REGION Network 4: CALL FB21013 POWDER FEEDER 1 HOPPER UNIT 02
   // 2#0000_0001 OPTIONS 0 BIT 0 LINE 1 ENABLED OPTION
   // 2#0000_0010 OPTIONS 0 BIT 1 LINE 2 ENABLED OPTION
   // 2#0000_0100 OPTIONS 0 BIT 2 SPARE
   // 2#0000_1000 OPTIONS 0 BIT 3 SPARE
   // 2#0001_0000 OPTIONS 0 BIT 4 SPARE
   // 2#0010_0000 OPTIONS 0 BIT 5 SPARE
   // 2#0100_0000 OPTIONS 0 BIT 6 SPARE
   // 2#1000_0000 OPTIONS 0 BIT 7 SPARE
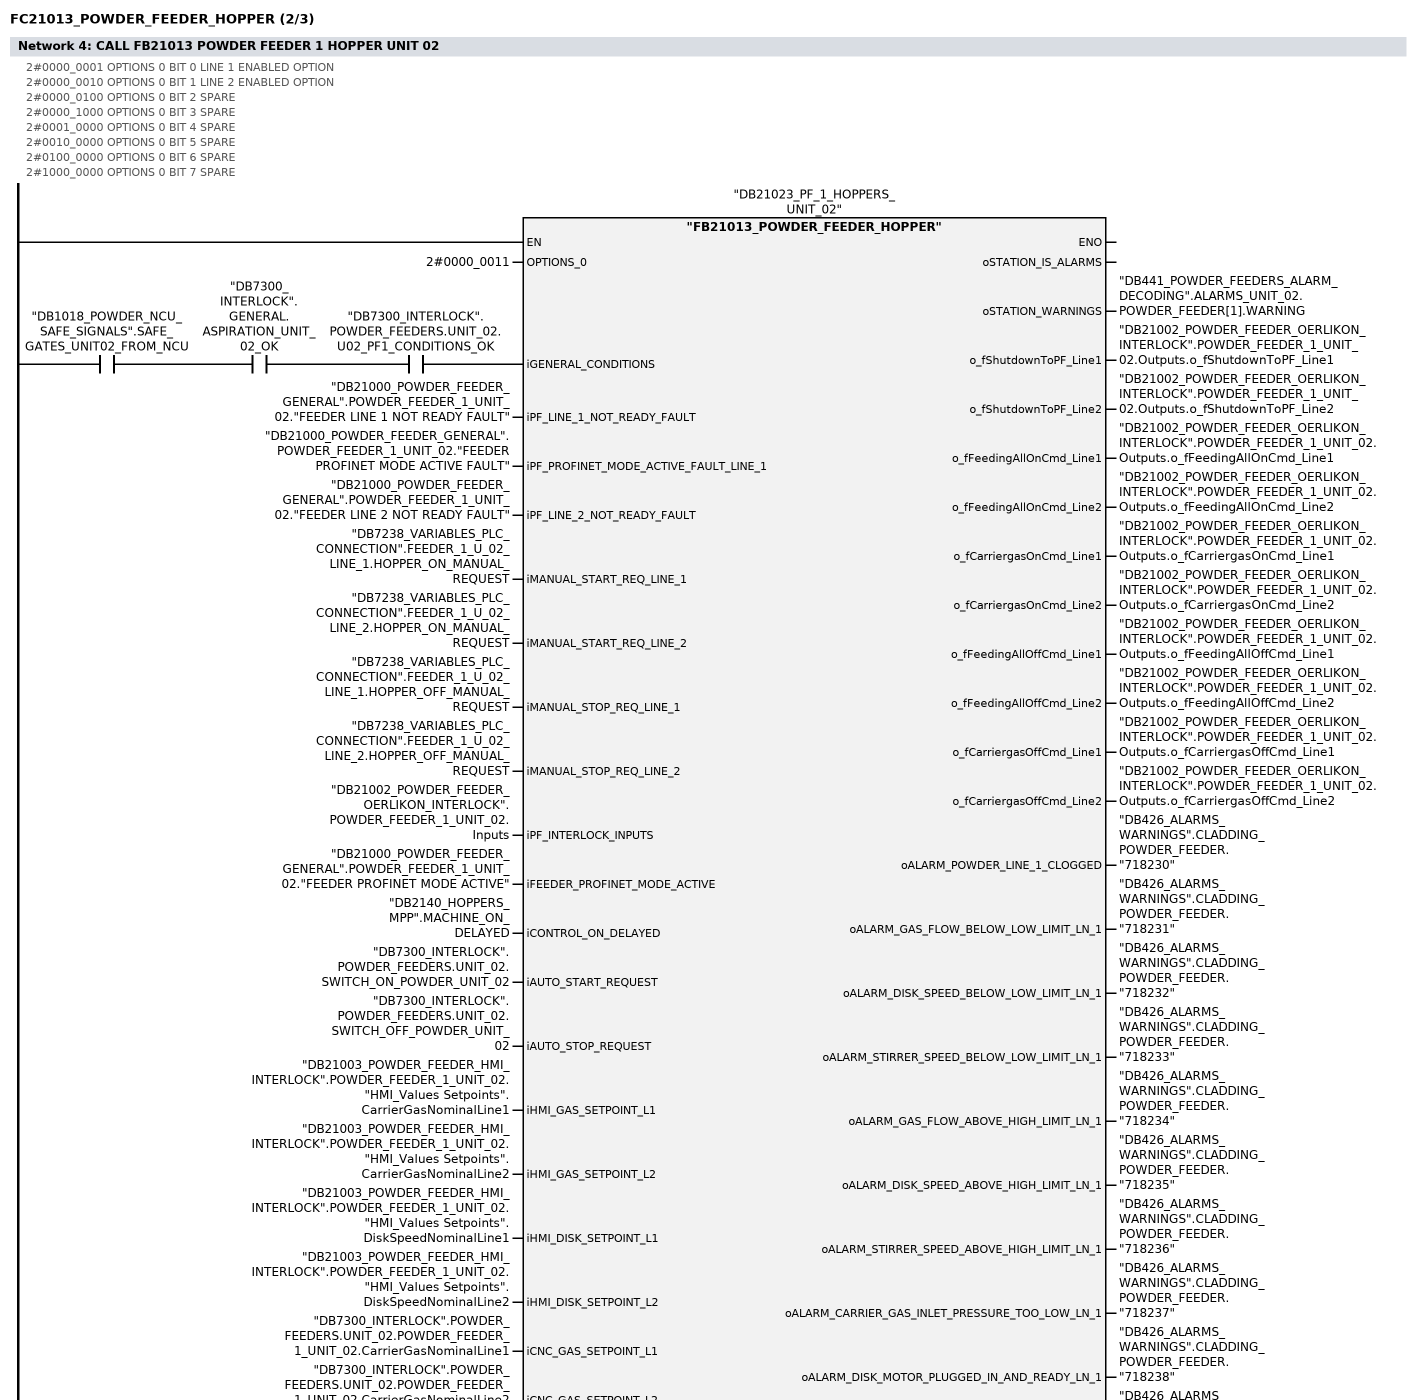
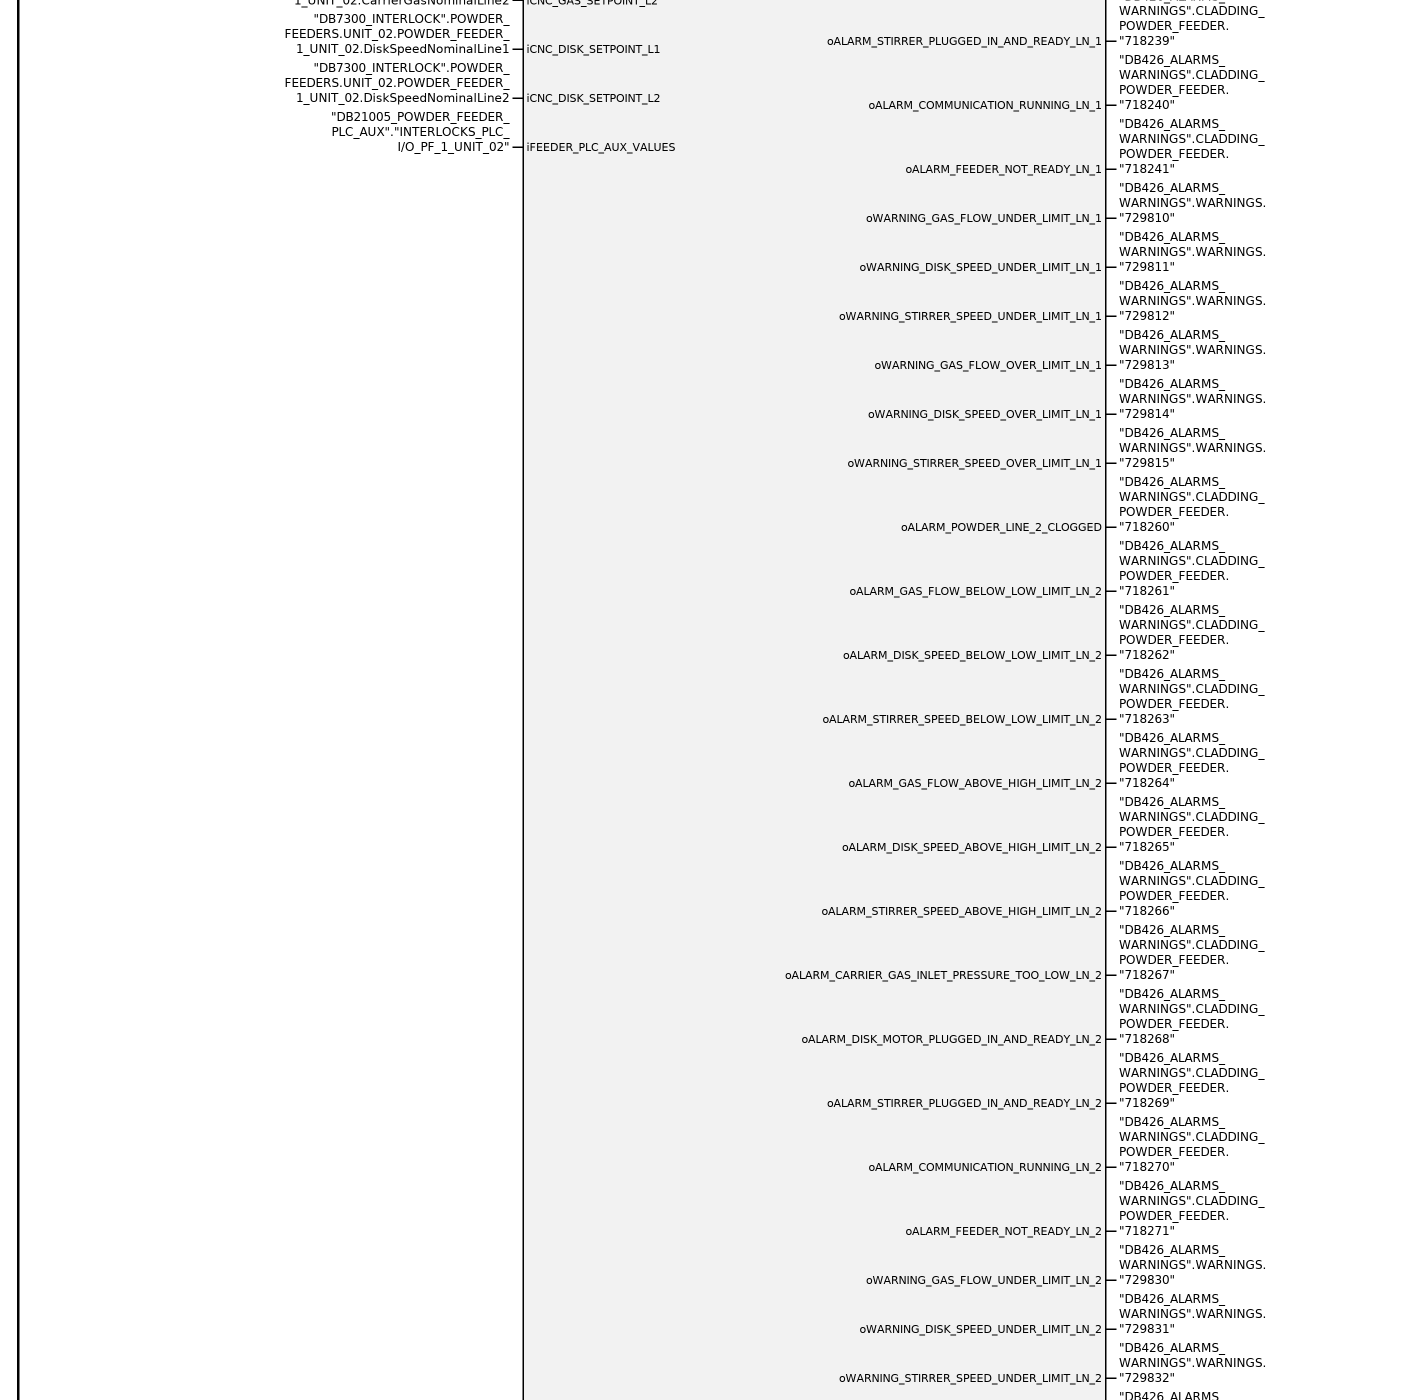
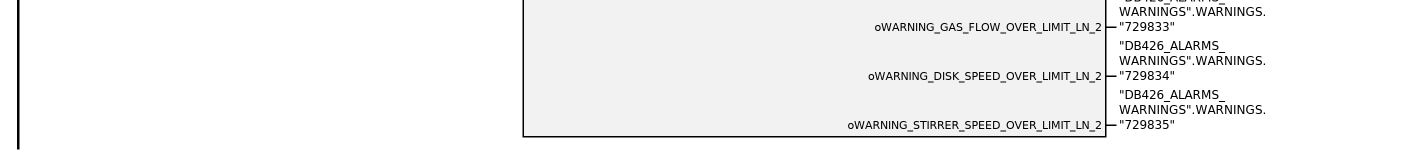
   RUNG wire#powerrail
      "DB21023_PF_1_HOPPERS_UNIT_02"(iGENERAL_CONDITIONS := wire#w1, OPTIONS_0 := 2#0000_0011, iPF_LINE_1_NOT_READY_FAULT := "DB21000_POWDER_FEEDER_GENERAL".POWDER_FEEDER_1_UNIT_02."FEEDER LINE 1 NOT READY FAULT", iPF_PROFINET_MODE_ACTIVE_FAULT_LINE_1 := "DB21000_POWDER_FEEDER_GENERAL".POWDER_FEEDER_1_UNIT_02."FEEDER PROFINET MODE ACTIVE FAULT", iPF_LINE_2_NOT_READY_FAULT := "DB21000_POWDER_FEEDER_GENERAL".POWDER_FEEDER_1_UNIT_02."FEEDER LINE 2 NOT READY FAULT", iMANUAL_START_REQ_LINE_1 := "DB7238_VARIABLES_PLC_CONNECTION".FEEDER_1_U_02_LINE_1.HOPPER_ON_MANUAL_REQUEST, iMANUAL_START_REQ_LINE_2 := "DB7238_VARIABLES_PLC_CONNECTION".FEEDER_1_U_02_LINE_2.HOPPER_ON_MANUAL_REQUEST, iMANUAL_STOP_REQ_LINE_1 := "DB7238_VARIABLES_PLC_CONNECTION".FEEDER_1_U_02_LINE_1.HOPPER_OFF_MANUAL_REQUEST, iMANUAL_STOP_REQ_LINE_2 := "DB7238_VARIABLES_PLC_CONNECTION".FEEDER_1_U_02_LINE_2.HOPPER_OFF_MANUAL_REQUEST, iPF_INTERLOCK_INPUTS := "DB21002_POWDER_FEEDER_OERLIKON_INTERLOCK".POWDER_FEEDER_1_UNIT_02.Inputs, iFEEDER_PROFINET_MODE_ACTIVE := "DB21000_POWDER_FEEDER_GENERAL".POWDER_FEEDER_1_UNIT_02."FEEDER PROFINET MODE ACTIVE", iCONTROL_ON_DELAYED := "DB2140_HOPPERS_MPP".MACHINE_ON_DELAYED, iAUTO_START_REQUEST := "DB7300_INTERLOCK".POWDER_FEEDERS.UNIT_02.SWITCH_ON_POWDER_UNIT_02, iAUTO_STOP_REQUEST := "DB7300_INTERLOCK".POWDER_FEEDERS.UNIT_02.SWITCH_OFF_POWDER_UNIT_02, iHMI_GAS_SETPOINT_L1 := "DB21003_POWDER_FEEDER_HMI_INTERLOCK".POWDER_FEEDER_1_UNIT_02."HMI_Values Setpoints".CarrierGasNominalLine1, iHMI_GAS_SETPOINT_L2 := "DB21003_POWDER_FEEDER_HMI_INTERLOCK".POWDER_FEEDER_1_UNIT_02."HMI_Values Setpoints".CarrierGasNominalLine2, iHMI_DISK_SETPOINT_L1 := "DB21003_POWDER_FEEDER_HMI_INTERLOCK".POWDER_FEEDER_1_UNIT_02."HMI_Values Setpoints".DiskSpeedNominalLine1, iHMI_DISK_SETPOINT_L2 := "DB21003_POWDER_FEEDER_HMI_INTERLOCK".POWDER_FEEDER_1_UNIT_02."HMI_Values Setpoints".DiskSpeedNominalLine2, iCNC_GAS_SETPOINT_L1 := "DB7300_INTERLOCK".POWDER_FEEDERS.UNIT_02.POWDER_FEEDER_1_UNIT_02.CarrierGasNominalLine1, iCNC_GAS_SETPOINT_L2 := "DB7300_INTERLOCK".POWDER_FEEDERS.UNIT_02.POWDER_FEEDER_1_UNIT_02.CarrierGasNominalLine2, iCNC_DISK_SETPOINT_L1 := "DB7300_INTERLOCK".POWDER_FEEDERS.UNIT_02.POWDER_FEEDER_1_UNIT_02.DiskSpeedNominalLine1, iCNC_DISK_SETPOINT_L2 := "DB7300_INTERLOCK".POWDER_FEEDERS.UNIT_02.POWDER_FEEDER_1_UNIT_02.DiskSpeedNominalLine2, iFEEDER_PLC_AUX_VALUES := "DB21005_POWDER_FEEDER_PLC_AUX"."INTERLOCKS_PLC_I/O_PF_1_UNIT_02", oSTATION_IS_ALARMS =>, oSTATION_WARNINGS => "DB441_POWDER_FEEDERS_ALARM_DECODING".ALARMS_UNIT_02.POWDER_FEEDER[1].WARNING, o_fShutdownToPF_Line1 => "DB21002_POWDER_FEEDER_OERLIKON_INTERLOCK".POWDER_FEEDER_1_UNIT_02.Outputs.o_fShutdownToPF_Line1, o_fShutdownToPF_Line2 => "DB21002_POWDER_FEEDER_OERLIKON_INTERLOCK".POWDER_FEEDER_1_UNIT_02.Outputs.o_fShutdownToPF_Line2, o_fFeedingAllOnCmd_Line1 => "DB21002_POWDER_FEEDER_OERLIKON_INTERLOCK".POWDER_FEEDER_1_UNIT_02.Outputs.o_fFeedingAllOnCmd_Line1, o_fFeedingAllOnCmd_Line2 => "DB21002_POWDER_FEEDER_OERLIKON_INTERLOCK".POWDER_FEEDER_1_UNIT_02.Outputs.o_fFeedingAllOnCmd_Line2, o_fCarriergasOnCmd_Line1 => "DB21002_POWDER_FEEDER_OERLIKON_INTERLOCK".POWDER_FEEDER_1_UNIT_02.Outputs.o_fCarriergasOnCmd_Line1, o_fCarriergasOnCmd_Line2 => "DB21002_POWDER_FEEDER_OERLIKON_INTERLOCK".POWDER_FEEDER_1_UNIT_02.Outputs.o_fCarriergasOnCmd_Line2, o_fFeedingAllOffCmd_Line1 => "DB21002_POWDER_FEEDER_OERLIKON_INTERLOCK".POWDER_FEEDER_1_UNIT_02.Outputs.o_fFeedingAllOffCmd_Line1, o_fFeedingAllOffCmd_Line2 => "DB21002_POWDER_FEEDER_OERLIKON_INTERLOCK".POWDER_FEEDER_1_UNIT_02.Outputs.o_fFeedingAllOffCmd_Line2, o_fCarriergasOffCmd_Line1 => "DB21002_POWDER_FEEDER_OERLIKON_INTERLOCK".POWDER_FEEDER_1_UNIT_02.Outputs.o_fCarriergasOffCmd_Line1, o_fCarriergasOffCmd_Line2 => "DB21002_POWDER_FEEDER_OERLIKON_INTERLOCK".POWDER_FEEDER_1_UNIT_02.Outputs.o_fCarriergasOffCmd_Line2, oALARM_POWDER_LINE_1_CLOGGED => "DB426_ALARMS_WARNINGS".CLADDING_POWDER_FEEDER."718230", oALARM_GAS_FLOW_BELOW_LOW_LIMIT_LN_1 => "DB426_ALARMS_WARNINGS".CLADDING_POWDER_FEEDER."718231", oALARM_DISK_SPEED_BELOW_LOW_LIMIT_LN_1 => "DB426_ALARMS_WARNINGS".CLADDING_POWDER_FEEDER."718232", oALARM_STIRRER_SPEED_BELOW_LOW_LIMIT_LN_1 => "DB426_ALARMS_WARNINGS".CLADDING_POWDER_FEEDER."718233", oALARM_GAS_FLOW_ABOVE_HIGH_LIMIT_LN_1 => "DB426_ALARMS_WARNINGS".CLADDING_POWDER_FEEDER."718234", oALARM_DISK_SPEED_ABOVE_HIGH_LIMIT_LN_1 => "DB426_ALARMS_WARNINGS".CLADDING_POWDER_FEEDER."718235", oALARM_STIRRER_SPEED_ABOVE_HIGH_LIMIT_LN_1 => "DB426_ALARMS_WARNINGS".CLADDING_POWDER_FEEDER."718236", oALARM_CARRIER_GAS_INLET_PRESSURE_TOO_LOW_LN_1 => "DB426_ALARMS_WARNINGS".CLADDING_POWDER_FEEDER."718237", oALARM_DISK_MOTOR_PLUGGED_IN_AND_READY_LN_1 => "DB426_ALARMS_WARNINGS".CLADDING_POWDER_FEEDER."718238", oALARM_STIRRER_PLUGGED_IN_AND_READY_LN_1 => "DB426_ALARMS_WARNINGS".CLADDING_POWDER_FEEDER."718239", oALARM_COMMUNICATION_RUNNING_LN_1 => "DB426_ALARMS_WARNINGS".CLADDING_POWDER_FEEDER."718240", oALARM_FEEDER_NOT_READY_LN_1 => "DB426_ALARMS_WARNINGS".CLADDING_POWDER_FEEDER."718241", oWARNING_GAS_FLOW_UNDER_LIMIT_LN_1 => "DB426_ALARMS_WARNINGS".WARNINGS."729810", oWARNING_DISK_SPEED_UNDER_LIMIT_LN_1 => "DB426_ALARMS_WARNINGS".WARNINGS."729811", oWARNING_STIRRER_SPEED_UNDER_LIMIT_LN_1 => "DB426_ALARMS_WARNINGS".WARNINGS."729812", oWARNING_GAS_FLOW_OVER_LIMIT_LN_1 => "DB426_ALARMS_WARNINGS".WARNINGS."729813", oWARNING_DISK_SPEED_OVER_LIMIT_LN_1 => "DB426_ALARMS_WARNINGS".WARNINGS."729814", oWARNING_STIRRER_SPEED_OVER_LIMIT_LN_1 => "DB426_ALARMS_WARNINGS".WARNINGS."729815", oALARM_POWDER_LINE_2_CLOGGED => "DB426_ALARMS_WARNINGS".CLADDING_POWDER_FEEDER."718260", oALARM_GAS_FLOW_BELOW_LOW_LIMIT_LN_2 => "DB426_ALARMS_WARNINGS".CLADDING_POWDER_FEEDER."718261", oALARM_DISK_SPEED_BELOW_LOW_LIMIT_LN_2 => "DB426_ALARMS_WARNINGS".CLADDING_POWDER_FEEDER."718262", oALARM_STIRRER_SPEED_BELOW_LOW_LIMIT_LN_2 => "DB426_ALARMS_WARNINGS".CLADDING_POWDER_FEEDER."718263", oALARM_GAS_FLOW_ABOVE_HIGH_LIMIT_LN_2 => "DB426_ALARMS_WARNINGS".CLADDING_POWDER_FEEDER."718264", oALARM_DISK_SPEED_ABOVE_HIGH_LIMIT_LN_2 => "DB426_ALARMS_WARNINGS".CLADDING_POWDER_FEEDER."718265", oALARM_STIRRER_SPEED_ABOVE_HIGH_LIMIT_LN_2 => "DB426_ALARMS_WARNINGS".CLADDING_POWDER_FEEDER."718266", oALARM_CARRIER_GAS_INLET_PRESSURE_TOO_LOW_LN_2 => "DB426_ALARMS_WARNINGS".CLADDING_POWDER_FEEDER."718267", oALARM_DISK_MOTOR_PLUGGED_IN_AND_READY_LN_2 => "DB426_ALARMS_WARNINGS".CLADDING_POWDER_FEEDER."718268", oALARM_STIRRER_PLUGGED_IN_AND_READY_LN_2 => "DB426_ALARMS_WARNINGS".CLADDING_POWDER_FEEDER."718269", oALARM_COMMUNICATION_RUNNING_LN_2 => "DB426_ALARMS_WARNINGS".CLADDING_POWDER_FEEDER."718270", oALARM_FEEDER_NOT_READY_LN_2 => "DB426_ALARMS_WARNINGS".CLADDING_POWDER_FEEDER."718271", oWARNING_GAS_FLOW_UNDER_LIMIT_LN_2 => "DB426_ALARMS_WARNINGS".WARNINGS."729830", oWARNING_DISK_SPEED_UNDER_LIMIT_LN_2 => "DB426_ALARMS_WARNINGS".WARNINGS."729831", oWARNING_STIRRER_SPEED_UNDER_LIMIT_LN_2 => "DB426_ALARMS_WARNINGS".WARNINGS."729832", oWARNING_GAS_FLOW_OVER_LIMIT_LN_2 => "DB426_ALARMS_WARNINGS".WARNINGS."729833", oWARNING_DISK_SPEED_OVER_LIMIT_LN_2 => "DB426_ALARMS_WARNINGS".WARNINGS."729834", oWARNING_STIRRER_SPEED_OVER_LIMIT_LN_2 => "DB426_ALARMS_WARNINGS".WARNINGS."729835")
   END_RUNG
   RUNG wire#powerrail
      Contact( "DB1018_POWDER_NCU_SAFE_SIGNALS".SAFE_GATES_UNIT02_FROM_NCU )
      Contact( "DB7300_INTERLOCK".GENERAL.ASPIRATION_UNIT_02_OK )
      Contact( "DB7300_INTERLOCK".POWDER_FEEDERS.UNIT_02.U02_PF1_CONDITIONS_OK )
   END_RUNG wire#w1
   // the same network as SCL:
   "DB21023_PF_1_HOPPERS_UNIT_02"(OPTIONS_0 := 2#0000_0011,   // "FB21013_POWDER_FEEDER_HOPPER"
                           iGENERAL_CONDITIONS := "DB1018_POWDER_NCU_SAFE_SIGNALS".SAFE_GATES_UNIT02_FROM_NCU AND "DB7300_INTERLOCK".GENERAL.ASPIRATION_UNIT_02_OK AND "DB7300_INTERLOCK".POWDER_FEEDERS.UNIT_02.U02_PF1_CONDITIONS_OK,
                           iPF_LINE_1_NOT_READY_FAULT := "DB21000_POWDER_FEEDER_GENERAL".POWDER_FEEDER_1_UNIT_02."FEEDER LINE 1 NOT READY FAULT",
                           iPF_PROFINET_MODE_ACTIVE_FAULT_LINE_1 := "DB21000_POWDER_FEEDER_GENERAL".POWDER_FEEDER_1_UNIT_02."FEEDER PROFINET MODE ACTIVE FAULT",
                           iPF_LINE_2_NOT_READY_FAULT := "DB21000_POWDER_FEEDER_GENERAL".POWDER_FEEDER_1_UNIT_02."FEEDER LINE 2 NOT READY FAULT",
                           iMANUAL_START_REQ_LINE_1 := "DB7238_VARIABLES_PLC_CONNECTION".FEEDER_1_U_02_LINE_1.HOPPER_ON_MANUAL_REQUEST,
                           iMANUAL_START_REQ_LINE_2 := "DB7238_VARIABLES_PLC_CONNECTION".FEEDER_1_U_02_LINE_2.HOPPER_ON_MANUAL_REQUEST,
                           iMANUAL_STOP_REQ_LINE_1 := "DB7238_VARIABLES_PLC_CONNECTION".FEEDER_1_U_02_LINE_1.HOPPER_OFF_MANUAL_REQUEST,
                           iMANUAL_STOP_REQ_LINE_2 := "DB7238_VARIABLES_PLC_CONNECTION".FEEDER_1_U_02_LINE_2.HOPPER_OFF_MANUAL_REQUEST,
                           iPF_INTERLOCK_INPUTS := "DB21002_POWDER_FEEDER_OERLIKON_INTERLOCK".POWDER_FEEDER_1_UNIT_02.Inputs,
                           iFEEDER_PROFINET_MODE_ACTIVE := "DB21000_POWDER_FEEDER_GENERAL".POWDER_FEEDER_1_UNIT_02."FEEDER PROFINET MODE ACTIVE",
                           iCONTROL_ON_DELAYED := "DB2140_HOPPERS_MPP".MACHINE_ON_DELAYED,
                           iAUTO_START_REQUEST := "DB7300_INTERLOCK".POWDER_FEEDERS.UNIT_02.SWITCH_ON_POWDER_UNIT_02,
                           iAUTO_STOP_REQUEST := "DB7300_INTERLOCK".POWDER_FEEDERS.UNIT_02.SWITCH_OFF_POWDER_UNIT_02,
                           iHMI_GAS_SETPOINT_L1 := "DB21003_POWDER_FEEDER_HMI_INTERLOCK".POWDER_FEEDER_1_UNIT_02."HMI_Values Setpoints".CarrierGasNominalLine1,
                           iHMI_GAS_SETPOINT_L2 := "DB21003_POWDER_FEEDER_HMI_INTERLOCK".POWDER_FEEDER_1_UNIT_02."HMI_Values Setpoints".CarrierGasNominalLine2,
                           iHMI_DISK_SETPOINT_L1 := "DB21003_POWDER_FEEDER_HMI_INTERLOCK".POWDER_FEEDER_1_UNIT_02."HMI_Values Setpoints".DiskSpeedNominalLine1,
                           iHMI_DISK_SETPOINT_L2 := "DB21003_POWDER_FEEDER_HMI_INTERLOCK".POWDER_FEEDER_1_UNIT_02."HMI_Values Setpoints".DiskSpeedNominalLine2,
                           iCNC_GAS_SETPOINT_L1 := "DB7300_INTERLOCK".POWDER_FEEDERS.UNIT_02.POWDER_FEEDER_1_UNIT_02.CarrierGasNominalLine1,
                           iCNC_GAS_SETPOINT_L2 := "DB7300_INTERLOCK".POWDER_FEEDERS.UNIT_02.POWDER_FEEDER_1_UNIT_02.CarrierGasNominalLine2,
                           iCNC_DISK_SETPOINT_L1 := "DB7300_INTERLOCK".POWDER_FEEDERS.UNIT_02.POWDER_FEEDER_1_UNIT_02.DiskSpeedNominalLine1,
                           iCNC_DISK_SETPOINT_L2 := "DB7300_INTERLOCK".POWDER_FEEDERS.UNIT_02.POWDER_FEEDER_1_UNIT_02.DiskSpeedNominalLine2,
                           iFEEDER_PLC_AUX_VALUES := "DB21005_POWDER_FEEDER_PLC_AUX"."INTERLOCKS_PLC_I/O_PF_1_UNIT_02",
                           oSTATION_WARNINGS => "DB441_POWDER_FEEDERS_ALARM_DECODING".ALARMS_UNIT_02.POWDER_FEEDER[1].WARNING,
                           o_fShutdownToPF_Line1 => "DB21002_POWDER_FEEDER_OERLIKON_INTERLOCK".POWDER_FEEDER_1_UNIT_02.Outputs.o_fShutdownToPF_Line1,
                           o_fShutdownToPF_Line2 => "DB21002_POWDER_FEEDER_OERLIKON_INTERLOCK".POWDER_FEEDER_1_UNIT_02.Outputs.o_fShutdownToPF_Line2,
                           o_fFeedingAllOnCmd_Line1 => "DB21002_POWDER_FEEDER_OERLIKON_INTERLOCK".POWDER_FEEDER_1_UNIT_02.Outputs.o_fFeedingAllOnCmd_Line1,
                           o_fFeedingAllOnCmd_Line2 => "DB21002_POWDER_FEEDER_OERLIKON_INTERLOCK".POWDER_FEEDER_1_UNIT_02.Outputs.o_fFeedingAllOnCmd_Line2,
                           o_fCarriergasOnCmd_Line1 => "DB21002_POWDER_FEEDER_OERLIKON_INTERLOCK".POWDER_FEEDER_1_UNIT_02.Outputs.o_fCarriergasOnCmd_Line1,
                           o_fCarriergasOnCmd_Line2 => "DB21002_POWDER_FEEDER_OERLIKON_INTERLOCK".POWDER_FEEDER_1_UNIT_02.Outputs.o_fCarriergasOnCmd_Line2,
                           o_fFeedingAllOffCmd_Line1 => "DB21002_POWDER_FEEDER_OERLIKON_INTERLOCK".POWDER_FEEDER_1_UNIT_02.Outputs.o_fFeedingAllOffCmd_Line1,
                           o_fFeedingAllOffCmd_Line2 => "DB21002_POWDER_FEEDER_OERLIKON_INTERLOCK".POWDER_FEEDER_1_UNIT_02.Outputs.o_fFeedingAllOffCmd_Line2,
                           o_fCarriergasOffCmd_Line1 => "DB21002_POWDER_FEEDER_OERLIKON_INTERLOCK".POWDER_FEEDER_1_UNIT_02.Outputs.o_fCarriergasOffCmd_Line1,
                           o_fCarriergasOffCmd_Line2 => "DB21002_POWDER_FEEDER_OERLIKON_INTERLOCK".POWDER_FEEDER_1_UNIT_02.Outputs.o_fCarriergasOffCmd_Line2,
                           oALARM_POWDER_LINE_1_CLOGGED => "DB426_ALARMS_WARNINGS".CLADDING_POWDER_FEEDER."718230",
                           oALARM_GAS_FLOW_BELOW_LOW_LIMIT_LN_1 => "DB426_ALARMS_WARNINGS".CLADDING_POWDER_FEEDER."718231",
                           oALARM_DISK_SPEED_BELOW_LOW_LIMIT_LN_1 => "DB426_ALARMS_WARNINGS".CLADDING_POWDER_FEEDER."718232",
                           oALARM_STIRRER_SPEED_BELOW_LOW_LIMIT_LN_1 => "DB426_ALARMS_WARNINGS".CLADDING_POWDER_FEEDER."718233",
                           oALARM_GAS_FLOW_ABOVE_HIGH_LIMIT_LN_1 => "DB426_ALARMS_WARNINGS".CLADDING_POWDER_FEEDER."718234",
                           oALARM_DISK_SPEED_ABOVE_HIGH_LIMIT_LN_1 => "DB426_ALARMS_WARNINGS".CLADDING_POWDER_FEEDER."718235",
                           oALARM_STIRRER_SPEED_ABOVE_HIGH_LIMIT_LN_1 => "DB426_ALARMS_WARNINGS".CLADDING_POWDER_FEEDER."718236",
                           oALARM_CARRIER_GAS_INLET_PRESSURE_TOO_LOW_LN_1 => "DB426_ALARMS_WARNINGS".CLADDING_POWDER_FEEDER."718237",
                           oALARM_DISK_MOTOR_PLUGGED_IN_AND_READY_LN_1 => "DB426_ALARMS_WARNINGS".CLADDING_POWDER_FEEDER."718238",
                           oALARM_STIRRER_PLUGGED_IN_AND_READY_LN_1 => "DB426_ALARMS_WARNINGS".CLADDING_POWDER_FEEDER."718239",
                           oALARM_COMMUNICATION_RUNNING_LN_1 => "DB426_ALARMS_WARNINGS".CLADDING_POWDER_FEEDER."718240",
                           oALARM_FEEDER_NOT_READY_LN_1 => "DB426_ALARMS_WARNINGS".CLADDING_POWDER_FEEDER."718241",
                           oWARNING_GAS_FLOW_UNDER_LIMIT_LN_1 => "DB426_ALARMS_WARNINGS".WARNINGS."729810",
                           oWARNING_DISK_SPEED_UNDER_LIMIT_LN_1 => "DB426_ALARMS_WARNINGS".WARNINGS."729811",
                           oWARNING_STIRRER_SPEED_UNDER_LIMIT_LN_1 => "DB426_ALARMS_WARNINGS".WARNINGS."729812",
                           oWARNING_GAS_FLOW_OVER_LIMIT_LN_1 => "DB426_ALARMS_WARNINGS".WARNINGS."729813",
                           oWARNING_DISK_SPEED_OVER_LIMIT_LN_1 => "DB426_ALARMS_WARNINGS".WARNINGS."729814",
                           oWARNING_STIRRER_SPEED_OVER_LIMIT_LN_1 => "DB426_ALARMS_WARNINGS".WARNINGS."729815",
                           oALARM_POWDER_LINE_2_CLOGGED => "DB426_ALARMS_WARNINGS".CLADDING_POWDER_FEEDER."718260",
                           oALARM_GAS_FLOW_BELOW_LOW_LIMIT_LN_2 => "DB426_ALARMS_WARNINGS".CLADDING_POWDER_FEEDER."718261",
                           oALARM_DISK_SPEED_BELOW_LOW_LIMIT_LN_2 => "DB426_ALARMS_WARNINGS".CLADDING_POWDER_FEEDER."718262",
                           oALARM_STIRRER_SPEED_BELOW_LOW_LIMIT_LN_2 => "DB426_ALARMS_WARNINGS".CLADDING_POWDER_FEEDER."718263",
                           oALARM_GAS_FLOW_ABOVE_HIGH_LIMIT_LN_2 => "DB426_ALARMS_WARNINGS".CLADDING_POWDER_FEEDER."718264",
                           oALARM_DISK_SPEED_ABOVE_HIGH_LIMIT_LN_2 => "DB426_ALARMS_WARNINGS".CLADDING_POWDER_FEEDER."718265",
                           oALARM_STIRRER_SPEED_ABOVE_HIGH_LIMIT_LN_2 => "DB426_ALARMS_WARNINGS".CLADDING_POWDER_FEEDER."718266",
                           oALARM_CARRIER_GAS_INLET_PRESSURE_TOO_LOW_LN_2 => "DB426_ALARMS_WARNINGS".CLADDING_POWDER_FEEDER."718267",
                           oALARM_DISK_MOTOR_PLUGGED_IN_AND_READY_LN_2 => "DB426_ALARMS_WARNINGS".CLADDING_POWDER_FEEDER."718268",
                           oALARM_STIRRER_PLUGGED_IN_AND_READY_LN_2 => "DB426_ALARMS_WARNINGS".CLADDING_POWDER_FEEDER."718269",
                           oALARM_COMMUNICATION_RUNNING_LN_2 => "DB426_ALARMS_WARNINGS".CLADDING_POWDER_FEEDER."718270",
                           oALARM_FEEDER_NOT_READY_LN_2 => "DB426_ALARMS_WARNINGS".CLADDING_POWDER_FEEDER."718271",
                           oWARNING_GAS_FLOW_UNDER_LIMIT_LN_2 => "DB426_ALARMS_WARNINGS".WARNINGS."729830",
                           oWARNING_DISK_SPEED_UNDER_LIMIT_LN_2 => "DB426_ALARMS_WARNINGS".WARNINGS."729831",
                           oWARNING_STIRRER_SPEED_UNDER_LIMIT_LN_2 => "DB426_ALARMS_WARNINGS".WARNINGS."729832",
                           oWARNING_GAS_FLOW_OVER_LIMIT_LN_2 => "DB426_ALARMS_WARNINGS".WARNINGS."729833",
                           oWARNING_DISK_SPEED_OVER_LIMIT_LN_2 => "DB426_ALARMS_WARNINGS".WARNINGS."729834",
                           oWARNING_STIRRER_SPEED_OVER_LIMIT_LN_2 => "DB426_ALARMS_WARNINGS".WARNINGS."729835");
END_REGION

REGION Network 5: CALL FB21013 POWDER FEEDER 2 HOPPER UNIT 02
   // 2#0000_0001 OPTIONS 0 BIT 0 LINE 1 ENABLED OPTION
   // 2#0000_0010 OPTIONS 0 BIT 1 LINE 2 ENABLED OPTION
   // 2#0000_0100 OPTIONS 0 BIT 2 SPARE
   // 2#0000_1000 OPTIONS 0 BIT 3 SPARE
   // 2#0001_0000 OPTIONS 0 BIT 4 SPARE
   // 2#0010_0000 OPTIONS 0 BIT 5 SPARE
   // 2#0100_0000 OPTIONS 0 BIT 6 SPARE
   // 2#1000_0000 OPTIONS 0 BIT 7 SPARE
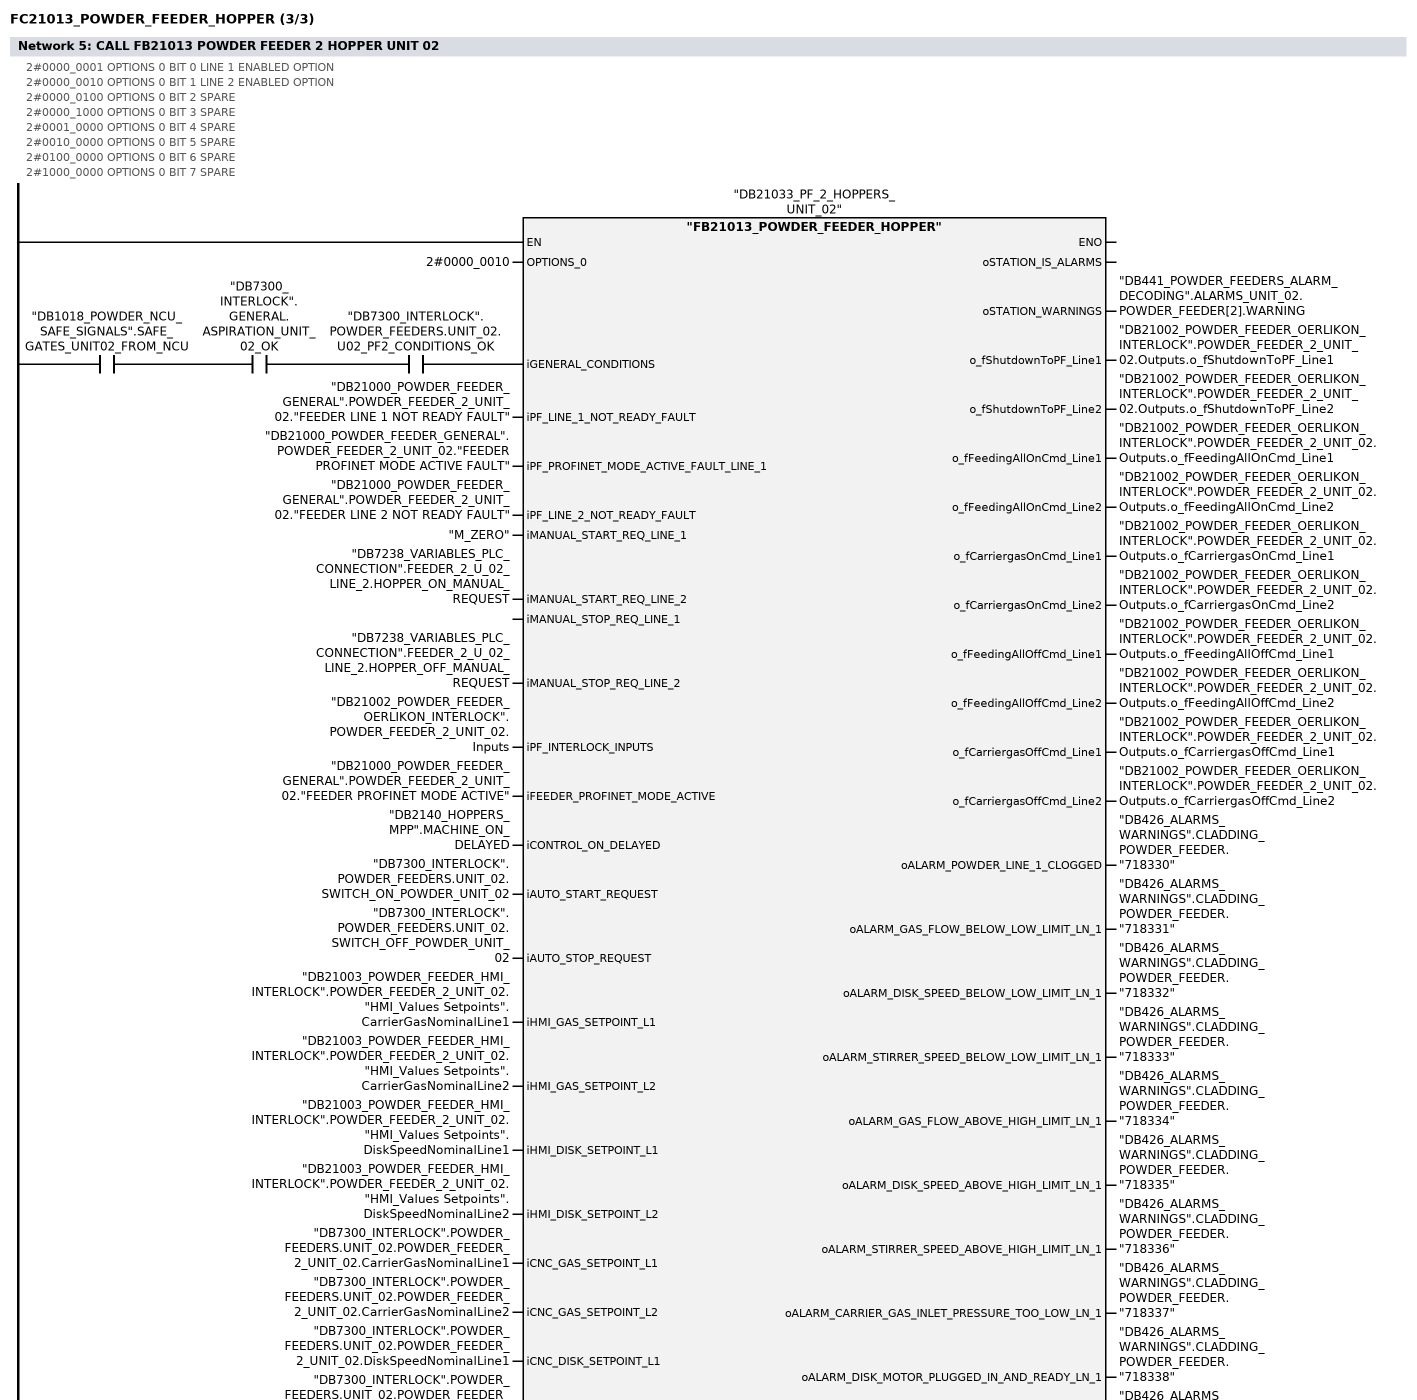
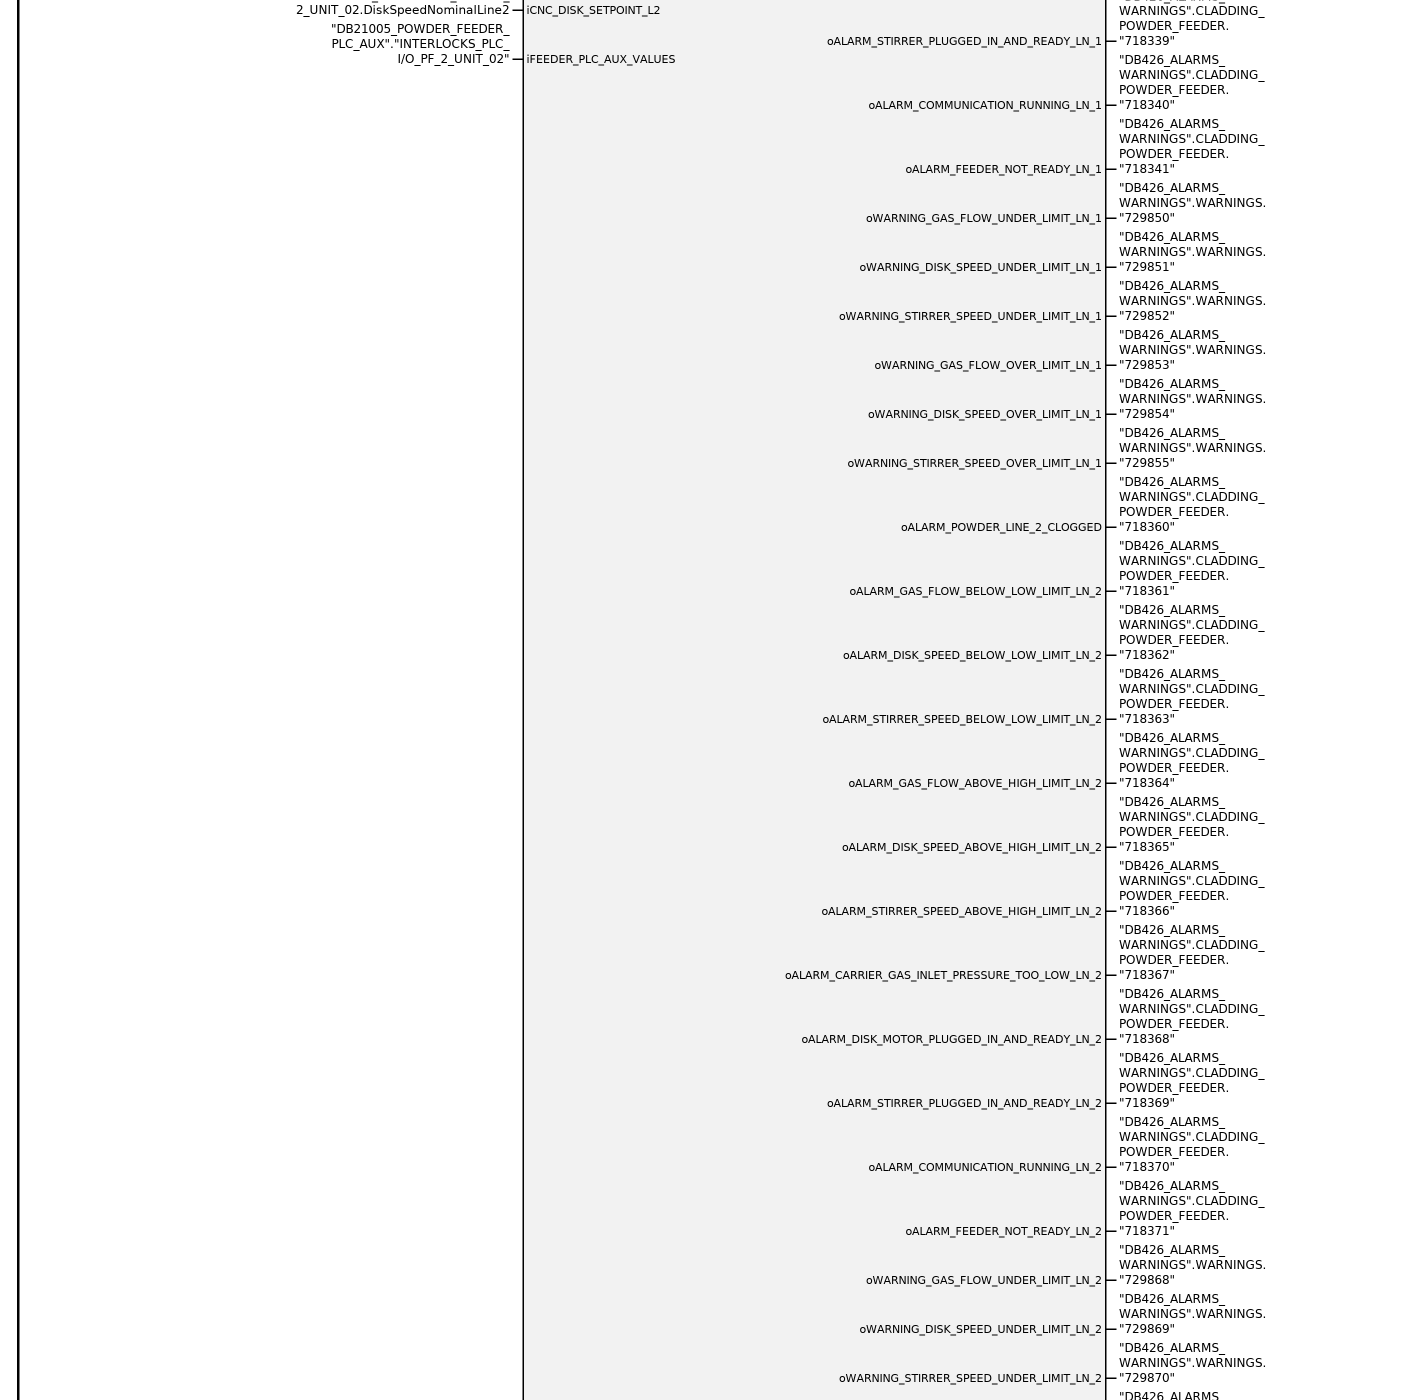
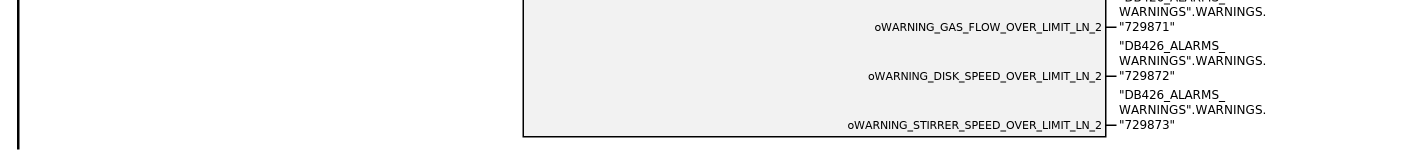
   RUNG wire#powerrail
      "DB21033_PF_2_HOPPERS_UNIT_02"(iGENERAL_CONDITIONS := wire#w1, OPTIONS_0 := 2#0000_0010, iPF_LINE_1_NOT_READY_FAULT := "DB21000_POWDER_FEEDER_GENERAL".POWDER_FEEDER_2_UNIT_02."FEEDER LINE 1 NOT READY FAULT", iPF_PROFINET_MODE_ACTIVE_FAULT_LINE_1 := "DB21000_POWDER_FEEDER_GENERAL".POWDER_FEEDER_2_UNIT_02."FEEDER PROFINET MODE ACTIVE FAULT", iPF_LINE_2_NOT_READY_FAULT := "DB21000_POWDER_FEEDER_GENERAL".POWDER_FEEDER_2_UNIT_02."FEEDER LINE 2 NOT READY FAULT", iMANUAL_START_REQ_LINE_1 := "M_ZERO", iMANUAL_START_REQ_LINE_2 := "DB7238_VARIABLES_PLC_CONNECTION".FEEDER_2_U_02_LINE_2.HOPPER_ON_MANUAL_REQUEST, iMANUAL_STOP_REQ_LINE_1 :=, iMANUAL_STOP_REQ_LINE_2 := "DB7238_VARIABLES_PLC_CONNECTION".FEEDER_2_U_02_LINE_2.HOPPER_OFF_MANUAL_REQUEST, iPF_INTERLOCK_INPUTS := "DB21002_POWDER_FEEDER_OERLIKON_INTERLOCK".POWDER_FEEDER_2_UNIT_02.Inputs, iFEEDER_PROFINET_MODE_ACTIVE := "DB21000_POWDER_FEEDER_GENERAL".POWDER_FEEDER_2_UNIT_02."FEEDER PROFINET MODE ACTIVE", iCONTROL_ON_DELAYED := "DB2140_HOPPERS_MPP".MACHINE_ON_DELAYED, iAUTO_START_REQUEST := "DB7300_INTERLOCK".POWDER_FEEDERS.UNIT_02.SWITCH_ON_POWDER_UNIT_02, iAUTO_STOP_REQUEST := "DB7300_INTERLOCK".POWDER_FEEDERS.UNIT_02.SWITCH_OFF_POWDER_UNIT_02, iHMI_GAS_SETPOINT_L1 := "DB21003_POWDER_FEEDER_HMI_INTERLOCK".POWDER_FEEDER_2_UNIT_02."HMI_Values Setpoints".CarrierGasNominalLine1, iHMI_GAS_SETPOINT_L2 := "DB21003_POWDER_FEEDER_HMI_INTERLOCK".POWDER_FEEDER_2_UNIT_02."HMI_Values Setpoints".CarrierGasNominalLine2, iHMI_DISK_SETPOINT_L1 := "DB21003_POWDER_FEEDER_HMI_INTERLOCK".POWDER_FEEDER_2_UNIT_02."HMI_Values Setpoints".DiskSpeedNominalLine1, iHMI_DISK_SETPOINT_L2 := "DB21003_POWDER_FEEDER_HMI_INTERLOCK".POWDER_FEEDER_2_UNIT_02."HMI_Values Setpoints".DiskSpeedNominalLine2, iCNC_GAS_SETPOINT_L1 := "DB7300_INTERLOCK".POWDER_FEEDERS.UNIT_02.POWDER_FEEDER_2_UNIT_02.CarrierGasNominalLine1, iCNC_GAS_SETPOINT_L2 := "DB7300_INTERLOCK".POWDER_FEEDERS.UNIT_02.POWDER_FEEDER_2_UNIT_02.CarrierGasNominalLine2, iCNC_DISK_SETPOINT_L1 := "DB7300_INTERLOCK".POWDER_FEEDERS.UNIT_02.POWDER_FEEDER_2_UNIT_02.DiskSpeedNominalLine1, iCNC_DISK_SETPOINT_L2 := "DB7300_INTERLOCK".POWDER_FEEDERS.UNIT_02.POWDER_FEEDER_2_UNIT_02.DiskSpeedNominalLine2, iFEEDER_PLC_AUX_VALUES := "DB21005_POWDER_FEEDER_PLC_AUX"."INTERLOCKS_PLC_I/O_PF_2_UNIT_02", oSTATION_IS_ALARMS =>, oSTATION_WARNINGS => "DB441_POWDER_FEEDERS_ALARM_DECODING".ALARMS_UNIT_02.POWDER_FEEDER[2].WARNING, o_fShutdownToPF_Line1 => "DB21002_POWDER_FEEDER_OERLIKON_INTERLOCK".POWDER_FEEDER_2_UNIT_02.Outputs.o_fShutdownToPF_Line1, o_fShutdownToPF_Line2 => "DB21002_POWDER_FEEDER_OERLIKON_INTERLOCK".POWDER_FEEDER_2_UNIT_02.Outputs.o_fShutdownToPF_Line2, o_fFeedingAllOnCmd_Line1 => "DB21002_POWDER_FEEDER_OERLIKON_INTERLOCK".POWDER_FEEDER_2_UNIT_02.Outputs.o_fFeedingAllOnCmd_Line1, o_fFeedingAllOnCmd_Line2 => "DB21002_POWDER_FEEDER_OERLIKON_INTERLOCK".POWDER_FEEDER_2_UNIT_02.Outputs.o_fFeedingAllOnCmd_Line2, o_fCarriergasOnCmd_Line1 => "DB21002_POWDER_FEEDER_OERLIKON_INTERLOCK".POWDER_FEEDER_2_UNIT_02.Outputs.o_fCarriergasOnCmd_Line1, o_fCarriergasOnCmd_Line2 => "DB21002_POWDER_FEEDER_OERLIKON_INTERLOCK".POWDER_FEEDER_2_UNIT_02.Outputs.o_fCarriergasOnCmd_Line2, o_fFeedingAllOffCmd_Line1 => "DB21002_POWDER_FEEDER_OERLIKON_INTERLOCK".POWDER_FEEDER_2_UNIT_02.Outputs.o_fFeedingAllOffCmd_Line1, o_fFeedingAllOffCmd_Line2 => "DB21002_POWDER_FEEDER_OERLIKON_INTERLOCK".POWDER_FEEDER_2_UNIT_02.Outputs.o_fFeedingAllOffCmd_Line2, o_fCarriergasOffCmd_Line1 => "DB21002_POWDER_FEEDER_OERLIKON_INTERLOCK".POWDER_FEEDER_2_UNIT_02.Outputs.o_fCarriergasOffCmd_Line1, o_fCarriergasOffCmd_Line2 => "DB21002_POWDER_FEEDER_OERLIKON_INTERLOCK".POWDER_FEEDER_2_UNIT_02.Outputs.o_fCarriergasOffCmd_Line2, oALARM_POWDER_LINE_1_CLOGGED => "DB426_ALARMS_WARNINGS".CLADDING_POWDER_FEEDER."718330", oALARM_GAS_FLOW_BELOW_LOW_LIMIT_LN_1 => "DB426_ALARMS_WARNINGS".CLADDING_POWDER_FEEDER."718331", oALARM_DISK_SPEED_BELOW_LOW_LIMIT_LN_1 => "DB426_ALARMS_WARNINGS".CLADDING_POWDER_FEEDER."718332", oALARM_STIRRER_SPEED_BELOW_LOW_LIMIT_LN_1 => "DB426_ALARMS_WARNINGS".CLADDING_POWDER_FEEDER."718333", oALARM_GAS_FLOW_ABOVE_HIGH_LIMIT_LN_1 => "DB426_ALARMS_WARNINGS".CLADDING_POWDER_FEEDER."718334", oALARM_DISK_SPEED_ABOVE_HIGH_LIMIT_LN_1 => "DB426_ALARMS_WARNINGS".CLADDING_POWDER_FEEDER."718335", oALARM_STIRRER_SPEED_ABOVE_HIGH_LIMIT_LN_1 => "DB426_ALARMS_WARNINGS".CLADDING_POWDER_FEEDER."718336", oALARM_CARRIER_GAS_INLET_PRESSURE_TOO_LOW_LN_1 => "DB426_ALARMS_WARNINGS".CLADDING_POWDER_FEEDER."718337", oALARM_DISK_MOTOR_PLUGGED_IN_AND_READY_LN_1 => "DB426_ALARMS_WARNINGS".CLADDING_POWDER_FEEDER."718338", oALARM_STIRRER_PLUGGED_IN_AND_READY_LN_1 => "DB426_ALARMS_WARNINGS".CLADDING_POWDER_FEEDER."718339", oALARM_COMMUNICATION_RUNNING_LN_1 => "DB426_ALARMS_WARNINGS".CLADDING_POWDER_FEEDER."718340", oALARM_FEEDER_NOT_READY_LN_1 => "DB426_ALARMS_WARNINGS".CLADDING_POWDER_FEEDER."718341", oWARNING_GAS_FLOW_UNDER_LIMIT_LN_1 => "DB426_ALARMS_WARNINGS".WARNINGS."729850", oWARNING_DISK_SPEED_UNDER_LIMIT_LN_1 => "DB426_ALARMS_WARNINGS".WARNINGS."729851", oWARNING_STIRRER_SPEED_UNDER_LIMIT_LN_1 => "DB426_ALARMS_WARNINGS".WARNINGS."729852", oWARNING_GAS_FLOW_OVER_LIMIT_LN_1 => "DB426_ALARMS_WARNINGS".WARNINGS."729853", oWARNING_DISK_SPEED_OVER_LIMIT_LN_1 => "DB426_ALARMS_WARNINGS".WARNINGS."729854", oWARNING_STIRRER_SPEED_OVER_LIMIT_LN_1 => "DB426_ALARMS_WARNINGS".WARNINGS."729855", oALARM_POWDER_LINE_2_CLOGGED => "DB426_ALARMS_WARNINGS".CLADDING_POWDER_FEEDER."718360", oALARM_GAS_FLOW_BELOW_LOW_LIMIT_LN_2 => "DB426_ALARMS_WARNINGS".CLADDING_POWDER_FEEDER."718361", oALARM_DISK_SPEED_BELOW_LOW_LIMIT_LN_2 => "DB426_ALARMS_WARNINGS".CLADDING_POWDER_FEEDER."718362", oALARM_STIRRER_SPEED_BELOW_LOW_LIMIT_LN_2 => "DB426_ALARMS_WARNINGS".CLADDING_POWDER_FEEDER."718363", oALARM_GAS_FLOW_ABOVE_HIGH_LIMIT_LN_2 => "DB426_ALARMS_WARNINGS".CLADDING_POWDER_FEEDER."718364", oALARM_DISK_SPEED_ABOVE_HIGH_LIMIT_LN_2 => "DB426_ALARMS_WARNINGS".CLADDING_POWDER_FEEDER."718365", oALARM_STIRRER_SPEED_ABOVE_HIGH_LIMIT_LN_2 => "DB426_ALARMS_WARNINGS".CLADDING_POWDER_FEEDER."718366", oALARM_CARRIER_GAS_INLET_PRESSURE_TOO_LOW_LN_2 => "DB426_ALARMS_WARNINGS".CLADDING_POWDER_FEEDER."718367", oALARM_DISK_MOTOR_PLUGGED_IN_AND_READY_LN_2 => "DB426_ALARMS_WARNINGS".CLADDING_POWDER_FEEDER."718368", oALARM_STIRRER_PLUGGED_IN_AND_READY_LN_2 => "DB426_ALARMS_WARNINGS".CLADDING_POWDER_FEEDER."718369", oALARM_COMMUNICATION_RUNNING_LN_2 => "DB426_ALARMS_WARNINGS".CLADDING_POWDER_FEEDER."718370", oALARM_FEEDER_NOT_READY_LN_2 => "DB426_ALARMS_WARNINGS".CLADDING_POWDER_FEEDER."718371", oWARNING_GAS_FLOW_UNDER_LIMIT_LN_2 => "DB426_ALARMS_WARNINGS".WARNINGS."729868", oWARNING_DISK_SPEED_UNDER_LIMIT_LN_2 => "DB426_ALARMS_WARNINGS".WARNINGS."729869", oWARNING_STIRRER_SPEED_UNDER_LIMIT_LN_2 => "DB426_ALARMS_WARNINGS".WARNINGS."729870", oWARNING_GAS_FLOW_OVER_LIMIT_LN_2 => "DB426_ALARMS_WARNINGS".WARNINGS."729871", oWARNING_DISK_SPEED_OVER_LIMIT_LN_2 => "DB426_ALARMS_WARNINGS".WARNINGS."729872", oWARNING_STIRRER_SPEED_OVER_LIMIT_LN_2 => "DB426_ALARMS_WARNINGS".WARNINGS."729873")
   END_RUNG
   RUNG wire#powerrail
      Contact( "DB1018_POWDER_NCU_SAFE_SIGNALS".SAFE_GATES_UNIT02_FROM_NCU )
      Contact( "DB7300_INTERLOCK".GENERAL.ASPIRATION_UNIT_02_OK )
      Contact( "DB7300_INTERLOCK".POWDER_FEEDERS.UNIT_02.U02_PF2_CONDITIONS_OK )
   END_RUNG wire#w1
   // the same network as SCL:
   "DB21033_PF_2_HOPPERS_UNIT_02"(OPTIONS_0 := 2#0000_0010,   // "FB21013_POWDER_FEEDER_HOPPER"
                           iGENERAL_CONDITIONS := "DB1018_POWDER_NCU_SAFE_SIGNALS".SAFE_GATES_UNIT02_FROM_NCU AND "DB7300_INTERLOCK".GENERAL.ASPIRATION_UNIT_02_OK AND "DB7300_INTERLOCK".POWDER_FEEDERS.UNIT_02.U02_PF2_CONDITIONS_OK,
                           iPF_LINE_1_NOT_READY_FAULT := "DB21000_POWDER_FEEDER_GENERAL".POWDER_FEEDER_2_UNIT_02."FEEDER LINE 1 NOT READY FAULT",
                           iPF_PROFINET_MODE_ACTIVE_FAULT_LINE_1 := "DB21000_POWDER_FEEDER_GENERAL".POWDER_FEEDER_2_UNIT_02."FEEDER PROFINET MODE ACTIVE FAULT",
                           iPF_LINE_2_NOT_READY_FAULT := "DB21000_POWDER_FEEDER_GENERAL".POWDER_FEEDER_2_UNIT_02."FEEDER LINE 2 NOT READY FAULT",
                           iMANUAL_START_REQ_LINE_1 := "M_ZERO",
                           iMANUAL_START_REQ_LINE_2 := "DB7238_VARIABLES_PLC_CONNECTION".FEEDER_2_U_02_LINE_2.HOPPER_ON_MANUAL_REQUEST,
                           iMANUAL_STOP_REQ_LINE_2 := "DB7238_VARIABLES_PLC_CONNECTION".FEEDER_2_U_02_LINE_2.HOPPER_OFF_MANUAL_REQUEST,
                           iPF_INTERLOCK_INPUTS := "DB21002_POWDER_FEEDER_OERLIKON_INTERLOCK".POWDER_FEEDER_2_UNIT_02.Inputs,
                           iFEEDER_PROFINET_MODE_ACTIVE := "DB21000_POWDER_FEEDER_GENERAL".POWDER_FEEDER_2_UNIT_02."FEEDER PROFINET MODE ACTIVE",
                           iCONTROL_ON_DELAYED := "DB2140_HOPPERS_MPP".MACHINE_ON_DELAYED,
                           iAUTO_START_REQUEST := "DB7300_INTERLOCK".POWDER_FEEDERS.UNIT_02.SWITCH_ON_POWDER_UNIT_02,
                           iAUTO_STOP_REQUEST := "DB7300_INTERLOCK".POWDER_FEEDERS.UNIT_02.SWITCH_OFF_POWDER_UNIT_02,
                           iHMI_GAS_SETPOINT_L1 := "DB21003_POWDER_FEEDER_HMI_INTERLOCK".POWDER_FEEDER_2_UNIT_02."HMI_Values Setpoints".CarrierGasNominalLine1,
                           iHMI_GAS_SETPOINT_L2 := "DB21003_POWDER_FEEDER_HMI_INTERLOCK".POWDER_FEEDER_2_UNIT_02."HMI_Values Setpoints".CarrierGasNominalLine2,
                           iHMI_DISK_SETPOINT_L1 := "DB21003_POWDER_FEEDER_HMI_INTERLOCK".POWDER_FEEDER_2_UNIT_02."HMI_Values Setpoints".DiskSpeedNominalLine1,
                           iHMI_DISK_SETPOINT_L2 := "DB21003_POWDER_FEEDER_HMI_INTERLOCK".POWDER_FEEDER_2_UNIT_02."HMI_Values Setpoints".DiskSpeedNominalLine2,
                           iCNC_GAS_SETPOINT_L1 := "DB7300_INTERLOCK".POWDER_FEEDERS.UNIT_02.POWDER_FEEDER_2_UNIT_02.CarrierGasNominalLine1,
                           iCNC_GAS_SETPOINT_L2 := "DB7300_INTERLOCK".POWDER_FEEDERS.UNIT_02.POWDER_FEEDER_2_UNIT_02.CarrierGasNominalLine2,
                           iCNC_DISK_SETPOINT_L1 := "DB7300_INTERLOCK".POWDER_FEEDERS.UNIT_02.POWDER_FEEDER_2_UNIT_02.DiskSpeedNominalLine1,
                           iCNC_DISK_SETPOINT_L2 := "DB7300_INTERLOCK".POWDER_FEEDERS.UNIT_02.POWDER_FEEDER_2_UNIT_02.DiskSpeedNominalLine2,
                           iFEEDER_PLC_AUX_VALUES := "DB21005_POWDER_FEEDER_PLC_AUX"."INTERLOCKS_PLC_I/O_PF_2_UNIT_02",
                           oSTATION_WARNINGS => "DB441_POWDER_FEEDERS_ALARM_DECODING".ALARMS_UNIT_02.POWDER_FEEDER[2].WARNING,
                           o_fShutdownToPF_Line1 => "DB21002_POWDER_FEEDER_OERLIKON_INTERLOCK".POWDER_FEEDER_2_UNIT_02.Outputs.o_fShutdownToPF_Line1,
                           o_fShutdownToPF_Line2 => "DB21002_POWDER_FEEDER_OERLIKON_INTERLOCK".POWDER_FEEDER_2_UNIT_02.Outputs.o_fShutdownToPF_Line2,
                           o_fFeedingAllOnCmd_Line1 => "DB21002_POWDER_FEEDER_OERLIKON_INTERLOCK".POWDER_FEEDER_2_UNIT_02.Outputs.o_fFeedingAllOnCmd_Line1,
                           o_fFeedingAllOnCmd_Line2 => "DB21002_POWDER_FEEDER_OERLIKON_INTERLOCK".POWDER_FEEDER_2_UNIT_02.Outputs.o_fFeedingAllOnCmd_Line2,
                           o_fCarriergasOnCmd_Line1 => "DB21002_POWDER_FEEDER_OERLIKON_INTERLOCK".POWDER_FEEDER_2_UNIT_02.Outputs.o_fCarriergasOnCmd_Line1,
                           o_fCarriergasOnCmd_Line2 => "DB21002_POWDER_FEEDER_OERLIKON_INTERLOCK".POWDER_FEEDER_2_UNIT_02.Outputs.o_fCarriergasOnCmd_Line2,
                           o_fFeedingAllOffCmd_Line1 => "DB21002_POWDER_FEEDER_OERLIKON_INTERLOCK".POWDER_FEEDER_2_UNIT_02.Outputs.o_fFeedingAllOffCmd_Line1,
                           o_fFeedingAllOffCmd_Line2 => "DB21002_POWDER_FEEDER_OERLIKON_INTERLOCK".POWDER_FEEDER_2_UNIT_02.Outputs.o_fFeedingAllOffCmd_Line2,
                           o_fCarriergasOffCmd_Line1 => "DB21002_POWDER_FEEDER_OERLIKON_INTERLOCK".POWDER_FEEDER_2_UNIT_02.Outputs.o_fCarriergasOffCmd_Line1,
                           o_fCarriergasOffCmd_Line2 => "DB21002_POWDER_FEEDER_OERLIKON_INTERLOCK".POWDER_FEEDER_2_UNIT_02.Outputs.o_fCarriergasOffCmd_Line2,
                           oALARM_POWDER_LINE_1_CLOGGED => "DB426_ALARMS_WARNINGS".CLADDING_POWDER_FEEDER."718330",
                           oALARM_GAS_FLOW_BELOW_LOW_LIMIT_LN_1 => "DB426_ALARMS_WARNINGS".CLADDING_POWDER_FEEDER."718331",
                           oALARM_DISK_SPEED_BELOW_LOW_LIMIT_LN_1 => "DB426_ALARMS_WARNINGS".CLADDING_POWDER_FEEDER."718332",
                           oALARM_STIRRER_SPEED_BELOW_LOW_LIMIT_LN_1 => "DB426_ALARMS_WARNINGS".CLADDING_POWDER_FEEDER."718333",
                           oALARM_GAS_FLOW_ABOVE_HIGH_LIMIT_LN_1 => "DB426_ALARMS_WARNINGS".CLADDING_POWDER_FEEDER."718334",
                           oALARM_DISK_SPEED_ABOVE_HIGH_LIMIT_LN_1 => "DB426_ALARMS_WARNINGS".CLADDING_POWDER_FEEDER."718335",
                           oALARM_STIRRER_SPEED_ABOVE_HIGH_LIMIT_LN_1 => "DB426_ALARMS_WARNINGS".CLADDING_POWDER_FEEDER."718336",
                           oALARM_CARRIER_GAS_INLET_PRESSURE_TOO_LOW_LN_1 => "DB426_ALARMS_WARNINGS".CLADDING_POWDER_FEEDER."718337",
                           oALARM_DISK_MOTOR_PLUGGED_IN_AND_READY_LN_1 => "DB426_ALARMS_WARNINGS".CLADDING_POWDER_FEEDER."718338",
                           oALARM_STIRRER_PLUGGED_IN_AND_READY_LN_1 => "DB426_ALARMS_WARNINGS".CLADDING_POWDER_FEEDER."718339",
                           oALARM_COMMUNICATION_RUNNING_LN_1 => "DB426_ALARMS_WARNINGS".CLADDING_POWDER_FEEDER."718340",
                           oALARM_FEEDER_NOT_READY_LN_1 => "DB426_ALARMS_WARNINGS".CLADDING_POWDER_FEEDER."718341",
                           oWARNING_GAS_FLOW_UNDER_LIMIT_LN_1 => "DB426_ALARMS_WARNINGS".WARNINGS."729850",
                           oWARNING_DISK_SPEED_UNDER_LIMIT_LN_1 => "DB426_ALARMS_WARNINGS".WARNINGS."729851",
                           oWARNING_STIRRER_SPEED_UNDER_LIMIT_LN_1 => "DB426_ALARMS_WARNINGS".WARNINGS."729852",
                           oWARNING_GAS_FLOW_OVER_LIMIT_LN_1 => "DB426_ALARMS_WARNINGS".WARNINGS."729853",
                           oWARNING_DISK_SPEED_OVER_LIMIT_LN_1 => "DB426_ALARMS_WARNINGS".WARNINGS."729854",
                           oWARNING_STIRRER_SPEED_OVER_LIMIT_LN_1 => "DB426_ALARMS_WARNINGS".WARNINGS."729855",
                           oALARM_POWDER_LINE_2_CLOGGED => "DB426_ALARMS_WARNINGS".CLADDING_POWDER_FEEDER."718360",
                           oALARM_GAS_FLOW_BELOW_LOW_LIMIT_LN_2 => "DB426_ALARMS_WARNINGS".CLADDING_POWDER_FEEDER."718361",
                           oALARM_DISK_SPEED_BELOW_LOW_LIMIT_LN_2 => "DB426_ALARMS_WARNINGS".CLADDING_POWDER_FEEDER."718362",
                           oALARM_STIRRER_SPEED_BELOW_LOW_LIMIT_LN_2 => "DB426_ALARMS_WARNINGS".CLADDING_POWDER_FEEDER."718363",
                           oALARM_GAS_FLOW_ABOVE_HIGH_LIMIT_LN_2 => "DB426_ALARMS_WARNINGS".CLADDING_POWDER_FEEDER."718364",
                           oALARM_DISK_SPEED_ABOVE_HIGH_LIMIT_LN_2 => "DB426_ALARMS_WARNINGS".CLADDING_POWDER_FEEDER."718365",
                           oALARM_STIRRER_SPEED_ABOVE_HIGH_LIMIT_LN_2 => "DB426_ALARMS_WARNINGS".CLADDING_POWDER_FEEDER."718366",
                           oALARM_CARRIER_GAS_INLET_PRESSURE_TOO_LOW_LN_2 => "DB426_ALARMS_WARNINGS".CLADDING_POWDER_FEEDER."718367",
                           oALARM_DISK_MOTOR_PLUGGED_IN_AND_READY_LN_2 => "DB426_ALARMS_WARNINGS".CLADDING_POWDER_FEEDER."718368",
                           oALARM_STIRRER_PLUGGED_IN_AND_READY_LN_2 => "DB426_ALARMS_WARNINGS".CLADDING_POWDER_FEEDER."718369",
                           oALARM_COMMUNICATION_RUNNING_LN_2 => "DB426_ALARMS_WARNINGS".CLADDING_POWDER_FEEDER."718370",
                           oALARM_FEEDER_NOT_READY_LN_2 => "DB426_ALARMS_WARNINGS".CLADDING_POWDER_FEEDER."718371",
                           oWARNING_GAS_FLOW_UNDER_LIMIT_LN_2 => "DB426_ALARMS_WARNINGS".WARNINGS."729868",
                           oWARNING_DISK_SPEED_UNDER_LIMIT_LN_2 => "DB426_ALARMS_WARNINGS".WARNINGS."729869",
                           oWARNING_STIRRER_SPEED_UNDER_LIMIT_LN_2 => "DB426_ALARMS_WARNINGS".WARNINGS."729870",
                           oWARNING_GAS_FLOW_OVER_LIMIT_LN_2 => "DB426_ALARMS_WARNINGS".WARNINGS."729871",
                           oWARNING_DISK_SPEED_OVER_LIMIT_LN_2 => "DB426_ALARMS_WARNINGS".WARNINGS."729872",
                           oWARNING_STIRRER_SPEED_OVER_LIMIT_LN_2 => "DB426_ALARMS_WARNINGS".WARNINGS."729873");
END_REGION
END_FUNCTION

FUNCTION_BLOCK "FB21013_POWDER_FEEDER_HOPPER"   // FB21013, LAD
TITLE = FB21013 POWDER FEEDER HOPPER
{ S7_Optimized_Access := 'FALSE' }
VERSION : 0.1
// stored: AutoNumber false, IsIECCheckEnabled false, SetENOAutomatically false, UDAEnableTagReadback false
   VAR_INPUT
      OPTIONS_0 : Byte := 2#0000_0000;
      iGENERAL_CONDITIONS : Bool;   // GENERAL CONDITIONS
      iPF_LINE_1_NOT_READY_FAULT : Bool;   // PF NOT READY FAULT LINE 1
      iPF_PROFINET_MODE_ACTIVE_FAULT_LINE_1 : Bool;   // PF PROFINET MODE ACTIVE FAULT LINE 1
      iPF_LINE_2_NOT_READY_FAULT : Bool;   // PF NOT READY FAULT LINE 2
      iMANUAL_START_REQ_LINE_1 : Bool;
      iMANUAL_START_REQ_LINE_2 : Bool;
      iMANUAL_STOP_REQ_LINE_1 : Bool;
      iMANUAL_STOP_REQ_LINE_2 : Bool;
      iPF_INTERLOCK_INPUTS : "POWDER FEEDER INTERLOCK INPUT";
      iFEEDER_PROFINET_MODE_ACTIVE : Bool;
      iCONTROL_ON_DELAYED : Bool;   // LOCAL MACHINE ON
      iAUTO_START_REQUEST : Bool;
      iAUTO_STOP_REQUEST : Bool;
      iHMI_GAS_SETPOINT_L1 : Real;
      iHMI_GAS_SETPOINT_L2 : Real;
      iHMI_DISK_SETPOINT_L1 : Real;
      iHMI_DISK_SETPOINT_L2 : Real;
      iCNC_GAS_SETPOINT_L1 : Real;
      iCNC_GAS_SETPOINT_L2 : Real;
      iCNC_DISK_SETPOINT_L1 : Real;
      iCNC_DISK_SETPOINT_L2 : Real;
      iFEEDER_PLC_AUX_VALUES : "POWDER FEEDER PLC AUXILIAR";
   END_VAR
   VAR_OUTPUT
      oSTATION_IS_ALARMS : Bool;   // STATION IS ALARMS
      oSTATION_WARNINGS : Bool;   // STATION WARNINGS
      o_fShutdownToPF_Line1 { ExternalAccessible := 'False'; ExternalVisible := 'False'; ExternalWritable := 'False'} : Bool;
      o_fShutdownToPF_Line2 { ExternalAccessible := 'False'; ExternalVisible := 'False'; ExternalWritable := 'False'} : Bool;
      o_fFeedingAllOnCmd_Line1 { ExternalAccessible := 'False'; ExternalVisible := 'False'; ExternalWritable := 'False'} : Bool;
      o_fFeedingAllOnCmd_Line2 { ExternalAccessible := 'False'; ExternalVisible := 'False'; ExternalWritable := 'False'} : Bool;
      o_fCarriergasOnCmd_Line1 { ExternalAccessible := 'False'; ExternalVisible := 'False'; ExternalWritable := 'False'} : Bool;
      o_fCarriergasOnCmd_Line2 { ExternalAccessible := 'False'; ExternalVisible := 'False'; ExternalWritable := 'False'} : Bool;
      o_fFeedingAllOffCmd_Line1 { ExternalAccessible := 'False'; ExternalVisible := 'False'; ExternalWritable := 'False'} : Bool;
      o_fFeedingAllOffCmd_Line2 { ExternalAccessible := 'False'; ExternalVisible := 'False'; ExternalWritable := 'False'} : Bool;
      o_fCarriergasOffCmd_Line1 { ExternalAccessible := 'False'; ExternalVisible := 'False'; ExternalWritable := 'False'} : Bool;
      o_fCarriergasOffCmd_Line2 { ExternalAccessible := 'False'; ExternalVisible := 'False'; ExternalWritable := 'False'} : Bool;
      oALARM_POWDER_LINE_1_CLOGGED : Bool;   // ALARM POWDER LINE 1 CLOGGED
      oALARM_GAS_FLOW_BELOW_LOW_LIMIT_LN_1 : Bool;   // ALARM GAS FLOW BELOW LOW LIMIT LINE 1
      oALARM_DISK_SPEED_BELOW_LOW_LIMIT_LN_1 : Bool;   // ALARM DISK SPEED BELOW LOW LIMIT LINE 1
      oALARM_STIRRER_SPEED_BELOW_LOW_LIMIT_LN_1 : Bool;   // ALARM STIRRER SPEED BELOW LOW LIMIT LINE 1
      oALARM_GAS_FLOW_ABOVE_HIGH_LIMIT_LN_1 : Bool;   // ALARM GAS FLOW ABOVE HIGH LIMIT LINE 1
      oALARM_DISK_SPEED_ABOVE_HIGH_LIMIT_LN_1 : Bool;   // ALARM DISK SPEED ABOVE HIGH LIMIT LINE 1
      oALARM_STIRRER_SPEED_ABOVE_HIGH_LIMIT_LN_1 : Bool;   // ALARM STIRRER SPEED ABOVE HIGH LIMIT LINE 1
      oALARM_CARRIER_GAS_INLET_PRESSURE_TOO_LOW_LN_1 : Bool;   // ALARM CARRIER GAS INLET PRESSURE TOO LOW LINE 1
      oALARM_DISK_MOTOR_PLUGGED_IN_AND_READY_LN_1 : Bool;   // ALARM DISK MOTOR PLUGGED IN AND READY LINE 1
      oALARM_STIRRER_PLUGGED_IN_AND_READY_LN_1 : Bool;   // ALARM STIRRER PLUGGED IN AND READY LINE 1
      oALARM_COMMUNICATION_RUNNING_LN_1 : Bool;   // ALARM COMMUNICATION RUNNING LINE 1
      oALARM_FEEDER_NOT_READY_LN_1 : Bool;   // ALARM FEEDER NOT READY LINE 1
      oWARNING_GAS_FLOW_UNDER_LIMIT_LN_1 : Bool;   // WARNING GAS FLOW UNDER LIMIT LINE 1
      oWARNING_DISK_SPEED_UNDER_LIMIT_LN_1 : Bool;   // WARNING DISK SPEED UNDER LIMIT LINE 1
      oWARNING_STIRRER_SPEED_UNDER_LIMIT_LN_1 : Bool;   // WARNING STIRRER SPEED UNDER LIMIT LINE 1
      oWARNING_GAS_FLOW_OVER_LIMIT_LN_1 : Bool;   // WARNING GAS FLOW OVER LIMIT LINE 1
      oWARNING_DISK_SPEED_OVER_LIMIT_LN_1 : Bool;   // WARNING DISK SPEED OVER LIMIT LINE 1
      oWARNING_STIRRER_SPEED_OVER_LIMIT_LN_1 : Bool;   // WARNING STIRRER SPEED OVER LIMIT LINE 1
      oALARM_POWDER_LINE_2_CLOGGED : Bool;   // ALARM POWDER LINE 2 CLOGGED
      oALARM_GAS_FLOW_BELOW_LOW_LIMIT_LN_2 : Bool;   // ALARM GAS FLOW BELOW LOW LIMIT LINE 2
      oALARM_DISK_SPEED_BELOW_LOW_LIMIT_LN_2 : Bool;   // ALARM DISK SPEED BELOW LOW LIMIT LINE 2
      oALARM_STIRRER_SPEED_BELOW_LOW_LIMIT_LN_2 : Bool;   // ALARM STIRRER SPEED BELOW LOW LIMIT LINE 2
      oALARM_GAS_FLOW_ABOVE_HIGH_LIMIT_LN_2 : Bool;   // ALARM GAS FLOW ABOVE HIGH LIMIT LINE 2
      oALARM_DISK_SPEED_ABOVE_HIGH_LIMIT_LN_2 : Bool;   // ALARM DISK SPEED ABOVE HIGH LIMIT LINE 2
      oALARM_STIRRER_SPEED_ABOVE_HIGH_LIMIT_LN_2 : Bool;   // ALARM STIRRER SPEED ABOVE HIGH LIMIT LINE 2
      oALARM_CARRIER_GAS_INLET_PRESSURE_TOO_LOW_LN_2 : Bool;   // ALARM CARRIER GAS INLET PRESSURE TOO LOW LINE 2
      oALARM_DISK_MOTOR_PLUGGED_IN_AND_READY_LN_2 : Bool;   // ALARM DISK MOTOR PLUGGED IN AND READY LINE 2
      oALARM_STIRRER_PLUGGED_IN_AND_READY_LN_2 : Bool;   // ALARM STIRRER PLUGGED IN AND READY LINE 2
      oALARM_COMMUNICATION_RUNNING_LN_2 : Bool;   // ALARM COMMUNICATION RUNNING LINE 2
      oALARM_FEEDER_NOT_READY_LN_2 : Bool;   // ALARM FEEDER NOT READY LINE 2
      oWARNING_GAS_FLOW_UNDER_LIMIT_LN_2 : Bool;   // WARNING GAS FLOW UNDER LIMIT LINE 2
      oWARNING_DISK_SPEED_UNDER_LIMIT_LN_2 : Bool;   // WARNING DISK SPEED UNDER LIMIT LINE 2
      oWARNING_STIRRER_SPEED_UNDER_LIMIT_LN_2 : Bool;   // WARNING STIRRER SPEED UNDER LIMIT LINE 2
      oWARNING_GAS_FLOW_OVER_LIMIT_LN_2 : Bool;   // WARNING GAS FLOW OVER LIMIT LINE 2
      oWARNING_DISK_SPEED_OVER_LIMIT_LN_2 : Bool;   // WARNING DISK SPEED OVER LIMIT LINE 2
      oWARNING_STIRRER_SPEED_OVER_LIMIT_LN_2 : Bool;   // WARNING STIRRER SPEED OVER LIMIT LINE 2
   END_VAR
   VAR DB_SPECIFIC
      DATA : "POWDER FEEDER HOPPER";
      INPUT_SETTINGS : Struct
         UNIT_NUMBER : Int;
         FEEDER_NUMBER : Int;
      END_STRUCT;
      Fault_timer { S7_SetPoint := 'True'} : TON_TIME;
      START_DONE_LINE_1 { S7_SetPoint := 'True'} : Bool;   // START DONE LINE 1
      START_DONE_LINE_2 { S7_SetPoint := 'True'} : Bool;   // START DONE LINE 2
      STOP_SEQUENCE_ON { S7_SetPoint := 'True'} : Bool;   // HOPPER STOP SEQUENCE IS ON
      STOP_PULSE_LINE_1 : Bool;
      STOP_PULSE_LINE_2 : Bool;
      HOPPER_STATUS_LINE_1 : Byte;   // HOPPER LINE 1 STATUS
      HOPPER_STATUS_LINE_2 : Byte;   // HOPPER LINE 2 STATUS
   END_VAR
   VAR
      SWITCH_ON_SEQUENCE_LINE_1 : "FB21250_POWDER_ON_OFF_SEQUENCE";
      SWITCH_ON_SEQUENCE_LINE_2 : "FB21250_POWDER_ON_OFF_SEQUENCE";
      SWITCH_OFF_SEQUENCE_LINE_1 : "FB21250_POWDER_ON_OFF_SEQUENCE";
      SWITCH_OFF_SEQUENCE_LINE_2 : "FB21250_POWDER_ON_OFF_SEQUENCE";
   END_VAR
   VAR DB_SPECIFIC
      SWITCH_OFF_DELAY_LINE_1 { S7_SetPoint := 'True'} : TOF_TIME;
      SWITCH_OFF_DELAY_LINE_2 { S7_SetPoint := 'True'} : TOF_TIME;
   END_VAR
   VAR_TEMP
      DB_NUMBER : DInt;
      INPUTS_MASK : Byte;
      O_BYTE_0 : Struct
         LINE_1_ENABLED : Bool;
         LINE_2_ENABLED : Bool;
         SPARE : Bool;
         SPARE_1 : Bool;
         SPARE_2 : Bool;
         SPARE_3 : Bool;
         SPARE_4 : Bool;
         SPARE_5 : Bool;
      END_STRUCT;
   END_VAR
   // Fault_timer.PT := T#1s;
   // SWITCH_OFF_DELAY_LINE_1.PT := T#4s;
   // SWITCH_OFF_DELAY_LINE_2.PT := T#4s;
   VAR_TEMP   // added for the SCL form of the ladder/FBD networks
      _w1 : Bool;
      _w2 : Bool;
   END_VAR
BEGIN

NETWORK
TITLE = READ INSTANCE DB NUMBER
      L     DINO;
      +     10#800000;
      T     #DB_NUMBER;

REGION Network 2: OPTIONS
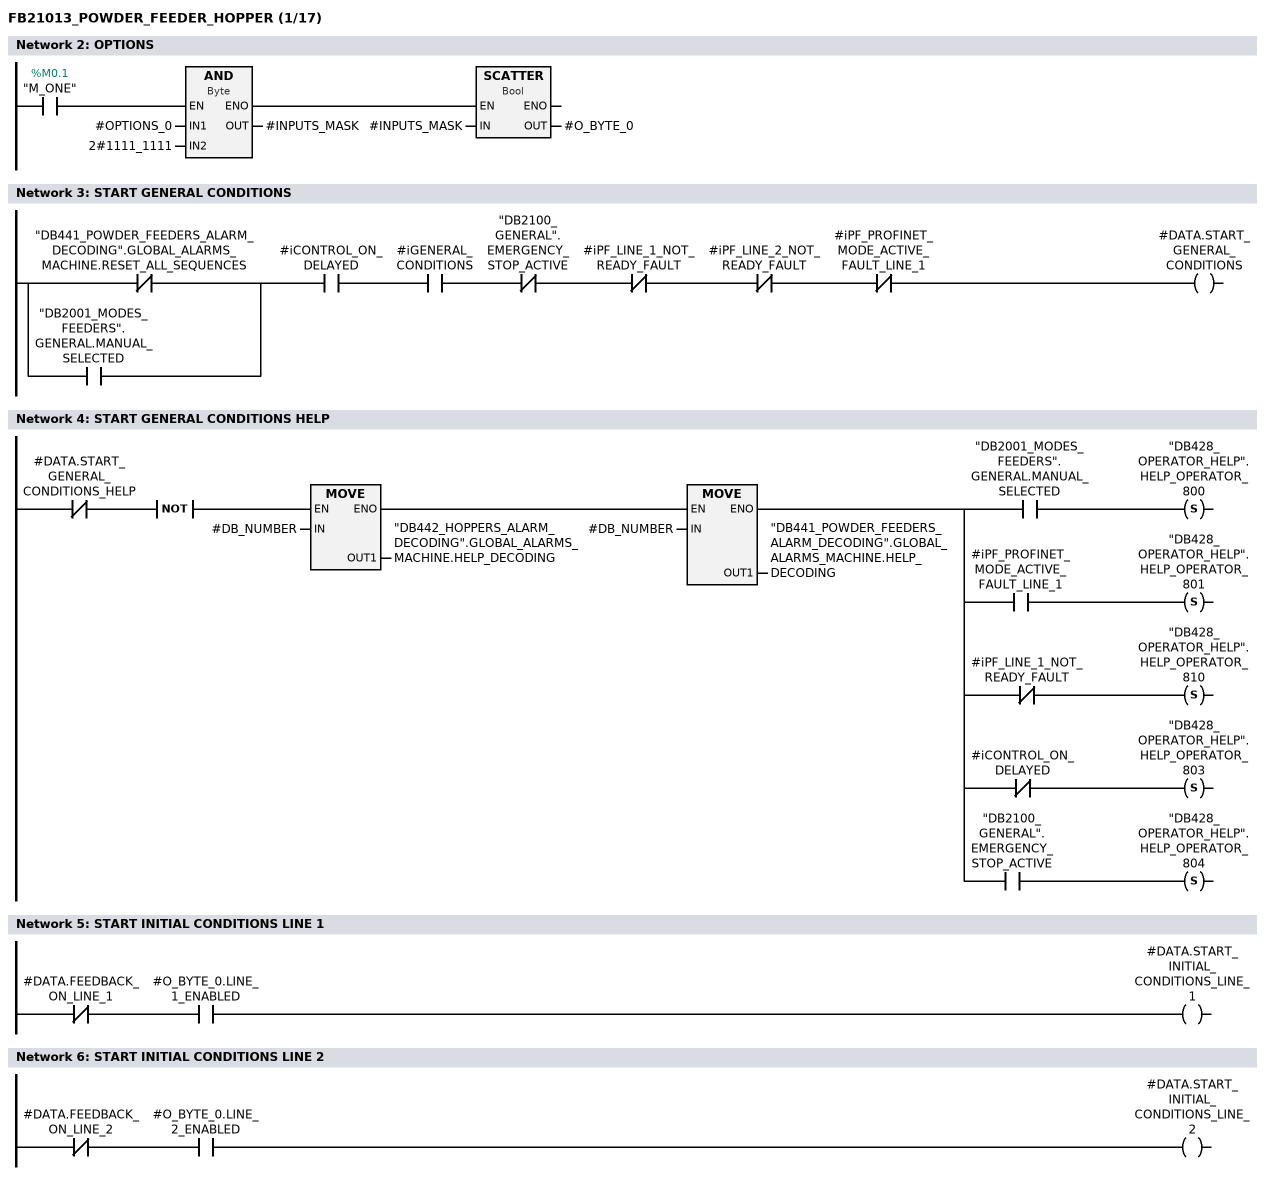
   RUNG wire#powerrail
      Contact( "M_ONE" )
      { S7_Templates := "SrcType := Byte" } And(in1 := #OPTIONS_0, in2 := 2#1111_1111, out => #INPUTS_MASK)
      { S7_Templates := "[dest_type := Bool, src_type := Byte]" } SCATTER(IN := #INPUTS_MASK, OUT => #O_BYTE_0)
   END_RUNG
   // the same network as SCL:
   IF "M_ONE" THEN
       #INPUTS_MASK := #OPTIONS_0 AND 2#1111_1111;
       SCATTER(IN := #INPUTS_MASK, OUT => #O_BYTE_0);
   END_IF;
END_REGION

REGION Network 3: START GENERAL CONDITIONS
   RUNG wire#powerrail
      I_Contact( "DB441_POWDER_FEEDERS_ALARM_DECODING".GLOBAL_ALARMS_MACHINE.RESET_ALL_SEQUENCES )
      wire#w1
      Contact( #iCONTROL_ON_DELAYED )
      Contact( #iGENERAL_CONDITIONS )
      I_Contact( "DB2100_GENERAL".EMERGENCY_STOP_ACTIVE )
      I_Contact( #iPF_LINE_1_NOT_READY_FAULT )
      I_Contact( #iPF_LINE_2_NOT_READY_FAULT )
      I_Contact( #iPF_PROFINET_MODE_ACTIVE_FAULT_LINE_1 )
      Coil( #DATA.START_GENERAL_CONDITIONS )
   END_RUNG
   RUNG wire#powerrail
      Contact( "DB2001_MODES_FEEDERS".GENERAL.MANUAL_SELECTED )
   END_RUNG wire#w1
   // the same network as SCL:
   #DATA.START_GENERAL_CONDITIONS := (NOT "DB441_POWDER_FEEDERS_ALARM_DECODING".GLOBAL_ALARMS_MACHINE.RESET_ALL_SEQUENCES OR "DB2001_MODES_FEEDERS".GENERAL.MANUAL_SELECTED) AND #iCONTROL_ON_DELAYED AND #iGENERAL_CONDITIONS AND NOT "DB2100_GENERAL".EMERGENCY_STOP_ACTIVE AND NOT #iPF_LINE_1_NOT_READY_FAULT AND NOT #iPF_LINE_2_NOT_READY_FAULT AND NOT #iPF_PROFINET_MODE_ACTIVE_FAULT_LINE_1;
END_REGION

REGION Network 4: START GENERAL CONDITIONS HELP
   RUNG wire#powerrail
      I_Contact( #DATA.START_GENERAL_CONDITIONS_HELP )
      Not()
      Move(in := #DB_NUMBER, out1 => "DB442_HOPPERS_ALARM_DECODING".GLOBAL_ALARMS_MACHINE.HELP_DECODING)
      Move(in := #DB_NUMBER, out1 => "DB441_POWDER_FEEDERS_ALARM_DECODING".GLOBAL_ALARMS_MACHINE.HELP_DECODING)
      wire#w1
      Contact( "DB2001_MODES_FEEDERS".GENERAL.MANUAL_SELECTED )
      S_Coil( "DB428_OPERATOR_HELP".HELP_OPERATOR_800 )
   END_RUNG
   RUNG wire#w1
      Contact( #iPF_PROFINET_MODE_ACTIVE_FAULT_LINE_1 )
      S_Coil( "DB428_OPERATOR_HELP".HELP_OPERATOR_801 )
   END_RUNG
   RUNG wire#w1
      I_Contact( #iPF_LINE_1_NOT_READY_FAULT )
      S_Coil( "DB428_OPERATOR_HELP".HELP_OPERATOR_810 )
   END_RUNG
   RUNG wire#w1
      I_Contact( #iCONTROL_ON_DELAYED )
      S_Coil( "DB428_OPERATOR_HELP".HELP_OPERATOR_803 )
   END_RUNG
   RUNG wire#w1
      Contact( "DB2100_GENERAL".EMERGENCY_STOP_ACTIVE )
      S_Coil( "DB428_OPERATOR_HELP".HELP_OPERATOR_804 )
   END_RUNG
   // the same network as SCL:
   #_w1 := NOT (NOT #DATA.START_GENERAL_CONDITIONS_HELP);
   IF #_w1 THEN
       "DB442_HOPPERS_ALARM_DECODING".GLOBAL_ALARMS_MACHINE.HELP_DECODING := #DB_NUMBER;
       "DB441_POWDER_FEEDERS_ALARM_DECODING".GLOBAL_ALARMS_MACHINE.HELP_DECODING := #DB_NUMBER;
   END_IF;
   IF #_w1 AND "DB2001_MODES_FEEDERS".GENERAL.MANUAL_SELECTED THEN
       "DB428_OPERATOR_HELP".HELP_OPERATOR_800 := TRUE;
   END_IF;
   IF #_w1 AND #iPF_PROFINET_MODE_ACTIVE_FAULT_LINE_1 THEN
       "DB428_OPERATOR_HELP".HELP_OPERATOR_801 := TRUE;
   END_IF;
   IF #_w1 AND NOT #iPF_LINE_1_NOT_READY_FAULT THEN "DB428_OPERATOR_HELP".HELP_OPERATOR_810 := TRUE; END_IF;
   IF #_w1 AND NOT #iCONTROL_ON_DELAYED THEN "DB428_OPERATOR_HELP".HELP_OPERATOR_803 := TRUE; END_IF;
   IF #_w1 AND "DB2100_GENERAL".EMERGENCY_STOP_ACTIVE THEN
       "DB428_OPERATOR_HELP".HELP_OPERATOR_804 := TRUE;
   END_IF;
END_REGION

REGION Network 5: START INITIAL CONDITIONS LINE 1
   RUNG wire#powerrail
      I_Contact( #DATA.FEEDBACK_ON_LINE_1 )
      Contact( #O_BYTE_0.LINE_1_ENABLED )
      Coil( #DATA.START_INITIAL_CONDITIONS_LINE_1 )
   END_RUNG
   // the same network as SCL:
   #DATA.START_INITIAL_CONDITIONS_LINE_1 := NOT #DATA.FEEDBACK_ON_LINE_1 AND #O_BYTE_0.LINE_1_ENABLED;
END_REGION

REGION Network 6: START INITIAL CONDITIONS LINE 2
   RUNG wire#powerrail
      I_Contact( #DATA.FEEDBACK_ON_LINE_2 )
      Contact( #O_BYTE_0.LINE_2_ENABLED )
      Coil( #DATA.START_INITIAL_CONDITIONS_LINE_2 )
   END_RUNG
   // the same network as SCL:
   #DATA.START_INITIAL_CONDITIONS_LINE_2 := NOT #DATA.FEEDBACK_ON_LINE_2 AND #O_BYTE_0.LINE_2_ENABLED;
END_REGION

REGION Network 7: START INITIAL CONDITIONS HELP
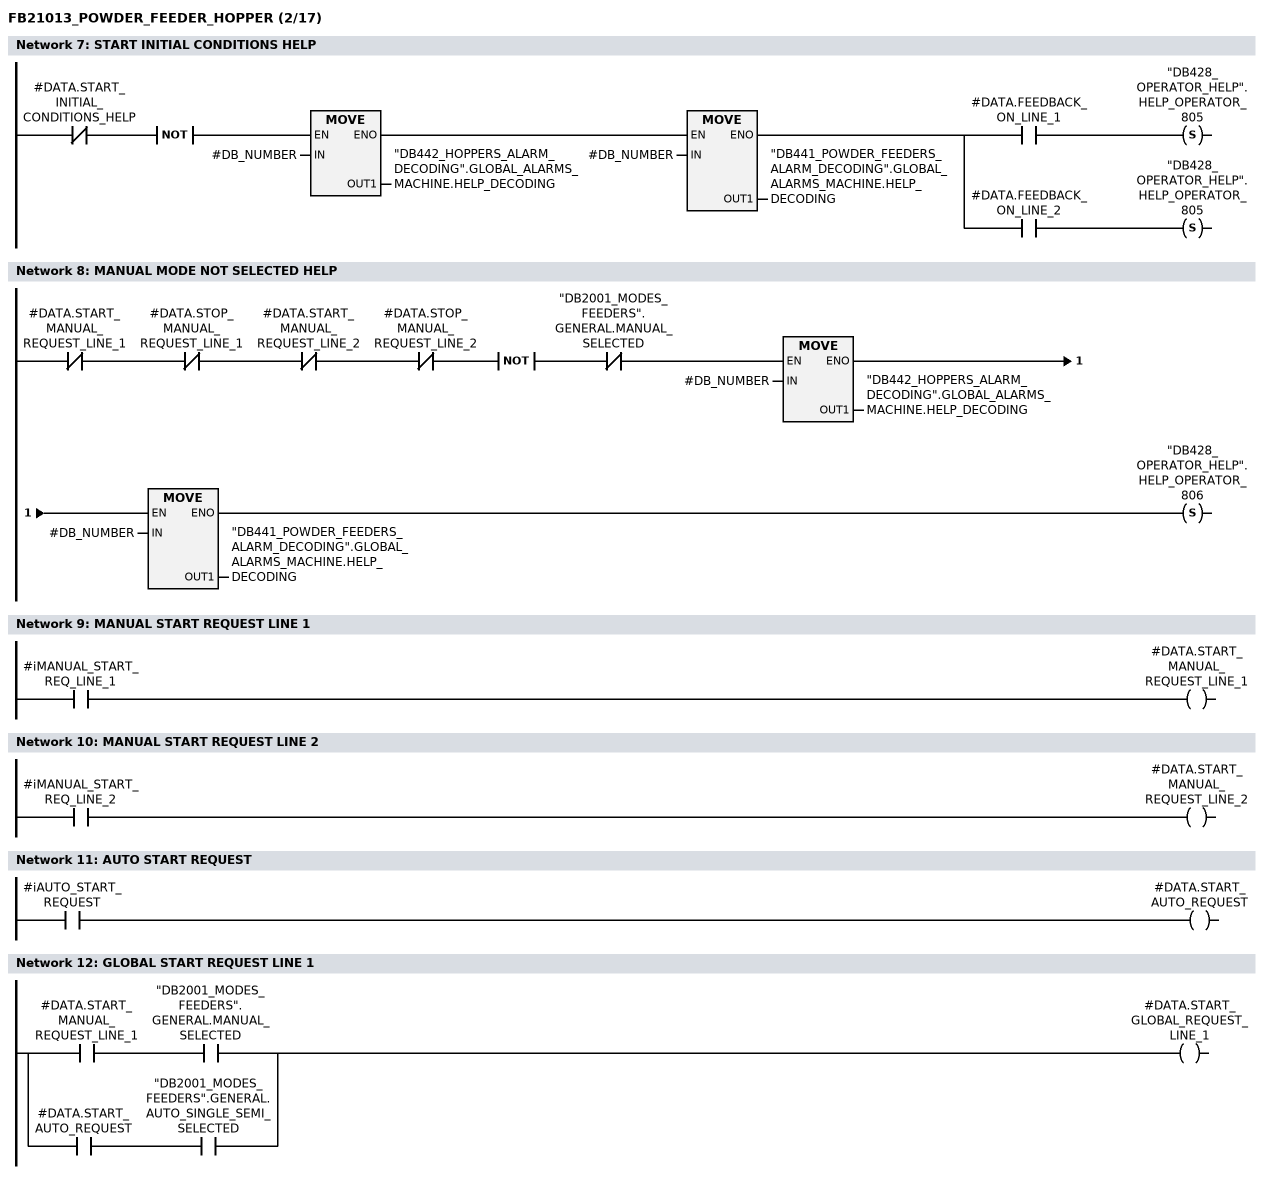
   RUNG wire#powerrail
      I_Contact( #DATA.START_INITIAL_CONDITIONS_HELP )
      Not()
      Move(in := #DB_NUMBER, out1 => "DB442_HOPPERS_ALARM_DECODING".GLOBAL_ALARMS_MACHINE.HELP_DECODING)
      Move(in := #DB_NUMBER, out1 => "DB441_POWDER_FEEDERS_ALARM_DECODING".GLOBAL_ALARMS_MACHINE.HELP_DECODING)
      wire#w1
      Contact( #DATA.FEEDBACK_ON_LINE_1 )
      S_Coil( "DB428_OPERATOR_HELP".HELP_OPERATOR_805 )
   END_RUNG
   RUNG wire#w1
      Contact( #DATA.FEEDBACK_ON_LINE_2 )
      S_Coil( "DB428_OPERATOR_HELP".HELP_OPERATOR_805 )
   END_RUNG
   // the same network as SCL:
   #_w1 := NOT (NOT #DATA.START_INITIAL_CONDITIONS_HELP);
   IF #_w1 THEN
       "DB442_HOPPERS_ALARM_DECODING".GLOBAL_ALARMS_MACHINE.HELP_DECODING := #DB_NUMBER;
       "DB441_POWDER_FEEDERS_ALARM_DECODING".GLOBAL_ALARMS_MACHINE.HELP_DECODING := #DB_NUMBER;
   END_IF;
   IF #_w1 AND #DATA.FEEDBACK_ON_LINE_1 THEN "DB428_OPERATOR_HELP".HELP_OPERATOR_805 := TRUE; END_IF;
   IF #_w1 AND #DATA.FEEDBACK_ON_LINE_2 THEN "DB428_OPERATOR_HELP".HELP_OPERATOR_805 := TRUE; END_IF;
END_REGION

REGION Network 8: MANUAL MODE NOT SELECTED HELP
   RUNG wire#powerrail
      I_Contact( #DATA.START_MANUAL_REQUEST_LINE_1 )
      I_Contact( #DATA.STOP_MANUAL_REQUEST_LINE_1 )
      I_Contact( #DATA.START_MANUAL_REQUEST_LINE_2 )
      I_Contact( #DATA.STOP_MANUAL_REQUEST_LINE_2 )
      Not()
      I_Contact( "DB2001_MODES_FEEDERS".GENERAL.MANUAL_SELECTED )
      Move(in := #DB_NUMBER, out1 => "DB442_HOPPERS_ALARM_DECODING".GLOBAL_ALARMS_MACHINE.HELP_DECODING)
      Move(in := #DB_NUMBER, out1 => "DB441_POWDER_FEEDERS_ALARM_DECODING".GLOBAL_ALARMS_MACHINE.HELP_DECODING)
      S_Coil( "DB428_OPERATOR_HELP".HELP_OPERATOR_806 )
   END_RUNG
   // the same network as SCL:
   IF NOT (NOT #DATA.START_MANUAL_REQUEST_LINE_1 AND NOT #DATA.STOP_MANUAL_REQUEST_LINE_1 AND NOT #DATA.START_MANUAL_REQUEST_LINE_2 AND NOT #DATA.STOP_MANUAL_REQUEST_LINE_2) AND NOT "DB2001_MODES_FEEDERS".GENERAL.MANUAL_SELECTED THEN
       "DB442_HOPPERS_ALARM_DECODING".GLOBAL_ALARMS_MACHINE.HELP_DECODING := #DB_NUMBER;
       "DB441_POWDER_FEEDERS_ALARM_DECODING".GLOBAL_ALARMS_MACHINE.HELP_DECODING := #DB_NUMBER;
       "DB428_OPERATOR_HELP".HELP_OPERATOR_806 := TRUE;
   END_IF;
END_REGION

REGION Network 9: MANUAL START REQUEST LINE 1
   RUNG wire#powerrail
      Contact( #iMANUAL_START_REQ_LINE_1 )
      Coil( #DATA.START_MANUAL_REQUEST_LINE_1 )
   END_RUNG
   // the same network as SCL:
   #DATA.START_MANUAL_REQUEST_LINE_1 := #iMANUAL_START_REQ_LINE_1;
END_REGION

REGION Network 10: MANUAL START REQUEST LINE 2
   RUNG wire#powerrail
      Contact( #iMANUAL_START_REQ_LINE_2 )
      Coil( #DATA.START_MANUAL_REQUEST_LINE_2 )
   END_RUNG
   // the same network as SCL:
   #DATA.START_MANUAL_REQUEST_LINE_2 := #iMANUAL_START_REQ_LINE_2;
END_REGION

REGION Network 11: AUTO START REQUEST
   RUNG wire#powerrail
      Contact( #iAUTO_START_REQUEST )
      Coil( #DATA.START_AUTO_REQUEST )
   END_RUNG
   // the same network as SCL:
   #DATA.START_AUTO_REQUEST := #iAUTO_START_REQUEST;
END_REGION

REGION Network 12: GLOBAL START REQUEST LINE 1
   RUNG wire#powerrail
      Contact( #DATA.START_MANUAL_REQUEST_LINE_1 )
      Contact( "DB2001_MODES_FEEDERS".GENERAL.MANUAL_SELECTED )
      wire#w1
      Coil( #DATA.START_GLOBAL_REQUEST_LINE_1 )
   END_RUNG
   RUNG wire#powerrail
      Contact( #DATA.START_AUTO_REQUEST )
      Contact( "DB2001_MODES_FEEDERS".GENERAL.AUTO_SINGLE_SEMI_SELECTED )
   END_RUNG wire#w1
   // the same network as SCL:
   #DATA.START_GLOBAL_REQUEST_LINE_1 := (#DATA.START_MANUAL_REQUEST_LINE_1 AND "DB2001_MODES_FEEDERS".GENERAL.MANUAL_SELECTED) OR (#DATA.START_AUTO_REQUEST AND "DB2001_MODES_FEEDERS".GENERAL.AUTO_SINGLE_SEMI_SELECTED);
END_REGION

REGION Network 13: GLOBAL START REQUEST LINE 2
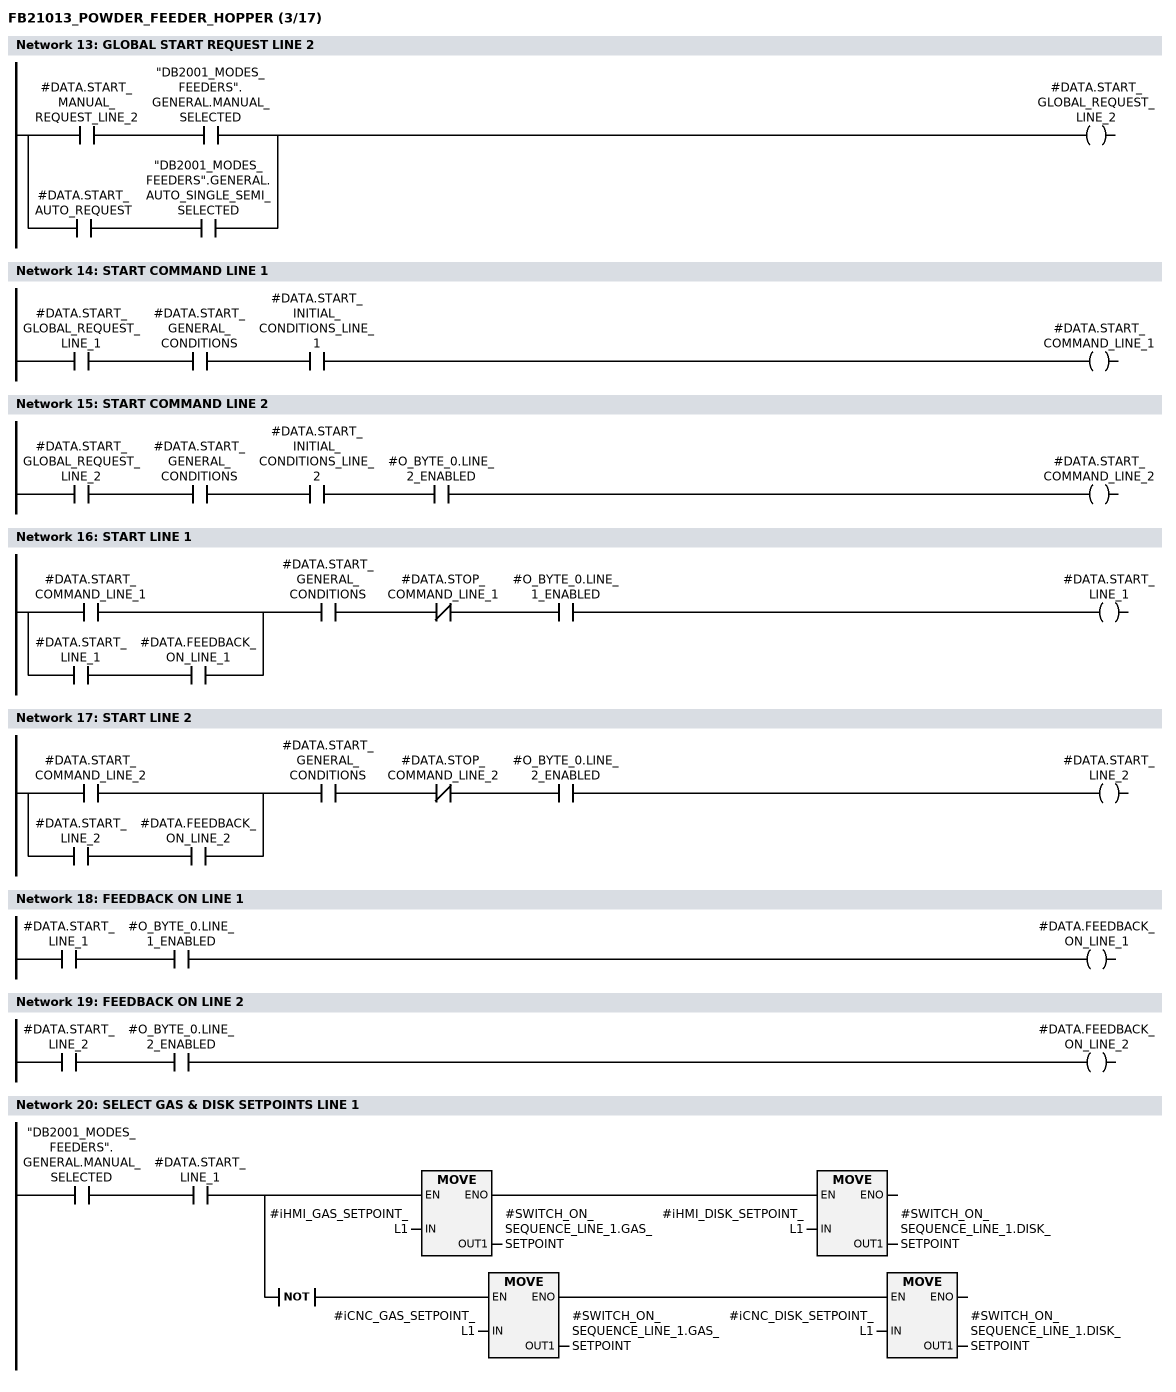
   RUNG wire#powerrail
      Contact( #DATA.START_MANUAL_REQUEST_LINE_2 )
      Contact( "DB2001_MODES_FEEDERS".GENERAL.MANUAL_SELECTED )
      wire#w1
      Coil( #DATA.START_GLOBAL_REQUEST_LINE_2 )
   END_RUNG
   RUNG wire#powerrail
      Contact( #DATA.START_AUTO_REQUEST )
      Contact( "DB2001_MODES_FEEDERS".GENERAL.AUTO_SINGLE_SEMI_SELECTED )
   END_RUNG wire#w1
   // the same network as SCL:
   #DATA.START_GLOBAL_REQUEST_LINE_2 := (#DATA.START_MANUAL_REQUEST_LINE_2 AND "DB2001_MODES_FEEDERS".GENERAL.MANUAL_SELECTED) OR (#DATA.START_AUTO_REQUEST AND "DB2001_MODES_FEEDERS".GENERAL.AUTO_SINGLE_SEMI_SELECTED);
END_REGION

REGION Network 14: START COMMAND LINE 1
   RUNG wire#powerrail
      Contact( #DATA.START_GLOBAL_REQUEST_LINE_1 )
      Contact( #DATA.START_GENERAL_CONDITIONS )
      Contact( #DATA.START_INITIAL_CONDITIONS_LINE_1 )
      Coil( #DATA.START_COMMAND_LINE_1 )
   END_RUNG
   // the same network as SCL:
   #DATA.START_COMMAND_LINE_1 := #DATA.START_GLOBAL_REQUEST_LINE_1 AND #DATA.START_GENERAL_CONDITIONS AND #DATA.START_INITIAL_CONDITIONS_LINE_1;
END_REGION

REGION Network 15: START COMMAND LINE 2
   RUNG wire#powerrail
      Contact( #DATA.START_GLOBAL_REQUEST_LINE_2 )
      Contact( #DATA.START_GENERAL_CONDITIONS )
      Contact( #DATA.START_INITIAL_CONDITIONS_LINE_2 )
      Contact( #O_BYTE_0.LINE_2_ENABLED )
      Coil( #DATA.START_COMMAND_LINE_2 )
   END_RUNG
   // the same network as SCL:
   #DATA.START_COMMAND_LINE_2 := #DATA.START_GLOBAL_REQUEST_LINE_2 AND #DATA.START_GENERAL_CONDITIONS AND #DATA.START_INITIAL_CONDITIONS_LINE_2 AND #O_BYTE_0.LINE_2_ENABLED;
END_REGION

REGION Network 16: START LINE 1
   RUNG wire#powerrail
      Contact( #DATA.START_COMMAND_LINE_1 )
      wire#w1
      Contact( #DATA.START_GENERAL_CONDITIONS )
      I_Contact( #DATA.STOP_COMMAND_LINE_1 )
      Contact( #O_BYTE_0.LINE_1_ENABLED )
      Coil( #DATA.START_LINE_1 )
   END_RUNG
   RUNG wire#powerrail
      Contact( #DATA.START_LINE_1 )
      Contact( #DATA.FEEDBACK_ON_LINE_1 )
   END_RUNG wire#w1
   // the same network as SCL:
   #DATA.START_LINE_1 := (#DATA.START_COMMAND_LINE_1 OR (#DATA.START_LINE_1 AND #DATA.FEEDBACK_ON_LINE_1)) AND #DATA.START_GENERAL_CONDITIONS AND NOT #DATA.STOP_COMMAND_LINE_1 AND #O_BYTE_0.LINE_1_ENABLED;
END_REGION

REGION Network 17: START LINE 2
   RUNG wire#powerrail
      Contact( #DATA.START_COMMAND_LINE_2 )
      wire#w1
      Contact( #DATA.START_GENERAL_CONDITIONS )
      I_Contact( #DATA.STOP_COMMAND_LINE_2 )
      Contact( #O_BYTE_0.LINE_2_ENABLED )
      Coil( #DATA.START_LINE_2 )
   END_RUNG
   RUNG wire#powerrail
      Contact( #DATA.START_LINE_2 )
      Contact( #DATA.FEEDBACK_ON_LINE_2 )
   END_RUNG wire#w1
   // the same network as SCL:
   #DATA.START_LINE_2 := (#DATA.START_COMMAND_LINE_2 OR (#DATA.START_LINE_2 AND #DATA.FEEDBACK_ON_LINE_2)) AND #DATA.START_GENERAL_CONDITIONS AND NOT #DATA.STOP_COMMAND_LINE_2 AND #O_BYTE_0.LINE_2_ENABLED;
END_REGION

REGION Network 18: FEEDBACK ON LINE 1
   RUNG wire#powerrail
      Contact( #DATA.START_LINE_1 )
      Contact( #O_BYTE_0.LINE_1_ENABLED )
      Coil( #DATA.FEEDBACK_ON_LINE_1 )
   END_RUNG
   // the same network as SCL:
   #DATA.FEEDBACK_ON_LINE_1 := #DATA.START_LINE_1 AND #O_BYTE_0.LINE_1_ENABLED;
END_REGION

REGION Network 19: FEEDBACK ON LINE 2
   RUNG wire#powerrail
      Contact( #DATA.START_LINE_2 )
      Contact( #O_BYTE_0.LINE_2_ENABLED )
      Coil( #DATA.FEEDBACK_ON_LINE_2 )
   END_RUNG
   // the same network as SCL:
   #DATA.FEEDBACK_ON_LINE_2 := #DATA.START_LINE_2 AND #O_BYTE_0.LINE_2_ENABLED;
END_REGION

REGION Network 20: SELECT GAS & DISK SETPOINTS LINE 1
   RUNG wire#powerrail
      Contact( "DB2001_MODES_FEEDERS".GENERAL.MANUAL_SELECTED )
      Contact( #DATA.START_LINE_1 )
      wire#w1
      Move(in := #iHMI_GAS_SETPOINT_L1, out1 => #SWITCH_ON_SEQUENCE_LINE_1.GAS_SETPOINT)
      Move(in := #iHMI_DISK_SETPOINT_L1, out1 => #SWITCH_ON_SEQUENCE_LINE_1.DISK_SETPOINT)
   END_RUNG
   RUNG wire#w1
      Not()
      Move(in := #iCNC_GAS_SETPOINT_L1, out1 => #SWITCH_ON_SEQUENCE_LINE_1.GAS_SETPOINT)
      Move(in := #iCNC_DISK_SETPOINT_L1, out1 => #SWITCH_ON_SEQUENCE_LINE_1.DISK_SETPOINT)
   END_RUNG
   // the same network as SCL:
   #_w1 := "DB2001_MODES_FEEDERS".GENERAL.MANUAL_SELECTED AND #DATA.START_LINE_1;
   IF #_w1 THEN
       #SWITCH_ON_SEQUENCE_LINE_1.GAS_SETPOINT := #iHMI_GAS_SETPOINT_L1;
       #SWITCH_ON_SEQUENCE_LINE_1.DISK_SETPOINT := #iHMI_DISK_SETPOINT_L1;
   END_IF;
   IF NOT #_w1 THEN
       #SWITCH_ON_SEQUENCE_LINE_1.GAS_SETPOINT := #iCNC_GAS_SETPOINT_L1;
       #SWITCH_ON_SEQUENCE_LINE_1.DISK_SETPOINT := #iCNC_DISK_SETPOINT_L1;
   END_IF;
END_REGION

REGION Network 21: SELECT GAS & DISK SETPOINTS LINE 2
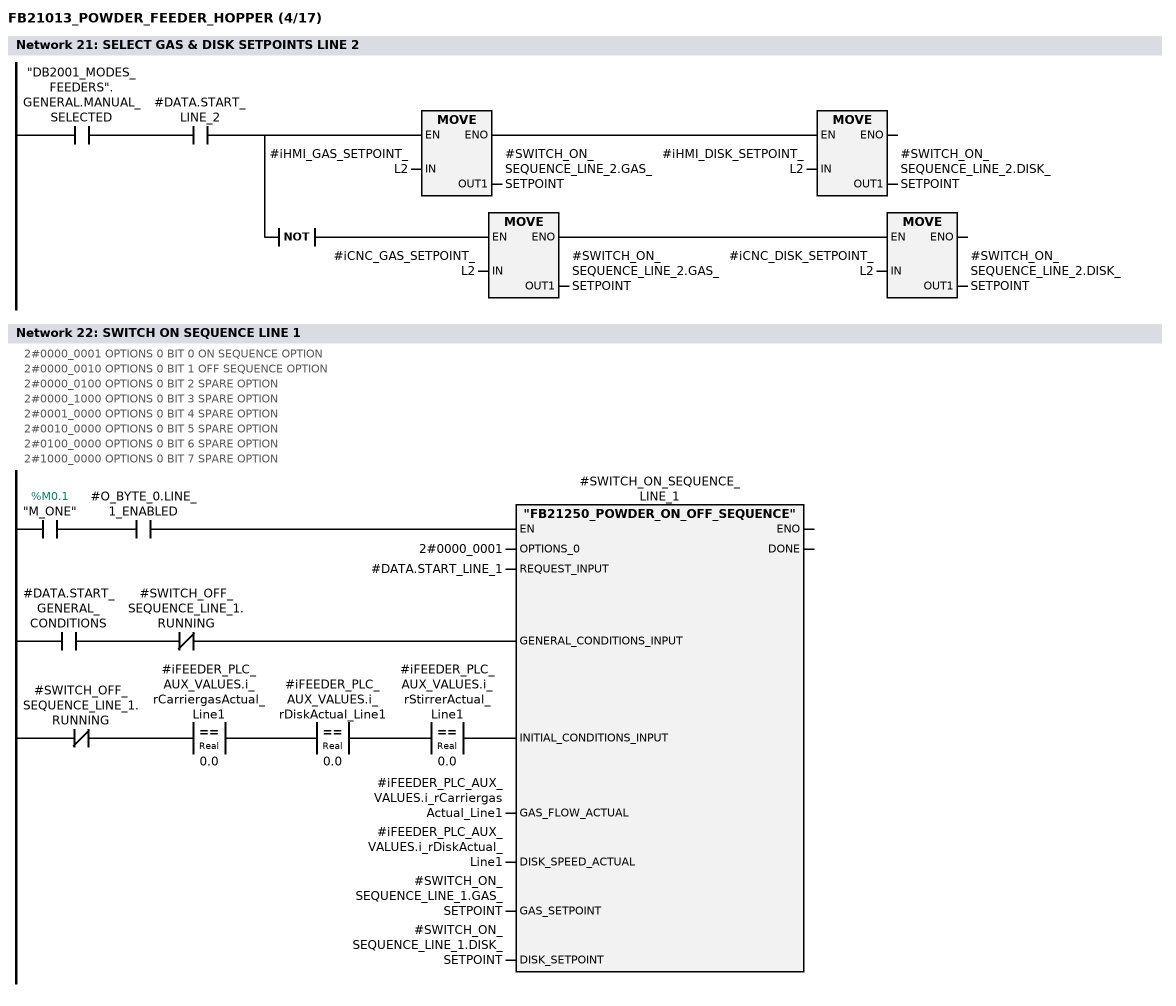
   RUNG wire#powerrail
      Contact( "DB2001_MODES_FEEDERS".GENERAL.MANUAL_SELECTED )
      Contact( #DATA.START_LINE_2 )
      wire#w1
      Move(in := #iHMI_GAS_SETPOINT_L2, out1 => #SWITCH_ON_SEQUENCE_LINE_2.GAS_SETPOINT)
      Move(in := #iHMI_DISK_SETPOINT_L2, out1 => #SWITCH_ON_SEQUENCE_LINE_2.DISK_SETPOINT)
   END_RUNG
   RUNG wire#w1
      Not()
      Move(in := #iCNC_GAS_SETPOINT_L2, out1 => #SWITCH_ON_SEQUENCE_LINE_2.GAS_SETPOINT)
      Move(in := #iCNC_DISK_SETPOINT_L2, out1 => #SWITCH_ON_SEQUENCE_LINE_2.DISK_SETPOINT)
   END_RUNG
   // the same network as SCL:
   #_w1 := "DB2001_MODES_FEEDERS".GENERAL.MANUAL_SELECTED AND #DATA.START_LINE_2;
   IF #_w1 THEN
       #SWITCH_ON_SEQUENCE_LINE_2.GAS_SETPOINT := #iHMI_GAS_SETPOINT_L2;
       #SWITCH_ON_SEQUENCE_LINE_2.DISK_SETPOINT := #iHMI_DISK_SETPOINT_L2;
   END_IF;
   IF NOT #_w1 THEN
       #SWITCH_ON_SEQUENCE_LINE_2.GAS_SETPOINT := #iCNC_GAS_SETPOINT_L2;
       #SWITCH_ON_SEQUENCE_LINE_2.DISK_SETPOINT := #iCNC_DISK_SETPOINT_L2;
   END_IF;
END_REGION

REGION Network 22: SWITCH ON SEQUENCE LINE 1
   // 2#0000_0001 OPTIONS 0 BIT 0 ON SEQUENCE OPTION
   // 2#0000_0010 OPTIONS 0 BIT 1 OFF SEQUENCE OPTION
   // 2#0000_0100 OPTIONS 0 BIT 2 SPARE OPTION
   // 2#0000_1000 OPTIONS 0 BIT 3 SPARE OPTION
   // 2#0001_0000 OPTIONS 0 BIT 4 SPARE OPTION
   // 2#0010_0000 OPTIONS 0 BIT 5 SPARE OPTION
   // 2#0100_0000 OPTIONS 0 BIT 6 SPARE OPTION
   // 2#1000_0000 OPTIONS 0 BIT 7 SPARE OPTION
   RUNG wire#powerrail
      Contact( "M_ONE" )
      Contact( #O_BYTE_0.LINE_1_ENABLED )
      #SWITCH_ON_SEQUENCE_LINE_1(GENERAL_CONDITIONS_INPUT := wire#w1, INITIAL_CONDITIONS_INPUT := wire#w2, OPTIONS_0 := 2#0000_0001, REQUEST_INPUT := #DATA.START_LINE_1, GAS_FLOW_ACTUAL := #iFEEDER_PLC_AUX_VALUES.i_rCarriergasActual_Line1, DISK_SPEED_ACTUAL := #iFEEDER_PLC_AUX_VALUES.i_rDiskActual_Line1, GAS_SETPOINT := #SWITCH_ON_SEQUENCE_LINE_1.GAS_SETPOINT, DISK_SETPOINT := #SWITCH_ON_SEQUENCE_LINE_1.DISK_SETPOINT, DONE =>)
   END_RUNG
   RUNG wire#powerrail
      Contact( #DATA.START_GENERAL_CONDITIONS )
      I_Contact( #SWITCH_OFF_SEQUENCE_LINE_1.RUNNING )
   END_RUNG wire#w1
   RUNG wire#powerrail
      I_Contact( #SWITCH_OFF_SEQUENCE_LINE_1.RUNNING )
      { S7_Templates := "SrcType := Real" } EQ_Contact(in1 := #iFEEDER_PLC_AUX_VALUES.i_rCarriergasActual_Line1, in2 := 0.0)
      { S7_Templates := "SrcType := Real" } EQ_Contact(in1 := #iFEEDER_PLC_AUX_VALUES.i_rDiskActual_Line1, in2 := 0.0)
      { S7_Templates := "SrcType := Real" } EQ_Contact(in1 := #iFEEDER_PLC_AUX_VALUES.i_rStirrerActual_Line1, in2 := 0.0)
   END_RUNG wire#w2
   // the same network as SCL:
   IF "M_ONE" AND #O_BYTE_0.LINE_1_ENABLED THEN
       #SWITCH_ON_SEQUENCE_LINE_1(OPTIONS_0 := 2#0000_0001,   // "FB21250_POWDER_ON_OFF_SEQUENCE"
                               REQUEST_INPUT := #DATA.START_LINE_1,
                               GENERAL_CONDITIONS_INPUT := #DATA.START_GENERAL_CONDITIONS AND NOT #SWITCH_OFF_SEQUENCE_LINE_1.RUNNING,
                               INITIAL_CONDITIONS_INPUT := NOT #SWITCH_OFF_SEQUENCE_LINE_1.RUNNING AND (#iFEEDER_PLC_AUX_VALUES.i_rCarriergasActual_Line1 = 0.0) AND (#iFEEDER_PLC_AUX_VALUES.i_rDiskActual_Line1 = 0.0) AND (#iFEEDER_PLC_AUX_VALUES.i_rStirrerActual_Line1 = 0.0),
                               GAS_FLOW_ACTUAL := #iFEEDER_PLC_AUX_VALUES.i_rCarriergasActual_Line1,
                               DISK_SPEED_ACTUAL := #iFEEDER_PLC_AUX_VALUES.i_rDiskActual_Line1,
                               GAS_SETPOINT := #SWITCH_ON_SEQUENCE_LINE_1.GAS_SETPOINT,
                               DISK_SETPOINT := #SWITCH_ON_SEQUENCE_LINE_1.DISK_SETPOINT);
   END_IF;
END_REGION

REGION Network 23: SWITCH ON SEQUENCE LINE 2
   // 2#0000_0001 OPTIONS 0 BIT 0 ON SEQUENCE OPTION
   // 2#0000_0010 OPTIONS 0 BIT 1 OFF SEQUENCE OPTION
   // 2#0000_0100 OPTIONS 0 BIT 2 SPARE OPTION
   // 2#0000_1000 OPTIONS 0 BIT 3 SPARE OPTION
   // 2#0001_0000 OPTIONS 0 BIT 4 SPARE OPTION
   // 2#0010_0000 OPTIONS 0 BIT 5 SPARE OPTION
   // 2#0100_0000 OPTIONS 0 BIT 6 SPARE OPTION
   // 2#1000_0000 OPTIONS 0 BIT 7 SPARE OPTION
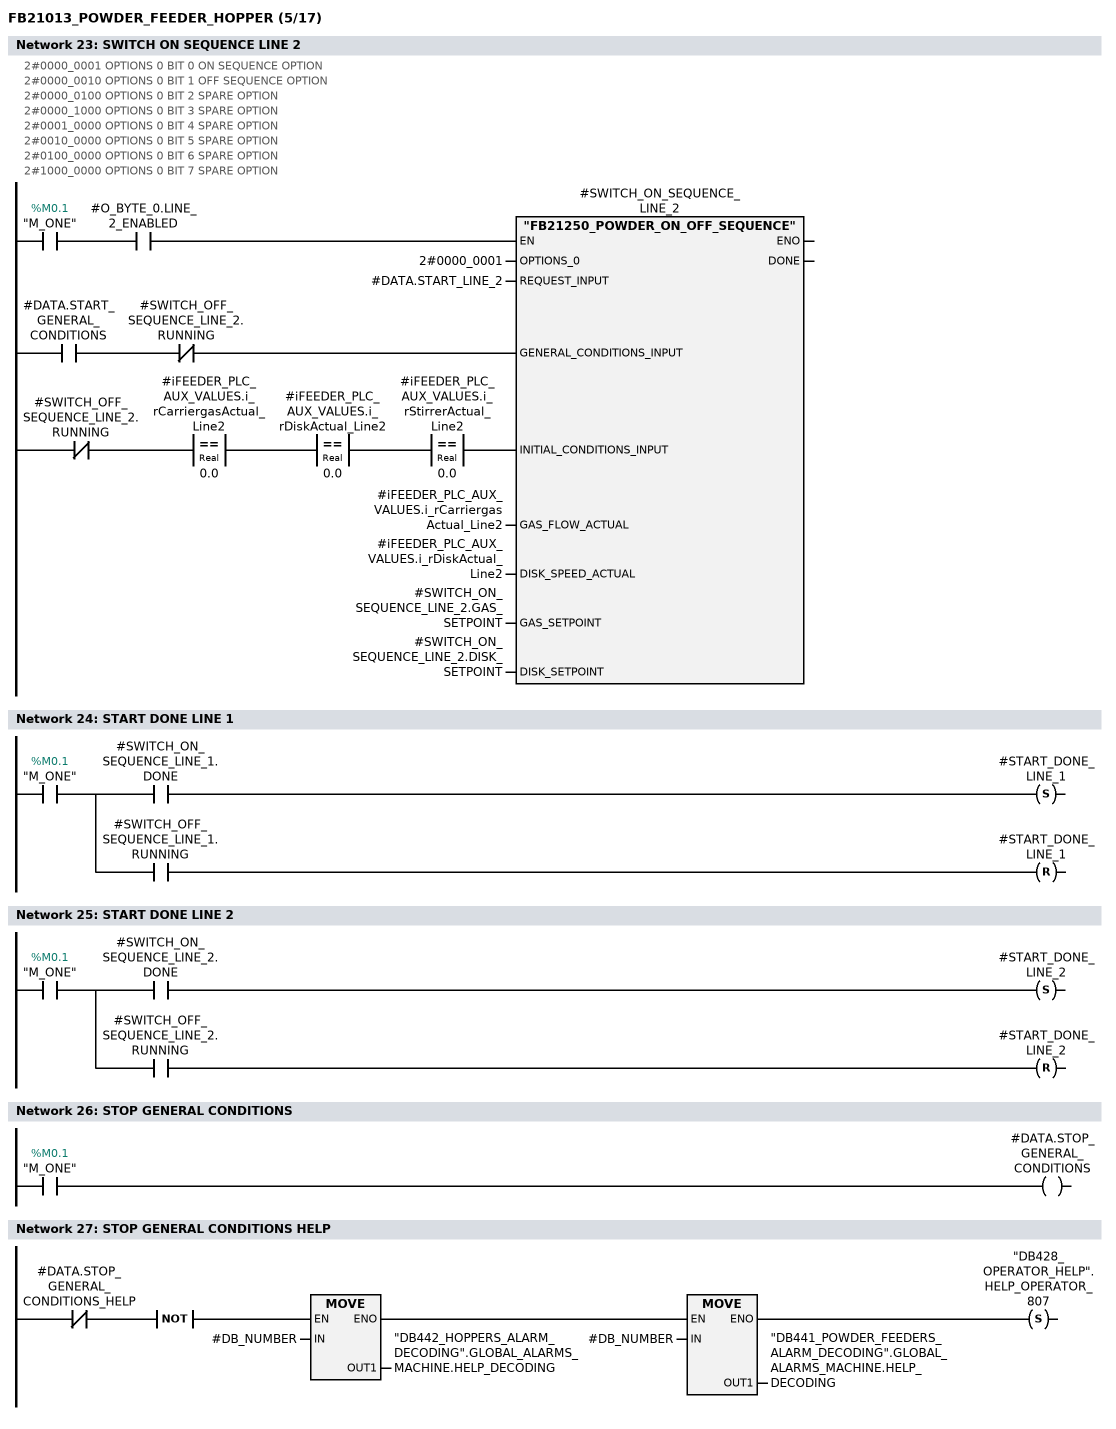
   RUNG wire#powerrail
      Contact( "M_ONE" )
      Contact( #O_BYTE_0.LINE_2_ENABLED )
      #SWITCH_ON_SEQUENCE_LINE_2(GENERAL_CONDITIONS_INPUT := wire#w1, INITIAL_CONDITIONS_INPUT := wire#w2, OPTIONS_0 := 2#0000_0001, REQUEST_INPUT := #DATA.START_LINE_2, GAS_FLOW_ACTUAL := #iFEEDER_PLC_AUX_VALUES.i_rCarriergasActual_Line2, DISK_SPEED_ACTUAL := #iFEEDER_PLC_AUX_VALUES.i_rDiskActual_Line2, GAS_SETPOINT := #SWITCH_ON_SEQUENCE_LINE_2.GAS_SETPOINT, DISK_SETPOINT := #SWITCH_ON_SEQUENCE_LINE_2.DISK_SETPOINT, DONE =>)
   END_RUNG
   RUNG wire#powerrail
      Contact( #DATA.START_GENERAL_CONDITIONS )
      I_Contact( #SWITCH_OFF_SEQUENCE_LINE_2.RUNNING )
   END_RUNG wire#w1
   RUNG wire#powerrail
      I_Contact( #SWITCH_OFF_SEQUENCE_LINE_2.RUNNING )
      { S7_Templates := "SrcType := Real" } EQ_Contact(in1 := #iFEEDER_PLC_AUX_VALUES.i_rCarriergasActual_Line2, in2 := 0.0)
      { S7_Templates := "SrcType := Real" } EQ_Contact(in1 := #iFEEDER_PLC_AUX_VALUES.i_rDiskActual_Line2, in2 := 0.0)
      { S7_Templates := "SrcType := Real" } EQ_Contact(in1 := #iFEEDER_PLC_AUX_VALUES.i_rStirrerActual_Line2, in2 := 0.0)
   END_RUNG wire#w2
   // the same network as SCL:
   IF "M_ONE" AND #O_BYTE_0.LINE_2_ENABLED THEN
       #SWITCH_ON_SEQUENCE_LINE_2(OPTIONS_0 := 2#0000_0001,   // "FB21250_POWDER_ON_OFF_SEQUENCE"
                               REQUEST_INPUT := #DATA.START_LINE_2,
                               GENERAL_CONDITIONS_INPUT := #DATA.START_GENERAL_CONDITIONS AND NOT #SWITCH_OFF_SEQUENCE_LINE_2.RUNNING,
                               INITIAL_CONDITIONS_INPUT := NOT #SWITCH_OFF_SEQUENCE_LINE_2.RUNNING AND (#iFEEDER_PLC_AUX_VALUES.i_rCarriergasActual_Line2 = 0.0) AND (#iFEEDER_PLC_AUX_VALUES.i_rDiskActual_Line2 = 0.0) AND (#iFEEDER_PLC_AUX_VALUES.i_rStirrerActual_Line2 = 0.0),
                               GAS_FLOW_ACTUAL := #iFEEDER_PLC_AUX_VALUES.i_rCarriergasActual_Line2,
                               DISK_SPEED_ACTUAL := #iFEEDER_PLC_AUX_VALUES.i_rDiskActual_Line2,
                               GAS_SETPOINT := #SWITCH_ON_SEQUENCE_LINE_2.GAS_SETPOINT,
                               DISK_SETPOINT := #SWITCH_ON_SEQUENCE_LINE_2.DISK_SETPOINT);
   END_IF;
END_REGION

REGION Network 24: START DONE LINE 1
   RUNG wire#powerrail
      Contact( "M_ONE" )
      wire#w1
      Contact( #SWITCH_ON_SEQUENCE_LINE_1.DONE )
      S_Coil( #START_DONE_LINE_1 )
   END_RUNG
   RUNG wire#w1
      Contact( #SWITCH_OFF_SEQUENCE_LINE_1.RUNNING )
      R_Coil( #START_DONE_LINE_1 )
   END_RUNG
   // the same network as SCL:
   IF "M_ONE" AND #SWITCH_ON_SEQUENCE_LINE_1.DONE THEN #START_DONE_LINE_1 := TRUE; END_IF;
   IF "M_ONE" AND #SWITCH_OFF_SEQUENCE_LINE_1.RUNNING THEN #START_DONE_LINE_1 := FALSE; END_IF;
END_REGION

REGION Network 25: START DONE LINE 2
   RUNG wire#powerrail
      Contact( "M_ONE" )
      wire#w1
      Contact( #SWITCH_ON_SEQUENCE_LINE_2.DONE )
      S_Coil( #START_DONE_LINE_2 )
   END_RUNG
   RUNG wire#w1
      Contact( #SWITCH_OFF_SEQUENCE_LINE_2.RUNNING )
      R_Coil( #START_DONE_LINE_2 )
   END_RUNG
   // the same network as SCL:
   IF "M_ONE" AND #SWITCH_ON_SEQUENCE_LINE_2.DONE THEN #START_DONE_LINE_2 := TRUE; END_IF;
   IF "M_ONE" AND #SWITCH_OFF_SEQUENCE_LINE_2.RUNNING THEN #START_DONE_LINE_2 := FALSE; END_IF;
END_REGION

REGION Network 26: STOP GENERAL CONDITIONS
   RUNG wire#powerrail
      Contact( "M_ONE" )
      Coil( #DATA.STOP_GENERAL_CONDITIONS )
   END_RUNG
   // the same network as SCL:
   #DATA.STOP_GENERAL_CONDITIONS := "M_ONE";
END_REGION

REGION Network 27: STOP GENERAL CONDITIONS HELP
   RUNG wire#powerrail
      I_Contact( #DATA.STOP_GENERAL_CONDITIONS_HELP )
      Not()
      Move(in := #DB_NUMBER, out1 => "DB442_HOPPERS_ALARM_DECODING".GLOBAL_ALARMS_MACHINE.HELP_DECODING)
      Move(in := #DB_NUMBER, out1 => "DB441_POWDER_FEEDERS_ALARM_DECODING".GLOBAL_ALARMS_MACHINE.HELP_DECODING)
      S_Coil( "DB428_OPERATOR_HELP".HELP_OPERATOR_807 )
   END_RUNG
   // the same network as SCL:
   IF NOT (NOT #DATA.STOP_GENERAL_CONDITIONS_HELP) THEN
       "DB442_HOPPERS_ALARM_DECODING".GLOBAL_ALARMS_MACHINE.HELP_DECODING := #DB_NUMBER;
       "DB441_POWDER_FEEDERS_ALARM_DECODING".GLOBAL_ALARMS_MACHINE.HELP_DECODING := #DB_NUMBER;
       "DB428_OPERATOR_HELP".HELP_OPERATOR_807 := TRUE;
   END_IF;
END_REGION

REGION Network 28: STOP INITIAL CONDITIONS LINE 1
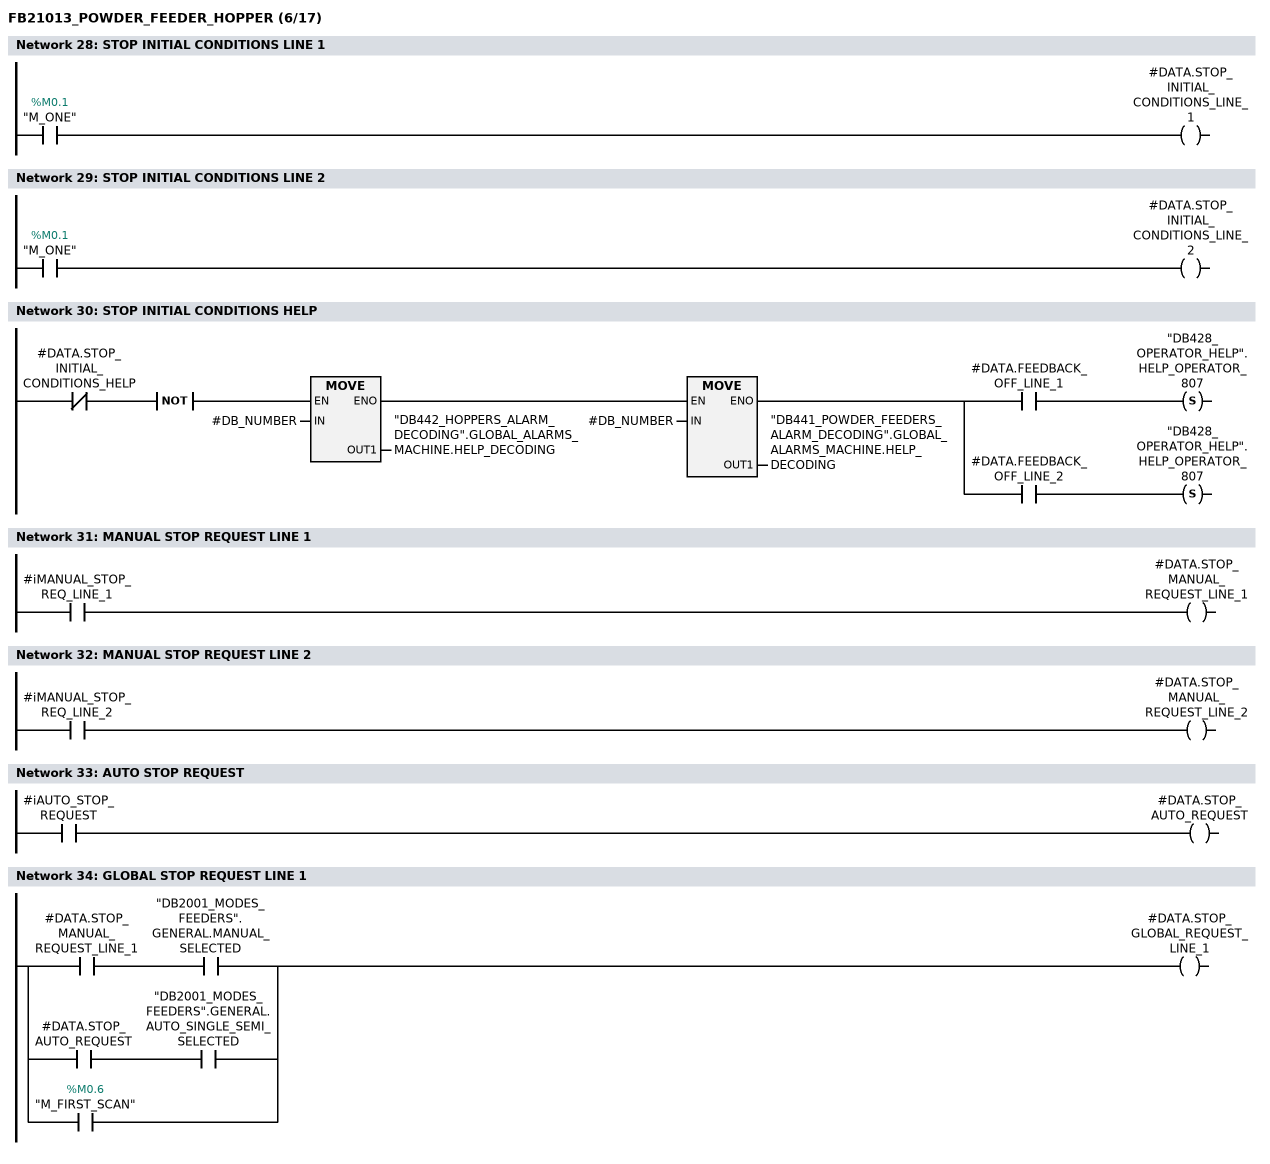
   RUNG wire#powerrail
      Contact( "M_ONE" )
      Coil( #DATA.STOP_INITIAL_CONDITIONS_LINE_1 )
   END_RUNG
   // the same network as SCL:
   #DATA.STOP_INITIAL_CONDITIONS_LINE_1 := "M_ONE";
END_REGION

REGION Network 29: STOP INITIAL CONDITIONS LINE 2
   RUNG wire#powerrail
      Contact( "M_ONE" )
      Coil( #DATA.STOP_INITIAL_CONDITIONS_LINE_2 )
   END_RUNG
   // the same network as SCL:
   #DATA.STOP_INITIAL_CONDITIONS_LINE_2 := "M_ONE";
END_REGION

REGION Network 30: STOP INITIAL CONDITIONS HELP
   RUNG wire#powerrail
      I_Contact( #DATA.STOP_INITIAL_CONDITIONS_HELP )
      Not()
      Move(in := #DB_NUMBER, out1 => "DB442_HOPPERS_ALARM_DECODING".GLOBAL_ALARMS_MACHINE.HELP_DECODING)
      Move(in := #DB_NUMBER, out1 => "DB441_POWDER_FEEDERS_ALARM_DECODING".GLOBAL_ALARMS_MACHINE.HELP_DECODING)
      wire#w1
      Contact( #DATA.FEEDBACK_OFF_LINE_1 )
      S_Coil( "DB428_OPERATOR_HELP".HELP_OPERATOR_807 )
   END_RUNG
   RUNG wire#w1
      Contact( #DATA.FEEDBACK_OFF_LINE_2 )
      S_Coil( "DB428_OPERATOR_HELP".HELP_OPERATOR_807 )
   END_RUNG
   // the same network as SCL:
   #_w1 := NOT (NOT #DATA.STOP_INITIAL_CONDITIONS_HELP);
   IF #_w1 THEN
       "DB442_HOPPERS_ALARM_DECODING".GLOBAL_ALARMS_MACHINE.HELP_DECODING := #DB_NUMBER;
       "DB441_POWDER_FEEDERS_ALARM_DECODING".GLOBAL_ALARMS_MACHINE.HELP_DECODING := #DB_NUMBER;
   END_IF;
   IF #_w1 AND #DATA.FEEDBACK_OFF_LINE_1 THEN "DB428_OPERATOR_HELP".HELP_OPERATOR_807 := TRUE; END_IF;
   IF #_w1 AND #DATA.FEEDBACK_OFF_LINE_2 THEN "DB428_OPERATOR_HELP".HELP_OPERATOR_807 := TRUE; END_IF;
END_REGION

REGION Network 31: MANUAL STOP REQUEST LINE 1
   RUNG wire#powerrail
      Contact( #iMANUAL_STOP_REQ_LINE_1 )
      Coil( #DATA.STOP_MANUAL_REQUEST_LINE_1 )
   END_RUNG
   // the same network as SCL:
   #DATA.STOP_MANUAL_REQUEST_LINE_1 := #iMANUAL_STOP_REQ_LINE_1;
END_REGION

REGION Network 32: MANUAL STOP REQUEST LINE 2
   RUNG wire#powerrail
      Contact( #iMANUAL_STOP_REQ_LINE_2 )
      Coil( #DATA.STOP_MANUAL_REQUEST_LINE_2 )
   END_RUNG
   // the same network as SCL:
   #DATA.STOP_MANUAL_REQUEST_LINE_2 := #iMANUAL_STOP_REQ_LINE_2;
END_REGION

REGION Network 33: AUTO STOP REQUEST
   RUNG wire#powerrail
      Contact( #iAUTO_STOP_REQUEST )
      Coil( #DATA.STOP_AUTO_REQUEST )
   END_RUNG
   // the same network as SCL:
   #DATA.STOP_AUTO_REQUEST := #iAUTO_STOP_REQUEST;
END_REGION

REGION Network 34: GLOBAL STOP REQUEST LINE 1
   RUNG wire#powerrail
      Contact( #DATA.STOP_MANUAL_REQUEST_LINE_1 )
      Contact( "DB2001_MODES_FEEDERS".GENERAL.MANUAL_SELECTED )
      wire#w1
      Coil( #DATA.STOP_GLOBAL_REQUEST_LINE_1 )
   END_RUNG
   RUNG wire#powerrail
      Contact( #DATA.STOP_AUTO_REQUEST )
      Contact( "DB2001_MODES_FEEDERS".GENERAL.AUTO_SINGLE_SEMI_SELECTED )
   END_RUNG wire#w1
   RUNG wire#powerrail
      Contact( "M_FIRST_SCAN" )
   END_RUNG wire#w1
   // the same network as SCL:
   #DATA.STOP_GLOBAL_REQUEST_LINE_1 := (#DATA.STOP_MANUAL_REQUEST_LINE_1 AND "DB2001_MODES_FEEDERS".GENERAL.MANUAL_SELECTED) OR (#DATA.STOP_AUTO_REQUEST AND "DB2001_MODES_FEEDERS".GENERAL.AUTO_SINGLE_SEMI_SELECTED) OR "M_FIRST_SCAN";
END_REGION

REGION Network 35: GLOBAL STOP REQUEST LINE 2
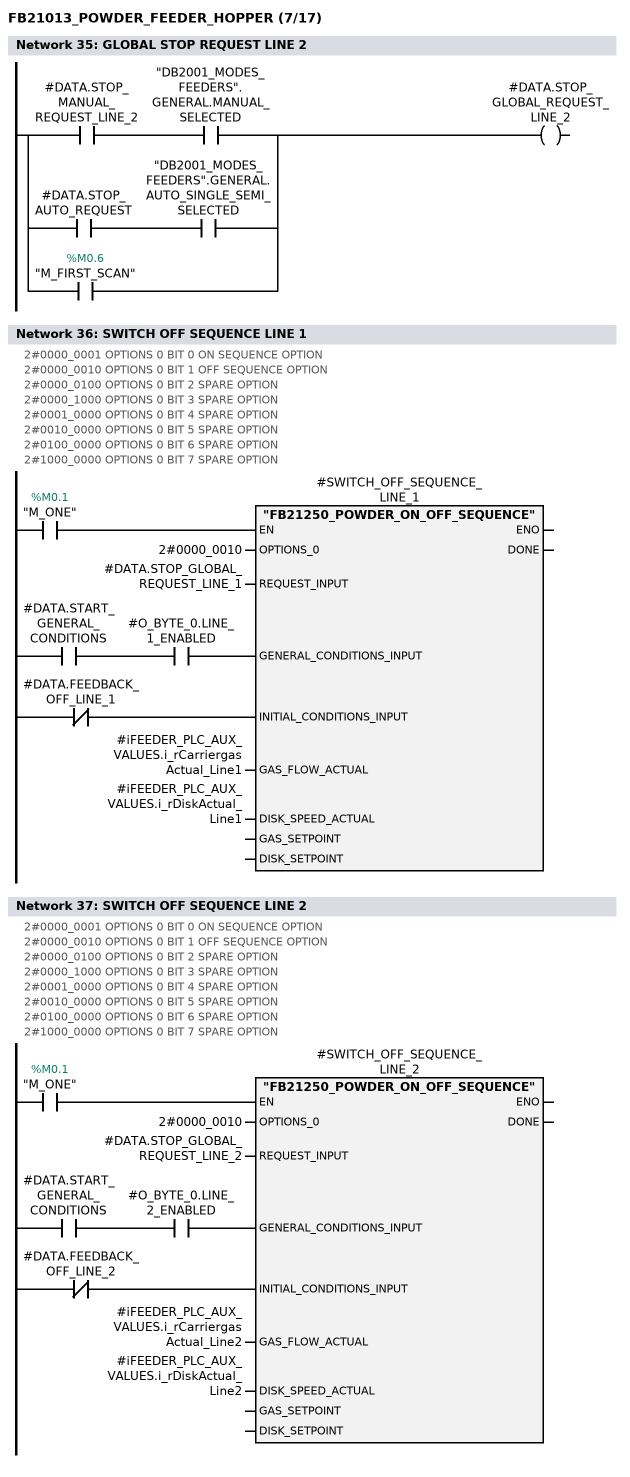
   RUNG wire#powerrail
      Contact( #DATA.STOP_MANUAL_REQUEST_LINE_2 )
      Contact( "DB2001_MODES_FEEDERS".GENERAL.MANUAL_SELECTED )
      wire#w1
      Coil( #DATA.STOP_GLOBAL_REQUEST_LINE_2 )
   END_RUNG
   RUNG wire#powerrail
      Contact( #DATA.STOP_AUTO_REQUEST )
      Contact( "DB2001_MODES_FEEDERS".GENERAL.AUTO_SINGLE_SEMI_SELECTED )
   END_RUNG wire#w1
   RUNG wire#powerrail
      Contact( "M_FIRST_SCAN" )
   END_RUNG wire#w1
   // the same network as SCL:
   #DATA.STOP_GLOBAL_REQUEST_LINE_2 := (#DATA.STOP_MANUAL_REQUEST_LINE_2 AND "DB2001_MODES_FEEDERS".GENERAL.MANUAL_SELECTED) OR (#DATA.STOP_AUTO_REQUEST AND "DB2001_MODES_FEEDERS".GENERAL.AUTO_SINGLE_SEMI_SELECTED) OR "M_FIRST_SCAN";
END_REGION

REGION Network 36: SWITCH OFF SEQUENCE LINE 1
   // 2#0000_0001 OPTIONS 0 BIT 0 ON SEQUENCE OPTION
   // 2#0000_0010 OPTIONS 0 BIT 1 OFF SEQUENCE OPTION
   // 2#0000_0100 OPTIONS 0 BIT 2 SPARE OPTION
   // 2#0000_1000 OPTIONS 0 BIT 3 SPARE OPTION
   // 2#0001_0000 OPTIONS 0 BIT 4 SPARE OPTION
   // 2#0010_0000 OPTIONS 0 BIT 5 SPARE OPTION
   // 2#0100_0000 OPTIONS 0 BIT 6 SPARE OPTION
   // 2#1000_0000 OPTIONS 0 BIT 7 SPARE OPTION
   RUNG wire#powerrail
      Contact( "M_ONE" )
      #SWITCH_OFF_SEQUENCE_LINE_1(GENERAL_CONDITIONS_INPUT := wire#w1, INITIAL_CONDITIONS_INPUT := wire#w2, OPTIONS_0 := 2#0000_0010, REQUEST_INPUT := #DATA.STOP_GLOBAL_REQUEST_LINE_1, GAS_FLOW_ACTUAL := #iFEEDER_PLC_AUX_VALUES.i_rCarriergasActual_Line1, DISK_SPEED_ACTUAL := #iFEEDER_PLC_AUX_VALUES.i_rDiskActual_Line1, GAS_SETPOINT :=, DISK_SETPOINT :=, DONE =>)
   END_RUNG
   RUNG wire#powerrail
      Contact( #DATA.START_GENERAL_CONDITIONS )
      Contact( #O_BYTE_0.LINE_1_ENABLED )
   END_RUNG wire#w1
   RUNG wire#powerrail
      I_Contact( #DATA.FEEDBACK_OFF_LINE_1 )
   END_RUNG wire#w2
   // the same network as SCL:
   IF "M_ONE" THEN
       #SWITCH_OFF_SEQUENCE_LINE_1(OPTIONS_0 := 2#0000_0010,   // "FB21250_POWDER_ON_OFF_SEQUENCE"
                               REQUEST_INPUT := #DATA.STOP_GLOBAL_REQUEST_LINE_1,
                               GENERAL_CONDITIONS_INPUT := #DATA.START_GENERAL_CONDITIONS AND #O_BYTE_0.LINE_1_ENABLED,
                               INITIAL_CONDITIONS_INPUT := NOT #DATA.FEEDBACK_OFF_LINE_1,
                               GAS_FLOW_ACTUAL := #iFEEDER_PLC_AUX_VALUES.i_rCarriergasActual_Line1,
                               DISK_SPEED_ACTUAL := #iFEEDER_PLC_AUX_VALUES.i_rDiskActual_Line1);
   END_IF;
END_REGION

REGION Network 37: SWITCH OFF SEQUENCE LINE 2
   // 2#0000_0001 OPTIONS 0 BIT 0 ON SEQUENCE OPTION
   // 2#0000_0010 OPTIONS 0 BIT 1 OFF SEQUENCE OPTION
   // 2#0000_0100 OPTIONS 0 BIT 2 SPARE OPTION
   // 2#0000_1000 OPTIONS 0 BIT 3 SPARE OPTION
   // 2#0001_0000 OPTIONS 0 BIT 4 SPARE OPTION
   // 2#0010_0000 OPTIONS 0 BIT 5 SPARE OPTION
   // 2#0100_0000 OPTIONS 0 BIT 6 SPARE OPTION
   // 2#1000_0000 OPTIONS 0 BIT 7 SPARE OPTION
   RUNG wire#powerrail
      Contact( "M_ONE" )
      #SWITCH_OFF_SEQUENCE_LINE_2(GENERAL_CONDITIONS_INPUT := wire#w1, INITIAL_CONDITIONS_INPUT := wire#w2, OPTIONS_0 := 2#0000_0010, REQUEST_INPUT := #DATA.STOP_GLOBAL_REQUEST_LINE_2, GAS_FLOW_ACTUAL := #iFEEDER_PLC_AUX_VALUES.i_rCarriergasActual_Line2, DISK_SPEED_ACTUAL := #iFEEDER_PLC_AUX_VALUES.i_rDiskActual_Line2, GAS_SETPOINT :=, DISK_SETPOINT :=, DONE =>)
   END_RUNG
   RUNG wire#powerrail
      Contact( #DATA.START_GENERAL_CONDITIONS )
      Contact( #O_BYTE_0.LINE_2_ENABLED )
   END_RUNG wire#w1
   RUNG wire#powerrail
      I_Contact( #DATA.FEEDBACK_OFF_LINE_2 )
   END_RUNG wire#w2
   // the same network as SCL:
   IF "M_ONE" THEN
       #SWITCH_OFF_SEQUENCE_LINE_2(OPTIONS_0 := 2#0000_0010,   // "FB21250_POWDER_ON_OFF_SEQUENCE"
                               REQUEST_INPUT := #DATA.STOP_GLOBAL_REQUEST_LINE_2,
                               GENERAL_CONDITIONS_INPUT := #DATA.START_GENERAL_CONDITIONS AND #O_BYTE_0.LINE_2_ENABLED,
                               INITIAL_CONDITIONS_INPUT := NOT #DATA.FEEDBACK_OFF_LINE_2,
                               GAS_FLOW_ACTUAL := #iFEEDER_PLC_AUX_VALUES.i_rCarriergasActual_Line2,
                               DISK_SPEED_ACTUAL := #iFEEDER_PLC_AUX_VALUES.i_rDiskActual_Line2);
   END_IF;
END_REGION

REGION Network 38: STOP COMMAND LINE 1
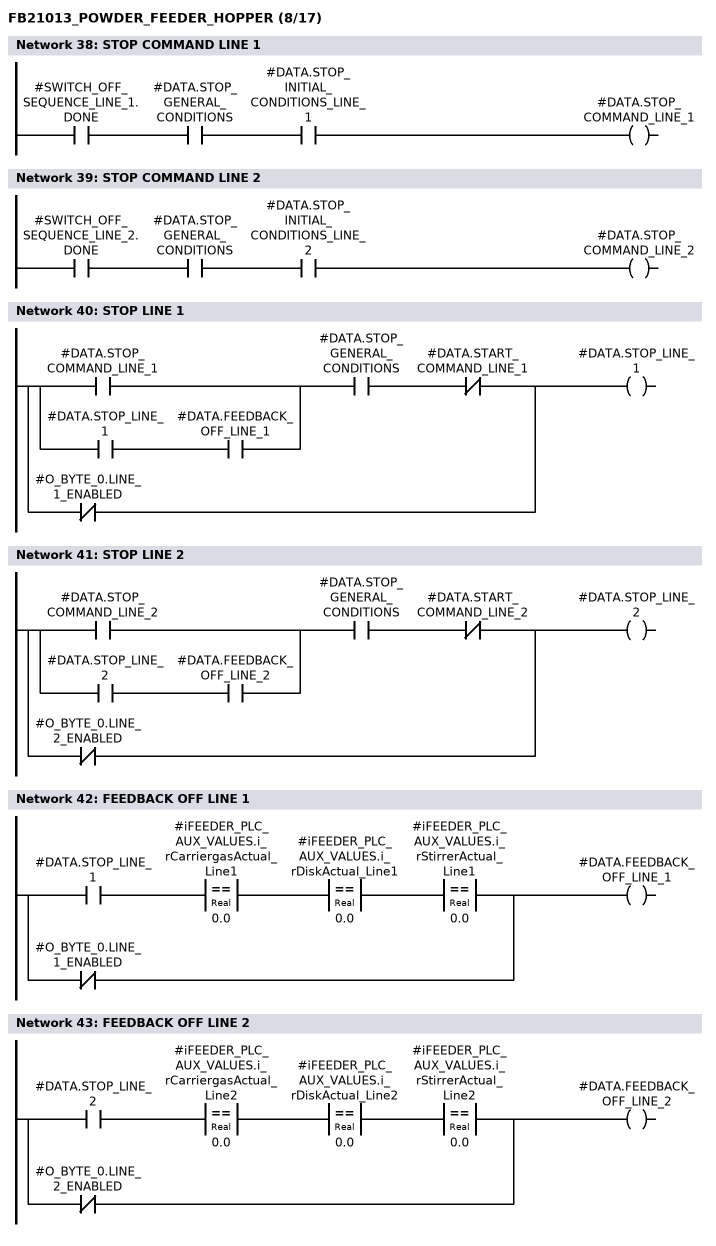
   RUNG wire#powerrail
      Contact( #SWITCH_OFF_SEQUENCE_LINE_1.DONE )
      Contact( #DATA.STOP_GENERAL_CONDITIONS )
      Contact( #DATA.STOP_INITIAL_CONDITIONS_LINE_1 )
      Coil( #DATA.STOP_COMMAND_LINE_1 )
   END_RUNG
   // the same network as SCL:
   #DATA.STOP_COMMAND_LINE_1 := #SWITCH_OFF_SEQUENCE_LINE_1.DONE AND #DATA.STOP_GENERAL_CONDITIONS AND #DATA.STOP_INITIAL_CONDITIONS_LINE_1;
END_REGION

REGION Network 39: STOP COMMAND LINE 2
   RUNG wire#powerrail
      Contact( #SWITCH_OFF_SEQUENCE_LINE_2.DONE )
      Contact( #DATA.STOP_GENERAL_CONDITIONS )
      Contact( #DATA.STOP_INITIAL_CONDITIONS_LINE_2 )
      Coil( #DATA.STOP_COMMAND_LINE_2 )
   END_RUNG
   // the same network as SCL:
   #DATA.STOP_COMMAND_LINE_2 := #SWITCH_OFF_SEQUENCE_LINE_2.DONE AND #DATA.STOP_GENERAL_CONDITIONS AND #DATA.STOP_INITIAL_CONDITIONS_LINE_2;
END_REGION

REGION Network 40: STOP LINE 1
   RUNG wire#powerrail
      Contact( #DATA.STOP_COMMAND_LINE_1 )
      wire#w1
      Contact( #DATA.STOP_GENERAL_CONDITIONS )
      I_Contact( #DATA.START_COMMAND_LINE_1 )
      wire#w2
      Coil( #DATA.STOP_LINE_1 )
   END_RUNG
   RUNG wire#powerrail
      Contact( #DATA.STOP_LINE_1 )
      Contact( #DATA.FEEDBACK_OFF_LINE_1 )
   END_RUNG wire#w1
   RUNG wire#powerrail
      I_Contact( #O_BYTE_0.LINE_1_ENABLED )
   END_RUNG wire#w2
   // the same network as SCL:
   #DATA.STOP_LINE_1 := ((#DATA.STOP_COMMAND_LINE_1 OR (#DATA.STOP_LINE_1 AND #DATA.FEEDBACK_OFF_LINE_1)) AND #DATA.STOP_GENERAL_CONDITIONS AND NOT #DATA.START_COMMAND_LINE_1) OR NOT #O_BYTE_0.LINE_1_ENABLED;
END_REGION

REGION Network 41: STOP LINE 2
   RUNG wire#powerrail
      Contact( #DATA.STOP_COMMAND_LINE_2 )
      wire#w1
      Contact( #DATA.STOP_GENERAL_CONDITIONS )
      I_Contact( #DATA.START_COMMAND_LINE_2 )
      wire#w2
      Coil( #DATA.STOP_LINE_2 )
   END_RUNG
   RUNG wire#powerrail
      Contact( #DATA.STOP_LINE_2 )
      Contact( #DATA.FEEDBACK_OFF_LINE_2 )
   END_RUNG wire#w1
   RUNG wire#powerrail
      I_Contact( #O_BYTE_0.LINE_2_ENABLED )
   END_RUNG wire#w2
   // the same network as SCL:
   #DATA.STOP_LINE_2 := ((#DATA.STOP_COMMAND_LINE_2 OR (#DATA.STOP_LINE_2 AND #DATA.FEEDBACK_OFF_LINE_2)) AND #DATA.STOP_GENERAL_CONDITIONS AND NOT #DATA.START_COMMAND_LINE_2) OR NOT #O_BYTE_0.LINE_2_ENABLED;
END_REGION

REGION Network 42: FEEDBACK OFF LINE 1
   RUNG wire#powerrail
      Contact( #DATA.STOP_LINE_1 )
      { S7_Templates := "SrcType := Real" } EQ_Contact(in1 := #iFEEDER_PLC_AUX_VALUES.i_rCarriergasActual_Line1, in2 := 0.0)
      { S7_Templates := "SrcType := Real" } EQ_Contact(in1 := #iFEEDER_PLC_AUX_VALUES.i_rDiskActual_Line1, in2 := 0.0)
      { S7_Templates := "SrcType := Real" } EQ_Contact(in1 := #iFEEDER_PLC_AUX_VALUES.i_rStirrerActual_Line1, in2 := 0.0)
      wire#w1
      Coil( #DATA.FEEDBACK_OFF_LINE_1 )
   END_RUNG
   RUNG wire#powerrail
      I_Contact( #O_BYTE_0.LINE_1_ENABLED )
   END_RUNG wire#w1
   // the same network as SCL:
   #DATA.FEEDBACK_OFF_LINE_1 := (#DATA.STOP_LINE_1 AND (#iFEEDER_PLC_AUX_VALUES.i_rCarriergasActual_Line1 = 0.0) AND (#iFEEDER_PLC_AUX_VALUES.i_rDiskActual_Line1 = 0.0) AND (#iFEEDER_PLC_AUX_VALUES.i_rStirrerActual_Line1 = 0.0)) OR NOT #O_BYTE_0.LINE_1_ENABLED;
END_REGION

REGION Network 43: FEEDBACK OFF LINE 2
   RUNG wire#powerrail
      Contact( #DATA.STOP_LINE_2 )
      { S7_Templates := "SrcType := Real" } EQ_Contact(in1 := #iFEEDER_PLC_AUX_VALUES.i_rCarriergasActual_Line2, in2 := 0.0)
      { S7_Templates := "SrcType := Real" } EQ_Contact(in1 := #iFEEDER_PLC_AUX_VALUES.i_rDiskActual_Line2, in2 := 0.0)
      { S7_Templates := "SrcType := Real" } EQ_Contact(in1 := #iFEEDER_PLC_AUX_VALUES.i_rStirrerActual_Line2, in2 := 0.0)
      wire#w1
      Coil( #DATA.FEEDBACK_OFF_LINE_2 )
   END_RUNG
   RUNG wire#powerrail
      I_Contact( #O_BYTE_0.LINE_2_ENABLED )
   END_RUNG wire#w1
   // the same network as SCL:
   #DATA.FEEDBACK_OFF_LINE_2 := (#DATA.STOP_LINE_2 AND (#iFEEDER_PLC_AUX_VALUES.i_rCarriergasActual_Line2 = 0.0) AND (#iFEEDER_PLC_AUX_VALUES.i_rDiskActual_Line2 = 0.0) AND (#iFEEDER_PLC_AUX_VALUES.i_rStirrerActual_Line2 = 0.0)) OR NOT #O_BYTE_0.LINE_2_ENABLED;
END_REGION

REGION Network 44: POWDER LINE CLOGGED FAULT LINE 1 (IS ALARM)
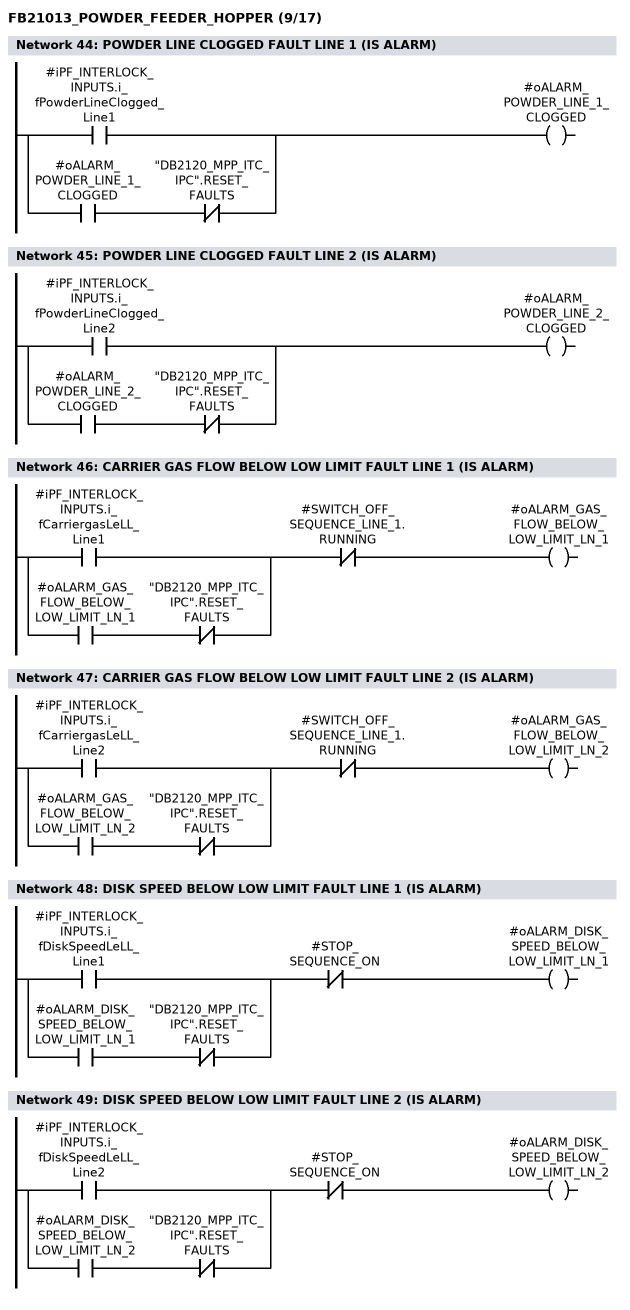
   RUNG wire#powerrail
      Contact( #iPF_INTERLOCK_INPUTS.i_fPowderLineClogged_Line1 )
      wire#w1
      Coil( #oALARM_POWDER_LINE_1_CLOGGED )
   END_RUNG
   RUNG wire#powerrail
      Contact( #oALARM_POWDER_LINE_1_CLOGGED )
      I_Contact( "DB2120_MPP_ITC_IPC".RESET_FAULTS )
   END_RUNG wire#w1
   // the same network as SCL:
   #oALARM_POWDER_LINE_1_CLOGGED := #iPF_INTERLOCK_INPUTS.i_fPowderLineClogged_Line1 OR (#oALARM_POWDER_LINE_1_CLOGGED AND NOT "DB2120_MPP_ITC_IPC".RESET_FAULTS);
END_REGION

REGION Network 45: POWDER LINE CLOGGED FAULT LINE 2 (IS ALARM)
   RUNG wire#powerrail
      Contact( #iPF_INTERLOCK_INPUTS.i_fPowderLineClogged_Line2 )
      wire#w1
      Coil( #oALARM_POWDER_LINE_2_CLOGGED )
   END_RUNG
   RUNG wire#powerrail
      Contact( #oALARM_POWDER_LINE_2_CLOGGED )
      I_Contact( "DB2120_MPP_ITC_IPC".RESET_FAULTS )
   END_RUNG wire#w1
   // the same network as SCL:
   #oALARM_POWDER_LINE_2_CLOGGED := #iPF_INTERLOCK_INPUTS.i_fPowderLineClogged_Line2 OR (#oALARM_POWDER_LINE_2_CLOGGED AND NOT "DB2120_MPP_ITC_IPC".RESET_FAULTS);
END_REGION

REGION Network 46: CARRIER GAS FLOW BELOW LOW LIMIT FAULT LINE 1 (IS ALARM)
   RUNG wire#powerrail
      Contact( #iPF_INTERLOCK_INPUTS.i_fCarriergasLeLL_Line1 )
      wire#w1
      I_Contact( #SWITCH_OFF_SEQUENCE_LINE_1.RUNNING )
      Coil( #oALARM_GAS_FLOW_BELOW_LOW_LIMIT_LN_1 )
   END_RUNG
   RUNG wire#powerrail
      Contact( #oALARM_GAS_FLOW_BELOW_LOW_LIMIT_LN_1 )
      I_Contact( "DB2120_MPP_ITC_IPC".RESET_FAULTS )
   END_RUNG wire#w1
   // the same network as SCL:
   #oALARM_GAS_FLOW_BELOW_LOW_LIMIT_LN_1 := (#iPF_INTERLOCK_INPUTS.i_fCarriergasLeLL_Line1 OR (#oALARM_GAS_FLOW_BELOW_LOW_LIMIT_LN_1 AND NOT "DB2120_MPP_ITC_IPC".RESET_FAULTS)) AND NOT #SWITCH_OFF_SEQUENCE_LINE_1.RUNNING;
END_REGION

REGION Network 47: CARRIER GAS FLOW BELOW LOW LIMIT FAULT LINE 2 (IS ALARM)
   RUNG wire#powerrail
      Contact( #iPF_INTERLOCK_INPUTS.i_fCarriergasLeLL_Line2 )
      wire#w1
      I_Contact( #SWITCH_OFF_SEQUENCE_LINE_1.RUNNING )
      Coil( #oALARM_GAS_FLOW_BELOW_LOW_LIMIT_LN_2 )
   END_RUNG
   RUNG wire#powerrail
      Contact( #oALARM_GAS_FLOW_BELOW_LOW_LIMIT_LN_2 )
      I_Contact( "DB2120_MPP_ITC_IPC".RESET_FAULTS )
   END_RUNG wire#w1
   // the same network as SCL:
   #oALARM_GAS_FLOW_BELOW_LOW_LIMIT_LN_2 := (#iPF_INTERLOCK_INPUTS.i_fCarriergasLeLL_Line2 OR (#oALARM_GAS_FLOW_BELOW_LOW_LIMIT_LN_2 AND NOT "DB2120_MPP_ITC_IPC".RESET_FAULTS)) AND NOT #SWITCH_OFF_SEQUENCE_LINE_1.RUNNING;
END_REGION

REGION Network 48: DISK SPEED BELOW LOW LIMIT FAULT LINE 1 (IS ALARM)
   RUNG wire#powerrail
      Contact( #iPF_INTERLOCK_INPUTS.i_fDiskSpeedLeLL_Line1 )
      wire#w1
      I_Contact( #STOP_SEQUENCE_ON )
      Coil( #oALARM_DISK_SPEED_BELOW_LOW_LIMIT_LN_1 )
   END_RUNG
   RUNG wire#powerrail
      Contact( #oALARM_DISK_SPEED_BELOW_LOW_LIMIT_LN_1 )
      I_Contact( "DB2120_MPP_ITC_IPC".RESET_FAULTS )
   END_RUNG wire#w1
   // the same network as SCL:
   #oALARM_DISK_SPEED_BELOW_LOW_LIMIT_LN_1 := (#iPF_INTERLOCK_INPUTS.i_fDiskSpeedLeLL_Line1 OR (#oALARM_DISK_SPEED_BELOW_LOW_LIMIT_LN_1 AND NOT "DB2120_MPP_ITC_IPC".RESET_FAULTS)) AND NOT #STOP_SEQUENCE_ON;
END_REGION

REGION Network 49: DISK SPEED BELOW LOW LIMIT FAULT LINE 2 (IS ALARM)
   RUNG wire#powerrail
      Contact( #iPF_INTERLOCK_INPUTS.i_fDiskSpeedLeLL_Line2 )
      wire#w1
      I_Contact( #STOP_SEQUENCE_ON )
      Coil( #oALARM_DISK_SPEED_BELOW_LOW_LIMIT_LN_2 )
   END_RUNG
   RUNG wire#powerrail
      Contact( #oALARM_DISK_SPEED_BELOW_LOW_LIMIT_LN_2 )
      I_Contact( "DB2120_MPP_ITC_IPC".RESET_FAULTS )
   END_RUNG wire#w1
   // the same network as SCL:
   #oALARM_DISK_SPEED_BELOW_LOW_LIMIT_LN_2 := (#iPF_INTERLOCK_INPUTS.i_fDiskSpeedLeLL_Line2 OR (#oALARM_DISK_SPEED_BELOW_LOW_LIMIT_LN_2 AND NOT "DB2120_MPP_ITC_IPC".RESET_FAULTS)) AND NOT #STOP_SEQUENCE_ON;
END_REGION

REGION Network 50: STIRRER SPEED BELOW LOW LIMIT FAULT LINE 1 (IS ALARM)
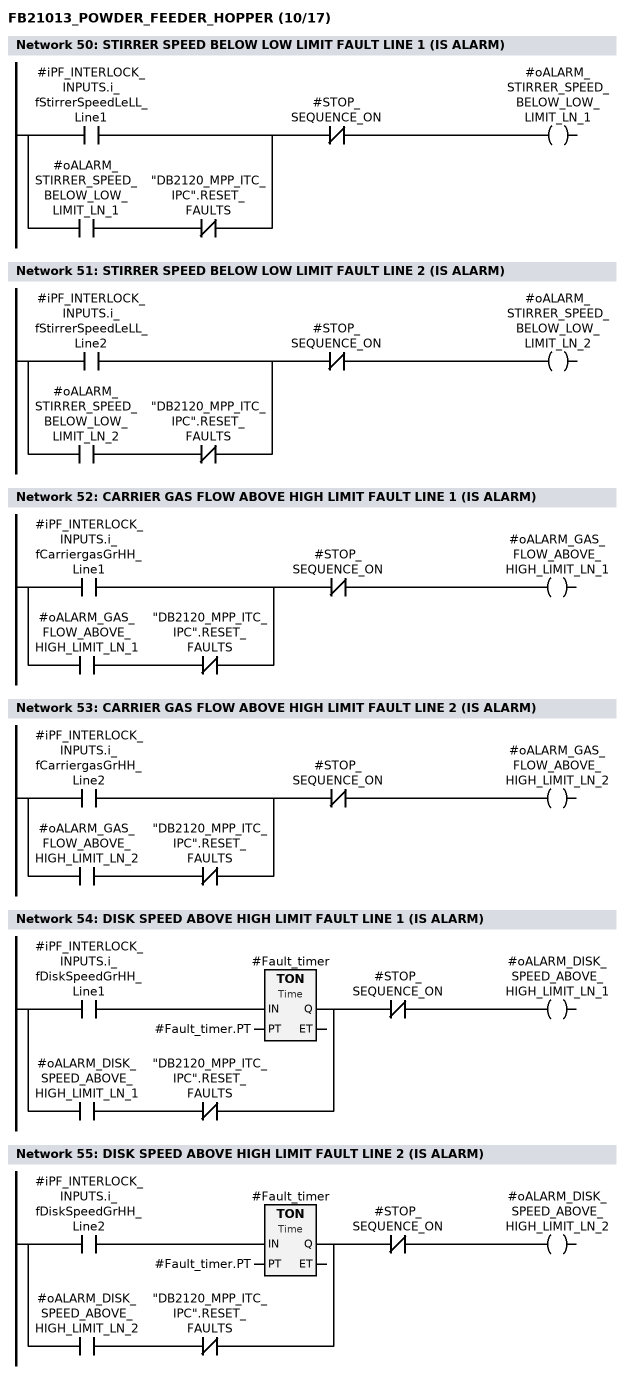
   RUNG wire#powerrail
      Contact( #iPF_INTERLOCK_INPUTS.i_fStirrerSpeedLeLL_Line1 )
      wire#w1
      I_Contact( #STOP_SEQUENCE_ON )
      Coil( #oALARM_STIRRER_SPEED_BELOW_LOW_LIMIT_LN_1 )
   END_RUNG
   RUNG wire#powerrail
      Contact( #oALARM_STIRRER_SPEED_BELOW_LOW_LIMIT_LN_1 )
      I_Contact( "DB2120_MPP_ITC_IPC".RESET_FAULTS )
   END_RUNG wire#w1
   // the same network as SCL:
   #oALARM_STIRRER_SPEED_BELOW_LOW_LIMIT_LN_1 := (#iPF_INTERLOCK_INPUTS.i_fStirrerSpeedLeLL_Line1 OR (#oALARM_STIRRER_SPEED_BELOW_LOW_LIMIT_LN_1 AND NOT "DB2120_MPP_ITC_IPC".RESET_FAULTS)) AND NOT #STOP_SEQUENCE_ON;
END_REGION

REGION Network 51: STIRRER SPEED BELOW LOW LIMIT FAULT LINE 2 (IS ALARM)
   RUNG wire#powerrail
      Contact( #iPF_INTERLOCK_INPUTS.i_fStirrerSpeedLeLL_Line2 )
      wire#w1
      I_Contact( #STOP_SEQUENCE_ON )
      Coil( #oALARM_STIRRER_SPEED_BELOW_LOW_LIMIT_LN_2 )
   END_RUNG
   RUNG wire#powerrail
      Contact( #oALARM_STIRRER_SPEED_BELOW_LOW_LIMIT_LN_2 )
      I_Contact( "DB2120_MPP_ITC_IPC".RESET_FAULTS )
   END_RUNG wire#w1
   // the same network as SCL:
   #oALARM_STIRRER_SPEED_BELOW_LOW_LIMIT_LN_2 := (#iPF_INTERLOCK_INPUTS.i_fStirrerSpeedLeLL_Line2 OR (#oALARM_STIRRER_SPEED_BELOW_LOW_LIMIT_LN_2 AND NOT "DB2120_MPP_ITC_IPC".RESET_FAULTS)) AND NOT #STOP_SEQUENCE_ON;
END_REGION

REGION Network 52: CARRIER GAS FLOW ABOVE HIGH LIMIT FAULT LINE 1 (IS ALARM)
   RUNG wire#powerrail
      Contact( #iPF_INTERLOCK_INPUTS.i_fCarriergasGrHH_Line1 )
      wire#w1
      I_Contact( #STOP_SEQUENCE_ON )
      Coil( #oALARM_GAS_FLOW_ABOVE_HIGH_LIMIT_LN_1 )
   END_RUNG
   RUNG wire#powerrail
      Contact( #oALARM_GAS_FLOW_ABOVE_HIGH_LIMIT_LN_1 )
      I_Contact( "DB2120_MPP_ITC_IPC".RESET_FAULTS )
   END_RUNG wire#w1
   // the same network as SCL:
   #oALARM_GAS_FLOW_ABOVE_HIGH_LIMIT_LN_1 := (#iPF_INTERLOCK_INPUTS.i_fCarriergasGrHH_Line1 OR (#oALARM_GAS_FLOW_ABOVE_HIGH_LIMIT_LN_1 AND NOT "DB2120_MPP_ITC_IPC".RESET_FAULTS)) AND NOT #STOP_SEQUENCE_ON;
END_REGION

REGION Network 53: CARRIER GAS FLOW ABOVE HIGH LIMIT FAULT LINE 2 (IS ALARM)
   RUNG wire#powerrail
      Contact( #iPF_INTERLOCK_INPUTS.i_fCarriergasGrHH_Line2 )
      wire#w1
      I_Contact( #STOP_SEQUENCE_ON )
      Coil( #oALARM_GAS_FLOW_ABOVE_HIGH_LIMIT_LN_2 )
   END_RUNG
   RUNG wire#powerrail
      Contact( #oALARM_GAS_FLOW_ABOVE_HIGH_LIMIT_LN_2 )
      I_Contact( "DB2120_MPP_ITC_IPC".RESET_FAULTS )
   END_RUNG wire#w1
   // the same network as SCL:
   #oALARM_GAS_FLOW_ABOVE_HIGH_LIMIT_LN_2 := (#iPF_INTERLOCK_INPUTS.i_fCarriergasGrHH_Line2 OR (#oALARM_GAS_FLOW_ABOVE_HIGH_LIMIT_LN_2 AND NOT "DB2120_MPP_ITC_IPC".RESET_FAULTS)) AND NOT #STOP_SEQUENCE_ON;
END_REGION

REGION Network 54: DISK SPEED ABOVE HIGH LIMIT FAULT LINE 1 (IS ALARM)
   RUNG wire#powerrail
      Contact( #iPF_INTERLOCK_INPUTS.i_fDiskSpeedGrHH_Line1 )
      { S7_Templates := "time_type := Time" } #Fault_timer.TON(pt := #Fault_timer.PT, et =>)
      wire#w1
      I_Contact( #STOP_SEQUENCE_ON )
      Coil( #oALARM_DISK_SPEED_ABOVE_HIGH_LIMIT_LN_1 )
   END_RUNG
   RUNG wire#powerrail
      Contact( #oALARM_DISK_SPEED_ABOVE_HIGH_LIMIT_LN_1 )
      I_Contact( "DB2120_MPP_ITC_IPC".RESET_FAULTS )
   END_RUNG wire#w1
   // the same network as SCL:
   #Fault_timer(IN := #iPF_INTERLOCK_INPUTS.i_fDiskSpeedGrHH_Line1, PT := #Fault_timer.PT);   // TON
   #oALARM_DISK_SPEED_ABOVE_HIGH_LIMIT_LN_1 := (#Fault_timer.Q OR (#oALARM_DISK_SPEED_ABOVE_HIGH_LIMIT_LN_1 AND NOT "DB2120_MPP_ITC_IPC".RESET_FAULTS)) AND NOT #STOP_SEQUENCE_ON;
END_REGION

REGION Network 55: DISK SPEED ABOVE HIGH LIMIT FAULT LINE 2 (IS ALARM)
   RUNG wire#powerrail
      Contact( #iPF_INTERLOCK_INPUTS.i_fDiskSpeedGrHH_Line2 )
      { S7_Templates := "time_type := Time" } #Fault_timer.TON(pt := #Fault_timer.PT, et =>)
      wire#w1
      I_Contact( #STOP_SEQUENCE_ON )
      Coil( #oALARM_DISK_SPEED_ABOVE_HIGH_LIMIT_LN_2 )
   END_RUNG
   RUNG wire#powerrail
      Contact( #oALARM_DISK_SPEED_ABOVE_HIGH_LIMIT_LN_2 )
      I_Contact( "DB2120_MPP_ITC_IPC".RESET_FAULTS )
   END_RUNG wire#w1
   // the same network as SCL:
   #Fault_timer(IN := #iPF_INTERLOCK_INPUTS.i_fDiskSpeedGrHH_Line2, PT := #Fault_timer.PT);   // TON
   #oALARM_DISK_SPEED_ABOVE_HIGH_LIMIT_LN_2 := (#Fault_timer.Q OR (#oALARM_DISK_SPEED_ABOVE_HIGH_LIMIT_LN_2 AND NOT "DB2120_MPP_ITC_IPC".RESET_FAULTS)) AND NOT #STOP_SEQUENCE_ON;
END_REGION

REGION Network 56: STIRRER SPEED ABOVE HIGH LIMIT FAULT LINE 1 (IS ALARM)
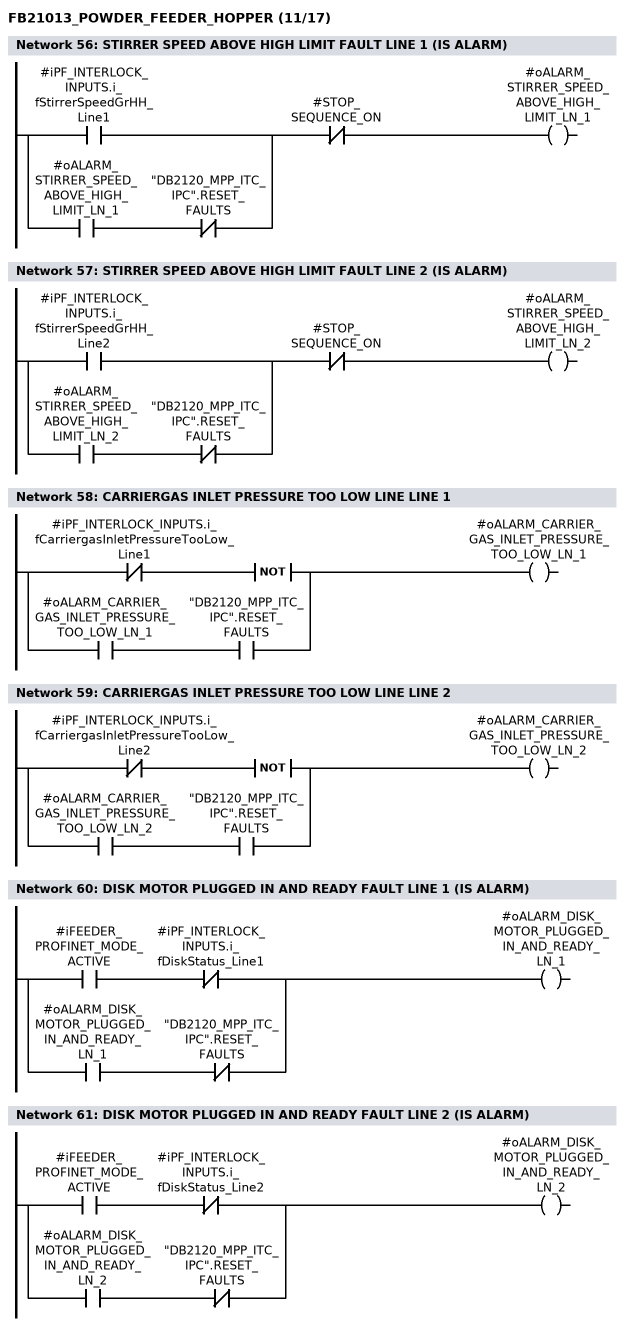
   RUNG wire#powerrail
      Contact( #iPF_INTERLOCK_INPUTS.i_fStirrerSpeedGrHH_Line1 )
      wire#w1
      I_Contact( #STOP_SEQUENCE_ON )
      Coil( #oALARM_STIRRER_SPEED_ABOVE_HIGH_LIMIT_LN_1 )
   END_RUNG
   RUNG wire#powerrail
      Contact( #oALARM_STIRRER_SPEED_ABOVE_HIGH_LIMIT_LN_1 )
      I_Contact( "DB2120_MPP_ITC_IPC".RESET_FAULTS )
   END_RUNG wire#w1
   // the same network as SCL:
   #oALARM_STIRRER_SPEED_ABOVE_HIGH_LIMIT_LN_1 := (#iPF_INTERLOCK_INPUTS.i_fStirrerSpeedGrHH_Line1 OR (#oALARM_STIRRER_SPEED_ABOVE_HIGH_LIMIT_LN_1 AND NOT "DB2120_MPP_ITC_IPC".RESET_FAULTS)) AND NOT #STOP_SEQUENCE_ON;
END_REGION

REGION Network 57: STIRRER SPEED ABOVE HIGH LIMIT FAULT LINE 2 (IS ALARM)
   RUNG wire#powerrail
      Contact( #iPF_INTERLOCK_INPUTS.i_fStirrerSpeedGrHH_Line2 )
      wire#w1
      I_Contact( #STOP_SEQUENCE_ON )
      Coil( #oALARM_STIRRER_SPEED_ABOVE_HIGH_LIMIT_LN_2 )
   END_RUNG
   RUNG wire#powerrail
      Contact( #oALARM_STIRRER_SPEED_ABOVE_HIGH_LIMIT_LN_2 )
      I_Contact( "DB2120_MPP_ITC_IPC".RESET_FAULTS )
   END_RUNG wire#w1
   // the same network as SCL:
   #oALARM_STIRRER_SPEED_ABOVE_HIGH_LIMIT_LN_2 := (#iPF_INTERLOCK_INPUTS.i_fStirrerSpeedGrHH_Line2 OR (#oALARM_STIRRER_SPEED_ABOVE_HIGH_LIMIT_LN_2 AND NOT "DB2120_MPP_ITC_IPC".RESET_FAULTS)) AND NOT #STOP_SEQUENCE_ON;
END_REGION

REGION Network 58: CARRIERGAS INLET PRESSURE TOO LOW LINE LINE 1
   RUNG wire#powerrail
      I_Contact( #iPF_INTERLOCK_INPUTS.i_fCarriergasInletPressureTooLow_Line1 )
      Not()
      wire#w1
      Coil( #oALARM_CARRIER_GAS_INLET_PRESSURE_TOO_LOW_LN_1 )
   END_RUNG
   RUNG wire#powerrail
      Contact( #oALARM_CARRIER_GAS_INLET_PRESSURE_TOO_LOW_LN_1 )
      Contact( "DB2120_MPP_ITC_IPC".RESET_FAULTS )
   END_RUNG wire#w1
   // the same network as SCL:
   #oALARM_CARRIER_GAS_INLET_PRESSURE_TOO_LOW_LN_1 := NOT (NOT #iPF_INTERLOCK_INPUTS.i_fCarriergasInletPressureTooLow_Line1) OR (#oALARM_CARRIER_GAS_INLET_PRESSURE_TOO_LOW_LN_1 AND "DB2120_MPP_ITC_IPC".RESET_FAULTS);
END_REGION

REGION Network 59: CARRIERGAS INLET PRESSURE TOO LOW LINE LINE 2
   RUNG wire#powerrail
      I_Contact( #iPF_INTERLOCK_INPUTS.i_fCarriergasInletPressureTooLow_Line2 )
      Not()
      wire#w1
      Coil( #oALARM_CARRIER_GAS_INLET_PRESSURE_TOO_LOW_LN_2 )
   END_RUNG
   RUNG wire#powerrail
      Contact( #oALARM_CARRIER_GAS_INLET_PRESSURE_TOO_LOW_LN_2 )
      Contact( "DB2120_MPP_ITC_IPC".RESET_FAULTS )
   END_RUNG wire#w1
   // the same network as SCL:
   #oALARM_CARRIER_GAS_INLET_PRESSURE_TOO_LOW_LN_2 := NOT (NOT #iPF_INTERLOCK_INPUTS.i_fCarriergasInletPressureTooLow_Line2) OR (#oALARM_CARRIER_GAS_INLET_PRESSURE_TOO_LOW_LN_2 AND "DB2120_MPP_ITC_IPC".RESET_FAULTS);
END_REGION

REGION Network 60: DISK MOTOR PLUGGED IN AND READY FAULT LINE 1 (IS ALARM)
   RUNG wire#powerrail
      Contact( #iFEEDER_PROFINET_MODE_ACTIVE )
      I_Contact( #iPF_INTERLOCK_INPUTS.i_fDiskStatus_Line1 )
      wire#w1
      Coil( #oALARM_DISK_MOTOR_PLUGGED_IN_AND_READY_LN_1 )
   END_RUNG
   RUNG wire#powerrail
      Contact( #oALARM_DISK_MOTOR_PLUGGED_IN_AND_READY_LN_1 )
      I_Contact( "DB2120_MPP_ITC_IPC".RESET_FAULTS )
   END_RUNG wire#w1
   // the same network as SCL:
   #oALARM_DISK_MOTOR_PLUGGED_IN_AND_READY_LN_1 := (#iFEEDER_PROFINET_MODE_ACTIVE AND NOT #iPF_INTERLOCK_INPUTS.i_fDiskStatus_Line1) OR (#oALARM_DISK_MOTOR_PLUGGED_IN_AND_READY_LN_1 AND NOT "DB2120_MPP_ITC_IPC".RESET_FAULTS);
END_REGION

REGION Network 61: DISK MOTOR PLUGGED IN AND READY FAULT LINE 2 (IS ALARM)
   RUNG wire#powerrail
      Contact( #iFEEDER_PROFINET_MODE_ACTIVE )
      I_Contact( #iPF_INTERLOCK_INPUTS.i_fDiskStatus_Line2 )
      wire#w1
      Coil( #oALARM_DISK_MOTOR_PLUGGED_IN_AND_READY_LN_2 )
   END_RUNG
   RUNG wire#powerrail
      Contact( #oALARM_DISK_MOTOR_PLUGGED_IN_AND_READY_LN_2 )
      I_Contact( "DB2120_MPP_ITC_IPC".RESET_FAULTS )
   END_RUNG wire#w1
   // the same network as SCL:
   #oALARM_DISK_MOTOR_PLUGGED_IN_AND_READY_LN_2 := (#iFEEDER_PROFINET_MODE_ACTIVE AND NOT #iPF_INTERLOCK_INPUTS.i_fDiskStatus_Line2) OR (#oALARM_DISK_MOTOR_PLUGGED_IN_AND_READY_LN_2 AND NOT "DB2120_MPP_ITC_IPC".RESET_FAULTS);
END_REGION

REGION Network 62: STIRRER PLUGGED IN AND READY FAULT LINE 1 (IS ALARM)
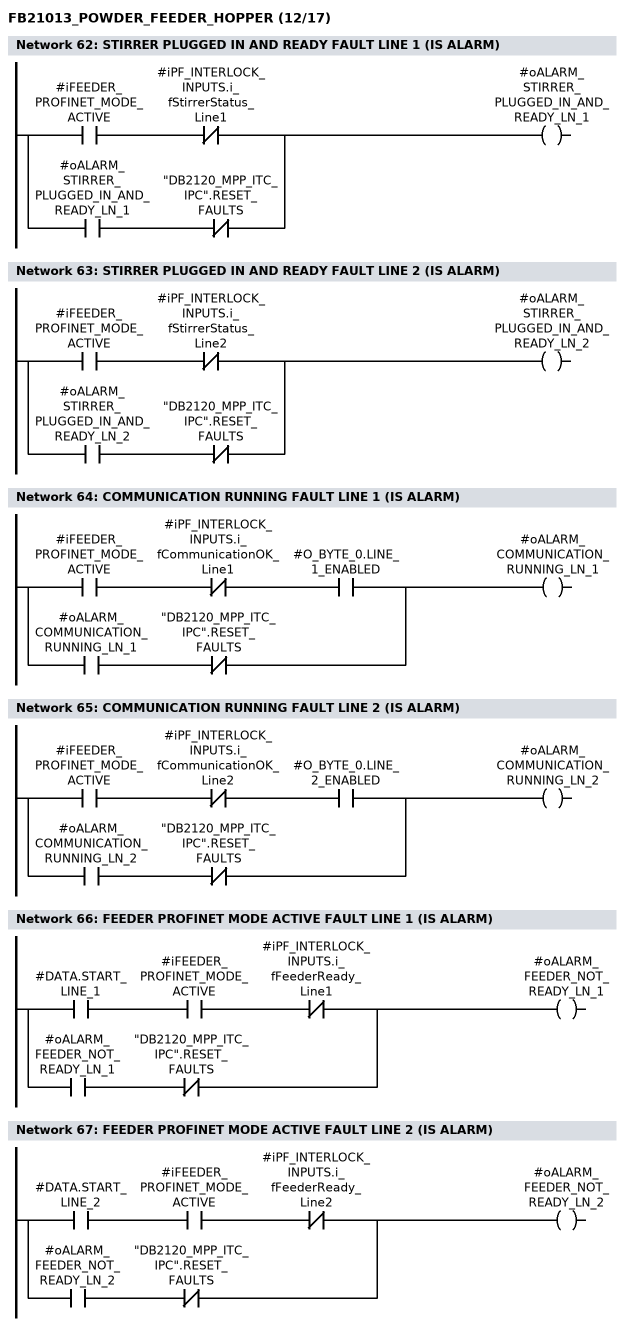
   RUNG wire#powerrail
      Contact( #iFEEDER_PROFINET_MODE_ACTIVE )
      I_Contact( #iPF_INTERLOCK_INPUTS.i_fStirrerStatus_Line1 )
      wire#w1
      Coil( #oALARM_STIRRER_PLUGGED_IN_AND_READY_LN_1 )
   END_RUNG
   RUNG wire#powerrail
      Contact( #oALARM_STIRRER_PLUGGED_IN_AND_READY_LN_1 )
      I_Contact( "DB2120_MPP_ITC_IPC".RESET_FAULTS )
   END_RUNG wire#w1
   // the same network as SCL:
   #oALARM_STIRRER_PLUGGED_IN_AND_READY_LN_1 := (#iFEEDER_PROFINET_MODE_ACTIVE AND NOT #iPF_INTERLOCK_INPUTS.i_fStirrerStatus_Line1) OR (#oALARM_STIRRER_PLUGGED_IN_AND_READY_LN_1 AND NOT "DB2120_MPP_ITC_IPC".RESET_FAULTS);
END_REGION

REGION Network 63: STIRRER PLUGGED IN AND READY FAULT LINE 2 (IS ALARM)
   RUNG wire#powerrail
      Contact( #iFEEDER_PROFINET_MODE_ACTIVE )
      I_Contact( #iPF_INTERLOCK_INPUTS.i_fStirrerStatus_Line2 )
      wire#w1
      Coil( #oALARM_STIRRER_PLUGGED_IN_AND_READY_LN_2 )
   END_RUNG
   RUNG wire#powerrail
      Contact( #oALARM_STIRRER_PLUGGED_IN_AND_READY_LN_2 )
      I_Contact( "DB2120_MPP_ITC_IPC".RESET_FAULTS )
   END_RUNG wire#w1
   // the same network as SCL:
   #oALARM_STIRRER_PLUGGED_IN_AND_READY_LN_2 := (#iFEEDER_PROFINET_MODE_ACTIVE AND NOT #iPF_INTERLOCK_INPUTS.i_fStirrerStatus_Line2) OR (#oALARM_STIRRER_PLUGGED_IN_AND_READY_LN_2 AND NOT "DB2120_MPP_ITC_IPC".RESET_FAULTS);
END_REGION

REGION Network 64: COMMUNICATION RUNNING FAULT LINE 1 (IS ALARM)
   RUNG wire#powerrail
      Contact( #iFEEDER_PROFINET_MODE_ACTIVE )
      I_Contact( #iPF_INTERLOCK_INPUTS.i_fCommunicationOK_Line1 )
      Contact( #O_BYTE_0.LINE_1_ENABLED )
      wire#w1
      Coil( #oALARM_COMMUNICATION_RUNNING_LN_1 )
   END_RUNG
   RUNG wire#powerrail
      Contact( #oALARM_COMMUNICATION_RUNNING_LN_1 )
      I_Contact( "DB2120_MPP_ITC_IPC".RESET_FAULTS )
   END_RUNG wire#w1
   // the same network as SCL:
   #oALARM_COMMUNICATION_RUNNING_LN_1 := (#iFEEDER_PROFINET_MODE_ACTIVE AND NOT #iPF_INTERLOCK_INPUTS.i_fCommunicationOK_Line1 AND #O_BYTE_0.LINE_1_ENABLED) OR (#oALARM_COMMUNICATION_RUNNING_LN_1 AND NOT "DB2120_MPP_ITC_IPC".RESET_FAULTS);
END_REGION

REGION Network 65: COMMUNICATION RUNNING FAULT LINE 2 (IS ALARM)
   RUNG wire#powerrail
      Contact( #iFEEDER_PROFINET_MODE_ACTIVE )
      I_Contact( #iPF_INTERLOCK_INPUTS.i_fCommunicationOK_Line2 )
      Contact( #O_BYTE_0.LINE_2_ENABLED )
      wire#w1
      Coil( #oALARM_COMMUNICATION_RUNNING_LN_2 )
   END_RUNG
   RUNG wire#powerrail
      Contact( #oALARM_COMMUNICATION_RUNNING_LN_2 )
      I_Contact( "DB2120_MPP_ITC_IPC".RESET_FAULTS )
   END_RUNG wire#w1
   // the same network as SCL:
   #oALARM_COMMUNICATION_RUNNING_LN_2 := (#iFEEDER_PROFINET_MODE_ACTIVE AND NOT #iPF_INTERLOCK_INPUTS.i_fCommunicationOK_Line2 AND #O_BYTE_0.LINE_2_ENABLED) OR (#oALARM_COMMUNICATION_RUNNING_LN_2 AND NOT "DB2120_MPP_ITC_IPC".RESET_FAULTS);
END_REGION

REGION Network 66: FEEDER PROFINET MODE ACTIVE FAULT LINE 1 (IS ALARM)
   RUNG wire#powerrail
      Contact( #DATA.START_LINE_1 )
      Contact( #iFEEDER_PROFINET_MODE_ACTIVE )
      I_Contact( #iPF_INTERLOCK_INPUTS.i_fFeederReady_Line1 )
      wire#w1
      Coil( #oALARM_FEEDER_NOT_READY_LN_1 )
   END_RUNG
   RUNG wire#powerrail
      Contact( #oALARM_FEEDER_NOT_READY_LN_1 )
      I_Contact( "DB2120_MPP_ITC_IPC".RESET_FAULTS )
   END_RUNG wire#w1
   // the same network as SCL:
   #oALARM_FEEDER_NOT_READY_LN_1 := (#DATA.START_LINE_1 AND #iFEEDER_PROFINET_MODE_ACTIVE AND NOT #iPF_INTERLOCK_INPUTS.i_fFeederReady_Line1) OR (#oALARM_FEEDER_NOT_READY_LN_1 AND NOT "DB2120_MPP_ITC_IPC".RESET_FAULTS);
END_REGION

REGION Network 67: FEEDER PROFINET MODE ACTIVE FAULT LINE 2 (IS ALARM)
   RUNG wire#powerrail
      Contact( #DATA.START_LINE_2 )
      Contact( #iFEEDER_PROFINET_MODE_ACTIVE )
      I_Contact( #iPF_INTERLOCK_INPUTS.i_fFeederReady_Line2 )
      wire#w1
      Coil( #oALARM_FEEDER_NOT_READY_LN_2 )
   END_RUNG
   RUNG wire#powerrail
      Contact( #oALARM_FEEDER_NOT_READY_LN_2 )
      I_Contact( "DB2120_MPP_ITC_IPC".RESET_FAULTS )
   END_RUNG wire#w1
   // the same network as SCL:
   #oALARM_FEEDER_NOT_READY_LN_2 := (#DATA.START_LINE_2 AND #iFEEDER_PROFINET_MODE_ACTIVE AND NOT #iPF_INTERLOCK_INPUTS.i_fFeederReady_Line2) OR (#oALARM_FEEDER_NOT_READY_LN_2 AND NOT "DB2120_MPP_ITC_IPC".RESET_FAULTS);
END_REGION

REGION Network 68: CARRIER GAS FLOW BELOW LOW LIMIT FAULT LINE 1 (WARNING)
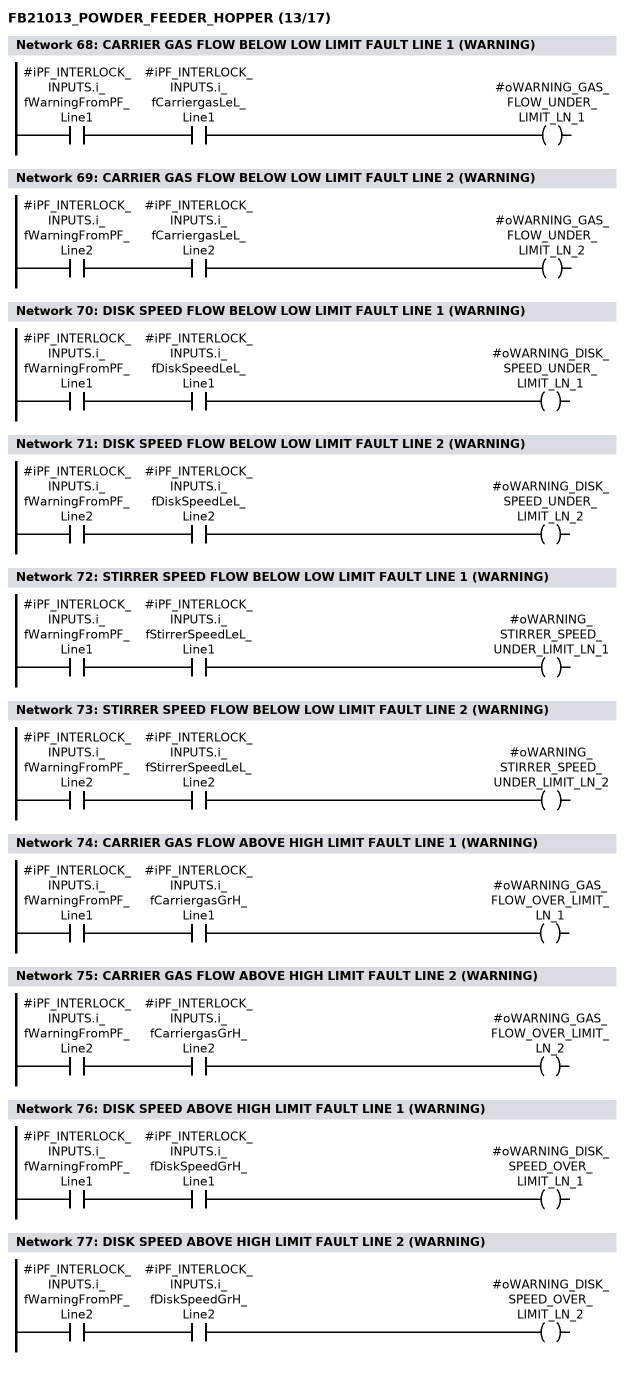
   RUNG wire#powerrail
      Contact( #iPF_INTERLOCK_INPUTS.i_fWarningFromPF_Line1 )
      Contact( #iPF_INTERLOCK_INPUTS.i_fCarriergasLeL_Line1 )
      Coil( #oWARNING_GAS_FLOW_UNDER_LIMIT_LN_1 )
   END_RUNG
   // the same network as SCL:
   #oWARNING_GAS_FLOW_UNDER_LIMIT_LN_1 := #iPF_INTERLOCK_INPUTS.i_fWarningFromPF_Line1 AND #iPF_INTERLOCK_INPUTS.i_fCarriergasLeL_Line1;
END_REGION

REGION Network 69: CARRIER GAS FLOW BELOW LOW LIMIT FAULT LINE 2 (WARNING)
   RUNG wire#powerrail
      Contact( #iPF_INTERLOCK_INPUTS.i_fWarningFromPF_Line2 )
      Contact( #iPF_INTERLOCK_INPUTS.i_fCarriergasLeL_Line2 )
      Coil( #oWARNING_GAS_FLOW_UNDER_LIMIT_LN_2 )
   END_RUNG
   // the same network as SCL:
   #oWARNING_GAS_FLOW_UNDER_LIMIT_LN_2 := #iPF_INTERLOCK_INPUTS.i_fWarningFromPF_Line2 AND #iPF_INTERLOCK_INPUTS.i_fCarriergasLeL_Line2;
END_REGION

REGION Network 70: DISK SPEED FLOW BELOW LOW LIMIT FAULT LINE 1 (WARNING)
   RUNG wire#powerrail
      Contact( #iPF_INTERLOCK_INPUTS.i_fWarningFromPF_Line1 )
      Contact( #iPF_INTERLOCK_INPUTS.i_fDiskSpeedLeL_Line1 )
      Coil( #oWARNING_DISK_SPEED_UNDER_LIMIT_LN_1 )
   END_RUNG
   // the same network as SCL:
   #oWARNING_DISK_SPEED_UNDER_LIMIT_LN_1 := #iPF_INTERLOCK_INPUTS.i_fWarningFromPF_Line1 AND #iPF_INTERLOCK_INPUTS.i_fDiskSpeedLeL_Line1;
END_REGION

REGION Network 71: DISK SPEED FLOW BELOW LOW LIMIT FAULT LINE 2 (WARNING)
   RUNG wire#powerrail
      Contact( #iPF_INTERLOCK_INPUTS.i_fWarningFromPF_Line2 )
      Contact( #iPF_INTERLOCK_INPUTS.i_fDiskSpeedLeL_Line2 )
      Coil( #oWARNING_DISK_SPEED_UNDER_LIMIT_LN_2 )
   END_RUNG
   // the same network as SCL:
   #oWARNING_DISK_SPEED_UNDER_LIMIT_LN_2 := #iPF_INTERLOCK_INPUTS.i_fWarningFromPF_Line2 AND #iPF_INTERLOCK_INPUTS.i_fDiskSpeedLeL_Line2;
END_REGION

REGION Network 72: STIRRER SPEED FLOW BELOW LOW LIMIT FAULT LINE 1 (WARNING)
   RUNG wire#powerrail
      Contact( #iPF_INTERLOCK_INPUTS.i_fWarningFromPF_Line1 )
      Contact( #iPF_INTERLOCK_INPUTS.i_fStirrerSpeedLeL_Line1 )
      Coil( #oWARNING_STIRRER_SPEED_UNDER_LIMIT_LN_1 )
   END_RUNG
   // the same network as SCL:
   #oWARNING_STIRRER_SPEED_UNDER_LIMIT_LN_1 := #iPF_INTERLOCK_INPUTS.i_fWarningFromPF_Line1 AND #iPF_INTERLOCK_INPUTS.i_fStirrerSpeedLeL_Line1;
END_REGION

REGION Network 73: STIRRER SPEED FLOW BELOW LOW LIMIT FAULT LINE 2 (WARNING)
   RUNG wire#powerrail
      Contact( #iPF_INTERLOCK_INPUTS.i_fWarningFromPF_Line2 )
      Contact( #iPF_INTERLOCK_INPUTS.i_fStirrerSpeedLeL_Line2 )
      Coil( #oWARNING_STIRRER_SPEED_UNDER_LIMIT_LN_2 )
   END_RUNG
   // the same network as SCL:
   #oWARNING_STIRRER_SPEED_UNDER_LIMIT_LN_2 := #iPF_INTERLOCK_INPUTS.i_fWarningFromPF_Line2 AND #iPF_INTERLOCK_INPUTS.i_fStirrerSpeedLeL_Line2;
END_REGION

REGION Network 74: CARRIER GAS FLOW ABOVE HIGH LIMIT FAULT LINE 1 (WARNING)
   RUNG wire#powerrail
      Contact( #iPF_INTERLOCK_INPUTS.i_fWarningFromPF_Line1 )
      Contact( #iPF_INTERLOCK_INPUTS.i_fCarriergasGrH_Line1 )
      Coil( #oWARNING_GAS_FLOW_OVER_LIMIT_LN_1 )
   END_RUNG
   // the same network as SCL:
   #oWARNING_GAS_FLOW_OVER_LIMIT_LN_1 := #iPF_INTERLOCK_INPUTS.i_fWarningFromPF_Line1 AND #iPF_INTERLOCK_INPUTS.i_fCarriergasGrH_Line1;
END_REGION

REGION Network 75: CARRIER GAS FLOW ABOVE HIGH LIMIT FAULT LINE 2 (WARNING)
   RUNG wire#powerrail
      Contact( #iPF_INTERLOCK_INPUTS.i_fWarningFromPF_Line2 )
      Contact( #iPF_INTERLOCK_INPUTS.i_fCarriergasGrH_Line2 )
      Coil( #oWARNING_GAS_FLOW_OVER_LIMIT_LN_2 )
   END_RUNG
   // the same network as SCL:
   #oWARNING_GAS_FLOW_OVER_LIMIT_LN_2 := #iPF_INTERLOCK_INPUTS.i_fWarningFromPF_Line2 AND #iPF_INTERLOCK_INPUTS.i_fCarriergasGrH_Line2;
END_REGION

REGION Network 76: DISK SPEED ABOVE HIGH LIMIT FAULT LINE 1 (WARNING)
   RUNG wire#powerrail
      Contact( #iPF_INTERLOCK_INPUTS.i_fWarningFromPF_Line1 )
      Contact( #iPF_INTERLOCK_INPUTS.i_fDiskSpeedGrH_Line1 )
      Coil( #oWARNING_DISK_SPEED_OVER_LIMIT_LN_1 )
   END_RUNG
   // the same network as SCL:
   #oWARNING_DISK_SPEED_OVER_LIMIT_LN_1 := #iPF_INTERLOCK_INPUTS.i_fWarningFromPF_Line1 AND #iPF_INTERLOCK_INPUTS.i_fDiskSpeedGrH_Line1;
END_REGION

REGION Network 77: DISK SPEED ABOVE HIGH LIMIT FAULT LINE 2 (WARNING)
   RUNG wire#powerrail
      Contact( #iPF_INTERLOCK_INPUTS.i_fWarningFromPF_Line2 )
      Contact( #iPF_INTERLOCK_INPUTS.i_fDiskSpeedGrH_Line2 )
      Coil( #oWARNING_DISK_SPEED_OVER_LIMIT_LN_2 )
   END_RUNG
   // the same network as SCL:
   #oWARNING_DISK_SPEED_OVER_LIMIT_LN_2 := #iPF_INTERLOCK_INPUTS.i_fWarningFromPF_Line2 AND #iPF_INTERLOCK_INPUTS.i_fDiskSpeedGrH_Line2;
END_REGION

REGION Network 78: STIRRER SPEED ABOVE HIGH LIMIT FAULT LINE 1 (WARNING)
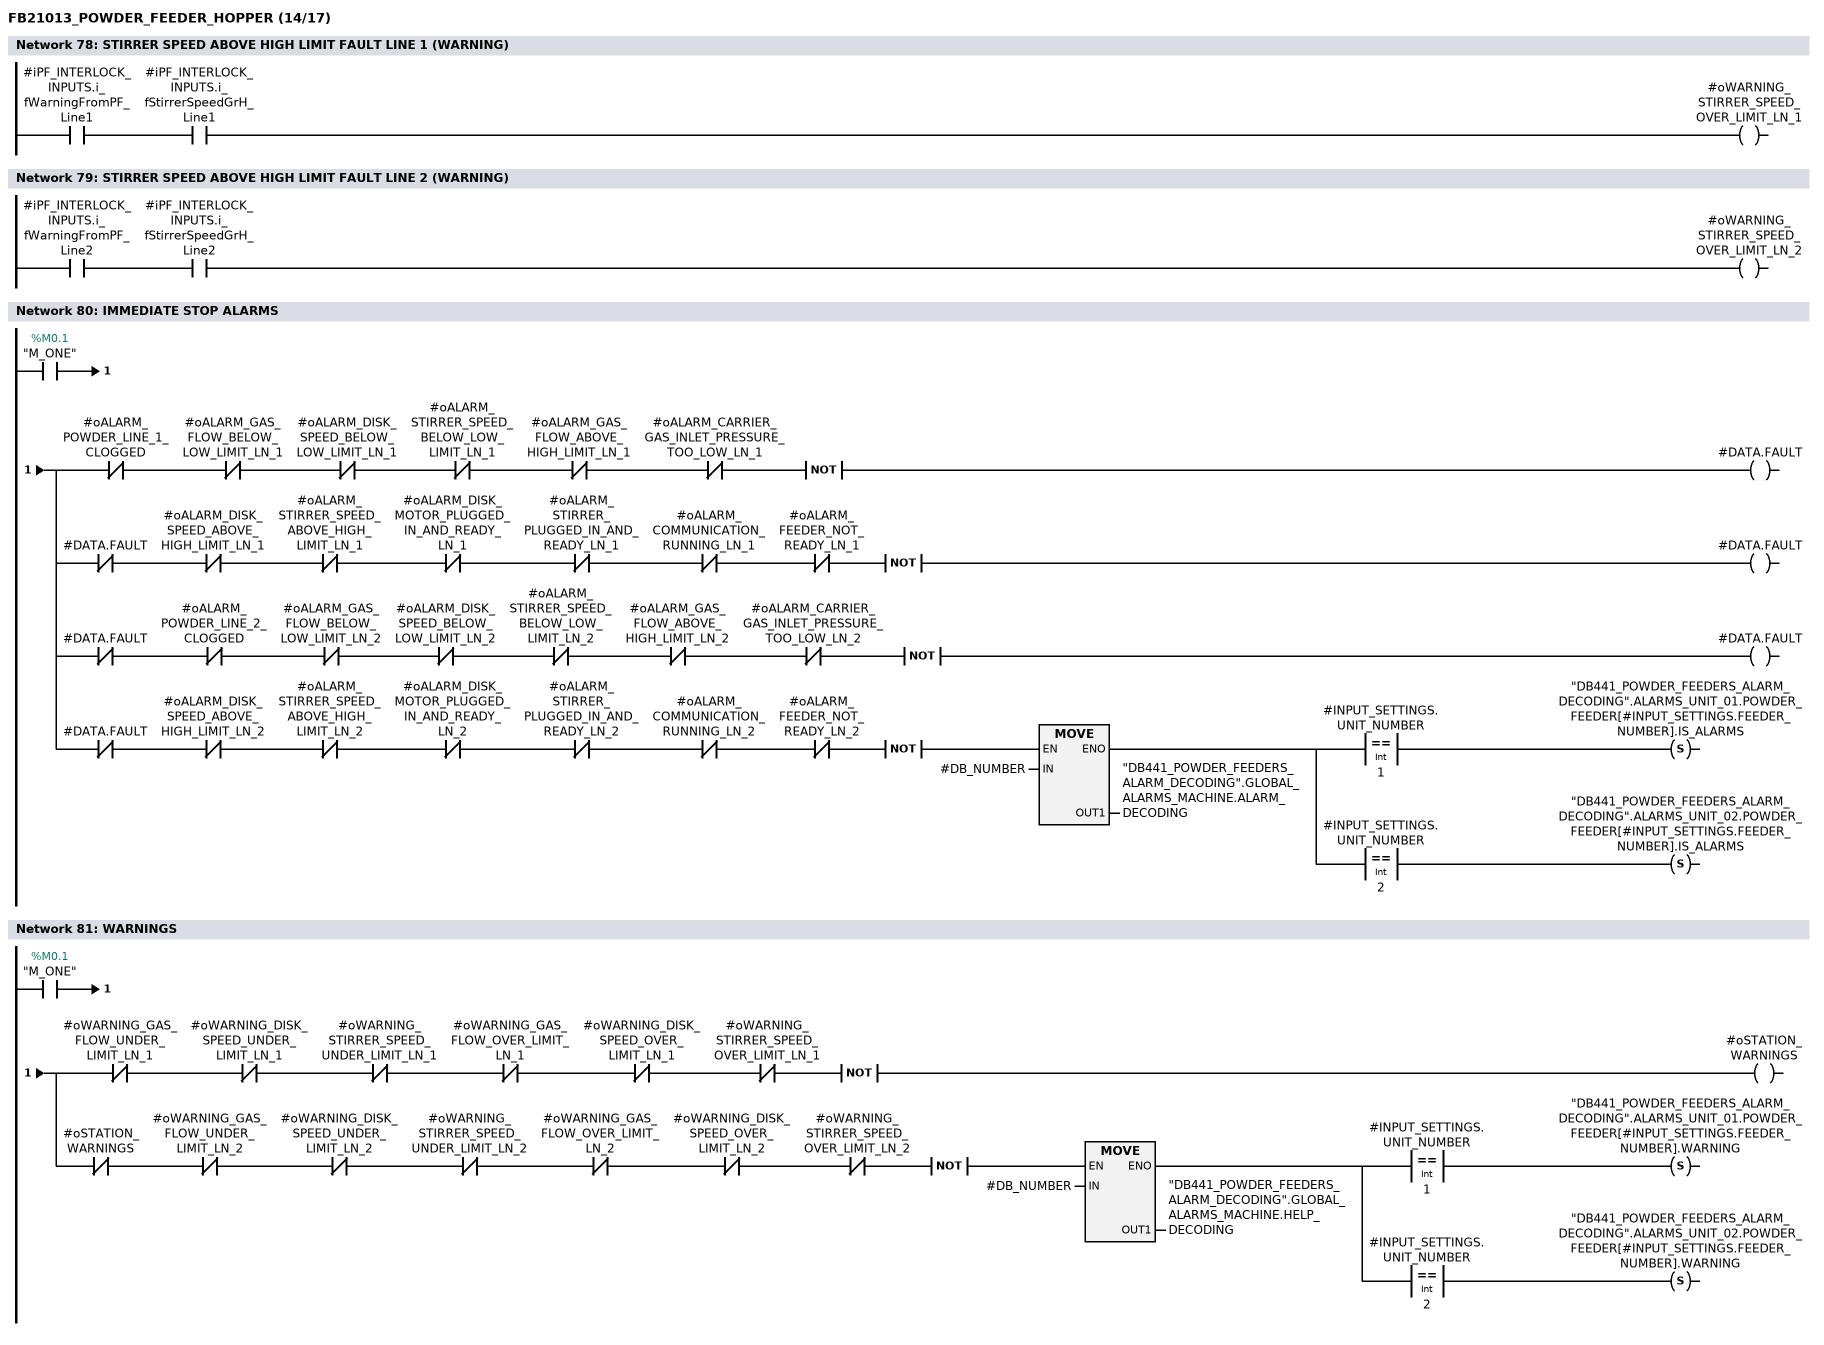
   RUNG wire#powerrail
      Contact( #iPF_INTERLOCK_INPUTS.i_fWarningFromPF_Line1 )
      Contact( #iPF_INTERLOCK_INPUTS.i_fStirrerSpeedGrH_Line1 )
      Coil( #oWARNING_STIRRER_SPEED_OVER_LIMIT_LN_1 )
   END_RUNG
   // the same network as SCL:
   #oWARNING_STIRRER_SPEED_OVER_LIMIT_LN_1 := #iPF_INTERLOCK_INPUTS.i_fWarningFromPF_Line1 AND #iPF_INTERLOCK_INPUTS.i_fStirrerSpeedGrH_Line1;
END_REGION

REGION Network 79: STIRRER SPEED ABOVE HIGH LIMIT FAULT LINE 2 (WARNING)
   RUNG wire#powerrail
      Contact( #iPF_INTERLOCK_INPUTS.i_fWarningFromPF_Line2 )
      Contact( #iPF_INTERLOCK_INPUTS.i_fStirrerSpeedGrH_Line2 )
      Coil( #oWARNING_STIRRER_SPEED_OVER_LIMIT_LN_2 )
   END_RUNG
   // the same network as SCL:
   #oWARNING_STIRRER_SPEED_OVER_LIMIT_LN_2 := #iPF_INTERLOCK_INPUTS.i_fWarningFromPF_Line2 AND #iPF_INTERLOCK_INPUTS.i_fStirrerSpeedGrH_Line2;
END_REGION

